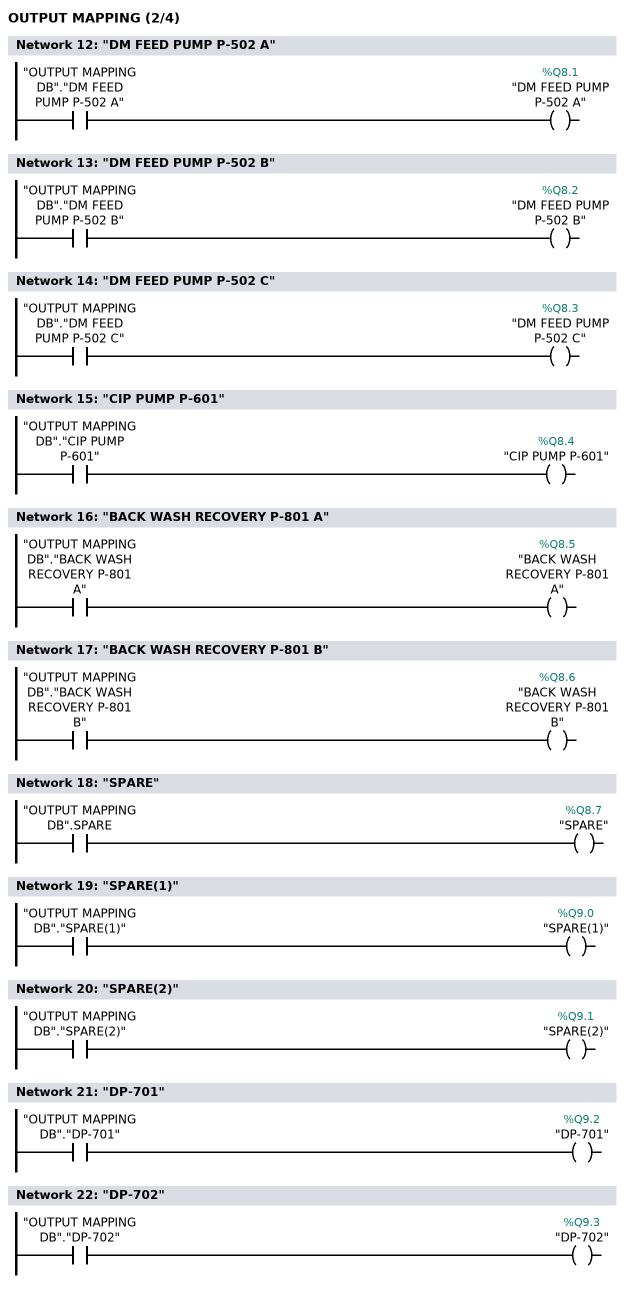
   RUNG wire#powerrail
      Contact( "OUTPUT MAPPING DB"."DM FEED PUMP P-502 A" )
      Coil( "DM FEED PUMP P-502 A" )
   END_RUNG
   // the same network as SCL:
   "DM FEED PUMP P-502 A" := "OUTPUT MAPPING DB"."DM FEED PUMP P-502 A";
END_REGION

REGION Network 13: "DM FEED PUMP P-502 B"
   RUNG wire#powerrail
      Contact( "OUTPUT MAPPING DB"."DM FEED PUMP P-502 B" )
      Coil( "DM FEED PUMP P-502 B" )
   END_RUNG
   // the same network as SCL:
   "DM FEED PUMP P-502 B" := "OUTPUT MAPPING DB"."DM FEED PUMP P-502 B";
END_REGION

REGION Network 14: "DM FEED PUMP P-502 C"
   RUNG wire#powerrail
      Contact( "OUTPUT MAPPING DB"."DM FEED PUMP P-502 C" )
      Coil( "DM FEED PUMP P-502 C" )
   END_RUNG
   // the same network as SCL:
   "DM FEED PUMP P-502 C" := "OUTPUT MAPPING DB"."DM FEED PUMP P-502 C";
END_REGION

REGION Network 15: "CIP PUMP P-601"
   RUNG wire#powerrail
      Contact( "OUTPUT MAPPING DB"."CIP PUMP P-601" )
      Coil( "CIP PUMP P-601" )
   END_RUNG
   // the same network as SCL:
   "CIP PUMP P-601" := "OUTPUT MAPPING DB"."CIP PUMP P-601";
END_REGION

REGION Network 16: "BACK WASH RECOVERY P-801 A"
   RUNG wire#powerrail
      Contact( "OUTPUT MAPPING DB"."BACK WASH RECOVERY P-801 A" )
      Coil( "BACK WASH RECOVERY P-801 A" )
   END_RUNG
   // the same network as SCL:
   "BACK WASH RECOVERY P-801 A" := "OUTPUT MAPPING DB"."BACK WASH RECOVERY P-801 A";
END_REGION

REGION Network 17: "BACK WASH RECOVERY P-801 B"
   RUNG wire#powerrail
      Contact( "OUTPUT MAPPING DB"."BACK WASH RECOVERY P-801 B" )
      Coil( "BACK WASH RECOVERY P-801 B" )
   END_RUNG
   // the same network as SCL:
   "BACK WASH RECOVERY P-801 B" := "OUTPUT MAPPING DB"."BACK WASH RECOVERY P-801 B";
END_REGION

REGION Network 18: "SPARE"
   RUNG wire#powerrail
      Contact( "OUTPUT MAPPING DB".SPARE )
      Coil( "SPARE" )
   END_RUNG
   // the same network as SCL:
   "SPARE" := "OUTPUT MAPPING DB".SPARE;
END_REGION

REGION Network 19: "SPARE(1)"
   RUNG wire#powerrail
      Contact( "OUTPUT MAPPING DB"."SPARE(1)" )
      Coil( "SPARE(1)" )
   END_RUNG
   // the same network as SCL:
   "SPARE(1)" := "OUTPUT MAPPING DB"."SPARE(1)";
END_REGION

REGION Network 20: "SPARE(2)"
   RUNG wire#powerrail
      Contact( "OUTPUT MAPPING DB"."SPARE(2)" )
      Coil( "SPARE(2)" )
   END_RUNG
   // the same network as SCL:
   "SPARE(2)" := "OUTPUT MAPPING DB"."SPARE(2)";
END_REGION

REGION Network 21: "DP-701"
   RUNG wire#powerrail
      Contact( "OUTPUT MAPPING DB"."DP-701" )
      Coil( "DP-701" )
   END_RUNG
   // the same network as SCL:
   "DP-701" := "OUTPUT MAPPING DB"."DP-701";
END_REGION

REGION Network 22: "DP-702"
   RUNG wire#powerrail
      Contact( "OUTPUT MAPPING DB"."DP-702" )
      Coil( "DP-702" )
   END_RUNG
   // the same network as SCL:
   "DP-702" := "OUTPUT MAPPING DB"."DP-702";
END_REGION

REGION Network 23: "NaOCL DOSING D-706 A"
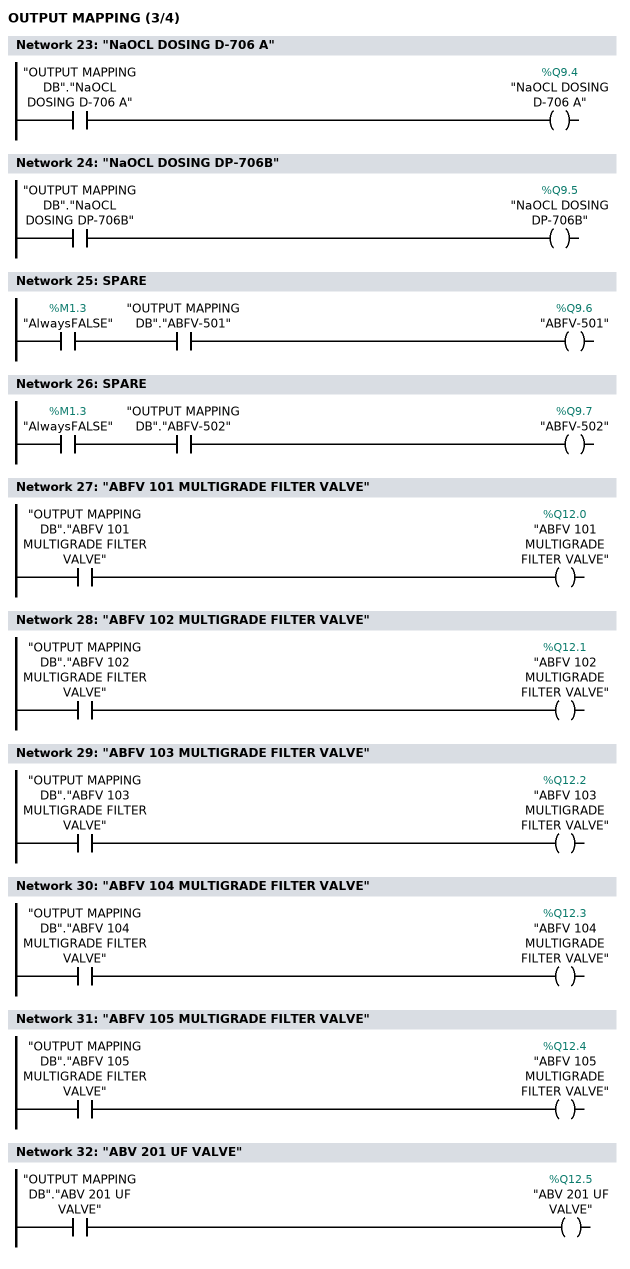
   RUNG wire#powerrail
      Contact( "OUTPUT MAPPING DB"."NaOCL DOSING D-706 A" )
      Coil( "NaOCL DOSING D-706 A" )
   END_RUNG
   // the same network as SCL:
   "NaOCL DOSING D-706 A" := "OUTPUT MAPPING DB"."NaOCL DOSING D-706 A";
END_REGION

REGION Network 24: "NaOCL DOSING DP-706B"
   RUNG wire#powerrail
      Contact( "OUTPUT MAPPING DB"."NaOCL DOSING DP-706B" )
      Coil( "NaOCL DOSING DP-706B" )
   END_RUNG
   // the same network as SCL:
   "NaOCL DOSING DP-706B" := "OUTPUT MAPPING DB"."NaOCL DOSING DP-706B";
END_REGION

REGION Network 25: SPARE
   RUNG wire#powerrail
      Contact( "AlwaysFALSE" )
      Contact( "OUTPUT MAPPING DB"."ABFV-501" )
      Coil( "ABFV-501" )
   END_RUNG
   // the same network as SCL:
   "ABFV-501" := "AlwaysFALSE" AND "OUTPUT MAPPING DB"."ABFV-501";
END_REGION

REGION Network 26: SPARE
   RUNG wire#powerrail
      Contact( "AlwaysFALSE" )
      Contact( "OUTPUT MAPPING DB"."ABFV-502" )
      Coil( "ABFV-502" )
   END_RUNG
   // the same network as SCL:
   "ABFV-502" := "AlwaysFALSE" AND "OUTPUT MAPPING DB"."ABFV-502";
END_REGION

REGION Network 27: "ABFV 101 MULTIGRADE FILTER VALVE"
   RUNG wire#powerrail
      Contact( "OUTPUT MAPPING DB"."ABFV 101 MULTIGRADE FILTER VALVE" )
      Coil( "ABFV 101 MULTIGRADE FILTER VALVE" )
   END_RUNG
   // the same network as SCL:
   "ABFV 101 MULTIGRADE FILTER VALVE" := "OUTPUT MAPPING DB"."ABFV 101 MULTIGRADE FILTER VALVE";
END_REGION

REGION Network 28: "ABFV 102 MULTIGRADE FILTER VALVE"
   RUNG wire#powerrail
      Contact( "OUTPUT MAPPING DB"."ABFV 102 MULTIGRADE FILTER VALVE" )
      Coil( "ABFV 102 MULTIGRADE FILTER VALVE" )
   END_RUNG
   // the same network as SCL:
   "ABFV 102 MULTIGRADE FILTER VALVE" := "OUTPUT MAPPING DB"."ABFV 102 MULTIGRADE FILTER VALVE";
END_REGION

REGION Network 29: "ABFV 103 MULTIGRADE FILTER VALVE"
   RUNG wire#powerrail
      Contact( "OUTPUT MAPPING DB"."ABFV 103 MULTIGRADE FILTER VALVE" )
      Coil( "ABFV 103 MULTIGRADE FILTER VALVE" )
   END_RUNG
   // the same network as SCL:
   "ABFV 103 MULTIGRADE FILTER VALVE" := "OUTPUT MAPPING DB"."ABFV 103 MULTIGRADE FILTER VALVE";
END_REGION

REGION Network 30: "ABFV 104 MULTIGRADE FILTER VALVE"
   RUNG wire#powerrail
      Contact( "OUTPUT MAPPING DB"."ABFV 104 MULTIGRADE FILTER VALVE" )
      Coil( "ABFV 104 MULTIGRADE FILTER VALVE" )
   END_RUNG
   // the same network as SCL:
   "ABFV 104 MULTIGRADE FILTER VALVE" := "OUTPUT MAPPING DB"."ABFV 104 MULTIGRADE FILTER VALVE";
END_REGION

REGION Network 31: "ABFV 105 MULTIGRADE FILTER VALVE"
   RUNG wire#powerrail
      Contact( "OUTPUT MAPPING DB"."ABFV 105 MULTIGRADE FILTER VALVE" )
      Coil( "ABFV 105 MULTIGRADE FILTER VALVE" )
   END_RUNG
   // the same network as SCL:
   "ABFV 105 MULTIGRADE FILTER VALVE" := "OUTPUT MAPPING DB"."ABFV 105 MULTIGRADE FILTER VALVE";
END_REGION

REGION Network 32: "ABV 201 UF VALVE"
   RUNG wire#powerrail
      Contact( "OUTPUT MAPPING DB"."ABV 201 UF VALVE" )
      Coil( "ABV 201 UF VALVE" )
   END_RUNG
   // the same network as SCL:
   "ABV 201 UF VALVE" := "OUTPUT MAPPING DB"."ABV 201 UF VALVE";
END_REGION

REGION Network 33: "ABFV 201 UF VALVE"
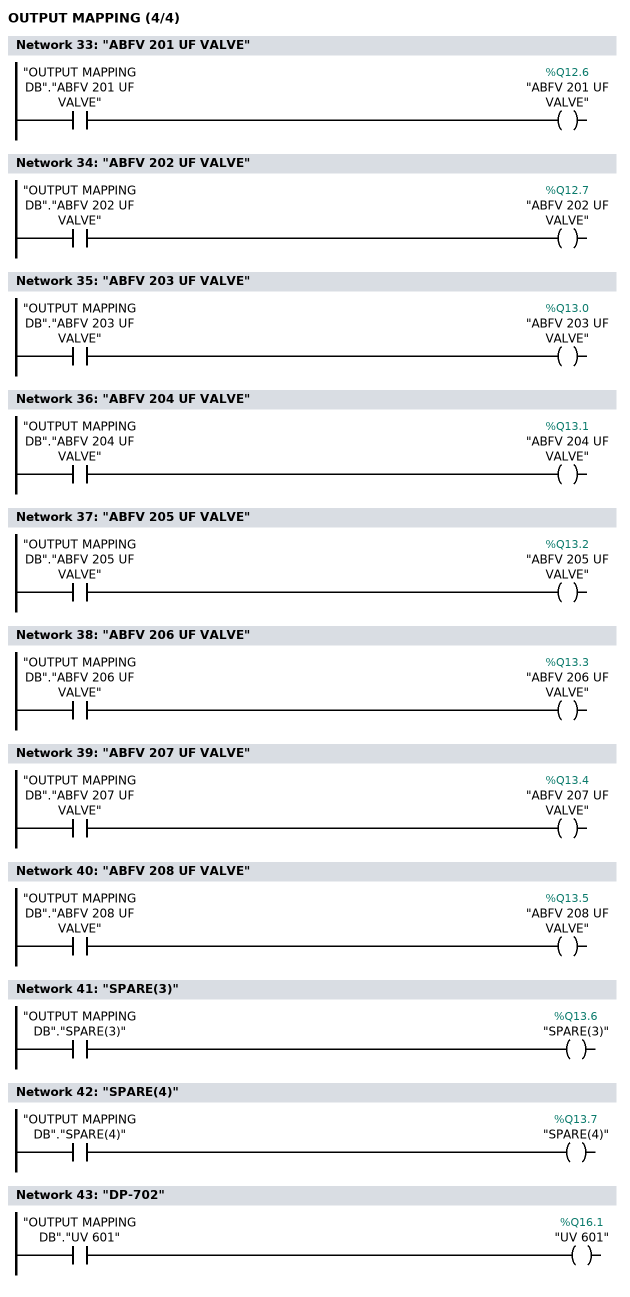
   RUNG wire#powerrail
      Contact( "OUTPUT MAPPING DB"."ABFV 201 UF VALVE" )
      Coil( "ABFV 201 UF VALVE" )
   END_RUNG
   // the same network as SCL:
   "ABFV 201 UF VALVE" := "OUTPUT MAPPING DB"."ABFV 201 UF VALVE";
END_REGION

REGION Network 34: "ABFV 202 UF VALVE"
   RUNG wire#powerrail
      Contact( "OUTPUT MAPPING DB"."ABFV 202 UF VALVE" )
      Coil( "ABFV 202 UF VALVE" )
   END_RUNG
   // the same network as SCL:
   "ABFV 202 UF VALVE" := "OUTPUT MAPPING DB"."ABFV 202 UF VALVE";
END_REGION

REGION Network 35: "ABFV 203 UF VALVE"
   RUNG wire#powerrail
      Contact( "OUTPUT MAPPING DB"."ABFV 203 UF VALVE" )
      Coil( "ABFV 203 UF VALVE" )
   END_RUNG
   // the same network as SCL:
   "ABFV 203 UF VALVE" := "OUTPUT MAPPING DB"."ABFV 203 UF VALVE";
END_REGION

REGION Network 36: "ABFV 204 UF VALVE"
   RUNG wire#powerrail
      Contact( "OUTPUT MAPPING DB"."ABFV 204 UF VALVE" )
      Coil( "ABFV 204 UF VALVE" )
   END_RUNG
   // the same network as SCL:
   "ABFV 204 UF VALVE" := "OUTPUT MAPPING DB"."ABFV 204 UF VALVE";
END_REGION

REGION Network 37: "ABFV 205 UF VALVE"
   RUNG wire#powerrail
      Contact( "OUTPUT MAPPING DB"."ABFV 205 UF VALVE" )
      Coil( "ABFV 205 UF VALVE" )
   END_RUNG
   // the same network as SCL:
   "ABFV 205 UF VALVE" := "OUTPUT MAPPING DB"."ABFV 205 UF VALVE";
END_REGION

REGION Network 38: "ABFV 206 UF VALVE"
   RUNG wire#powerrail
      Contact( "OUTPUT MAPPING DB"."ABFV 206 UF VALVE" )
      Coil( "ABFV 206 UF VALVE" )
   END_RUNG
   // the same network as SCL:
   "ABFV 206 UF VALVE" := "OUTPUT MAPPING DB"."ABFV 206 UF VALVE";
END_REGION

REGION Network 39: "ABFV 207 UF VALVE"
   RUNG wire#powerrail
      Contact( "OUTPUT MAPPING DB"."ABFV 207 UF VALVE" )
      Coil( "ABFV 207 UF VALVE" )
   END_RUNG
   // the same network as SCL:
   "ABFV 207 UF VALVE" := "OUTPUT MAPPING DB"."ABFV 207 UF VALVE";
END_REGION

REGION Network 40: "ABFV 208 UF VALVE"
   RUNG wire#powerrail
      Contact( "OUTPUT MAPPING DB"."ABFV 208 UF VALVE" )
      Coil( "ABFV 208 UF VALVE" )
   END_RUNG
   // the same network as SCL:
   "ABFV 208 UF VALVE" := "OUTPUT MAPPING DB"."ABFV 208 UF VALVE";
END_REGION

REGION Network 41: "SPARE(3)"
   RUNG wire#powerrail
      Contact( "OUTPUT MAPPING DB"."SPARE(3)" )
      Coil( "SPARE(3)" )
   END_RUNG
   // the same network as SCL:
   "SPARE(3)" := "OUTPUT MAPPING DB"."SPARE(3)";
END_REGION

REGION Network 42: "SPARE(4)"
   RUNG wire#powerrail
      Contact( "OUTPUT MAPPING DB"."SPARE(4)" )
      Coil( "SPARE(4)" )
   END_RUNG
   // the same network as SCL:
   "SPARE(4)" := "OUTPUT MAPPING DB"."SPARE(4)";
END_REGION

REGION Network 43: "DP-702"
   RUNG wire#powerrail
      Contact( "OUTPUT MAPPING DB"."UV 601" )
      Coil( "UV 601" )
   END_RUNG
   // the same network as SCL:
   "UV 601" := "OUTPUT MAPPING DB"."UV 601";
END_REGION
END_FUNCTION

FUNCTION "MODE SELECTION" : Void   // FC1, LAD
{ S7_Optimized_Access := 'TRUE' }
// stored: SetENOAutomatically false
   VAR_TEMP   // added for the SCL form of the ladder/FBD networks
      _w1 : Bool;
   END_VAR
BEGIN

REGION Network 1: STANDBY///////////////////////////////////// MGF ////////////////////////////////////////
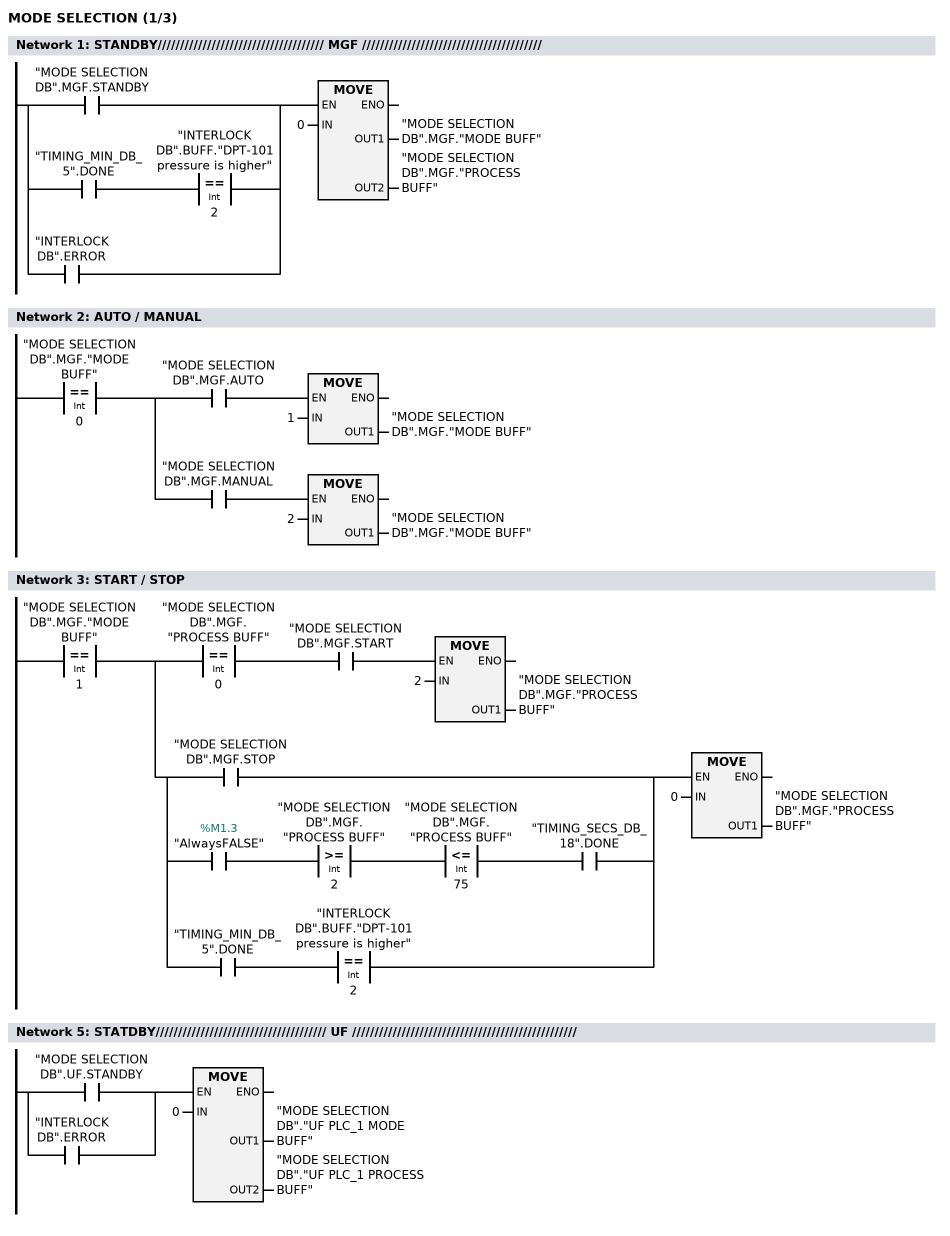
   RUNG wire#powerrail
      Contact( "MODE SELECTION DB".MGF.STANDBY )
      wire#w1
      Move(in := 0, out1 => "MODE SELECTION DB".MGF."MODE BUFF", out2 => "MODE SELECTION DB".MGF."PROCESS BUFF")
   END_RUNG
   RUNG wire#powerrail
      Contact( "TIMING_MIN_DB_5".DONE )
      { S7_Templates := "SrcType := Int" } EQ_Contact(in1 := "INTERLOCK DB".BUFF."DPT-101 pressure is higher", in2 := 2)
   END_RUNG wire#w1
   RUNG wire#powerrail
      Contact( "INTERLOCK DB".ERROR )
   END_RUNG wire#w1
   // the same network as SCL:
   IF "MODE SELECTION DB".MGF.STANDBY OR ("TIMING_MIN_DB_5".DONE AND ("INTERLOCK DB".BUFF."DPT-101 pressure is higher" = 2)) OR "INTERLOCK DB".ERROR THEN
       "MODE SELECTION DB".MGF."MODE BUFF" := 0;
       "MODE SELECTION DB".MGF."PROCESS BUFF" := 0;
   END_IF;
END_REGION

REGION Network 2: AUTO / MANUAL
   RUNG wire#powerrail
      { S7_Templates := "SrcType := Int" } EQ_Contact(in1 := "MODE SELECTION DB".MGF."MODE BUFF", in2 := 0)
      wire#w1
      Contact( "MODE SELECTION DB".MGF.AUTO )
      Move(in := 1, out1 => "MODE SELECTION DB".MGF."MODE BUFF")
   END_RUNG
   RUNG wire#w1
      Contact( "MODE SELECTION DB".MGF.MANUAL )
      Move(in := 2, out1 => "MODE SELECTION DB".MGF."MODE BUFF")
   END_RUNG
   // the same network as SCL:
   #_w1 := "MODE SELECTION DB".MGF."MODE BUFF" = 0;
   IF #_w1 AND "MODE SELECTION DB".MGF.AUTO THEN "MODE SELECTION DB".MGF."MODE BUFF" := 1; END_IF;
   IF #_w1 AND "MODE SELECTION DB".MGF.MANUAL THEN "MODE SELECTION DB".MGF."MODE BUFF" := 2; END_IF;
END_REGION

REGION Network 3: START / STOP
   RUNG wire#powerrail
      { S7_Templates := "SrcType := Int" } EQ_Contact(in1 := "MODE SELECTION DB".MGF."MODE BUFF", in2 := 1)
      wire#w1
      { S7_Templates := "SrcType := Int" } EQ_Contact(in1 := "MODE SELECTION DB".MGF."PROCESS BUFF", in2 := 0)
      Contact( "MODE SELECTION DB".MGF.START )
      Move(in := 2, out1 => "MODE SELECTION DB".MGF."PROCESS BUFF")
   END_RUNG
   RUNG wire#w1
      Contact( "MODE SELECTION DB".MGF.STOP )
      wire#w2
      Move(in := 0, out1 => "MODE SELECTION DB".MGF."PROCESS BUFF")
   END_RUNG
   RUNG wire#w1
      Contact( "AlwaysFALSE" )
      { S7_Templates := "SrcType := Int" } GE_Contact(in1 := "MODE SELECTION DB".MGF."PROCESS BUFF", in2 := 2)
      { S7_Templates := "SrcType := Int" } LE_Contact(in1 := "MODE SELECTION DB".MGF."PROCESS BUFF", in2 := 75)
      Contact( "TIMING_SECS_DB_18".DONE )
   END_RUNG wire#w2
   RUNG wire#w1
      Contact( "TIMING_MIN_DB_5".DONE )
      { S7_Templates := "SrcType := Int" } EQ_Contact(in1 := "INTERLOCK DB".BUFF."DPT-101 pressure is higher", in2 := 2)
   END_RUNG wire#w2
   // the same network as SCL:
   #_w1 := "MODE SELECTION DB".MGF."MODE BUFF" = 1;
   IF #_w1 AND ("MODE SELECTION DB".MGF."PROCESS BUFF" = 0) AND "MODE SELECTION DB".MGF.START THEN
       "MODE SELECTION DB".MGF."PROCESS BUFF" := 2;
   END_IF;
   IF #_w1 AND ("MODE SELECTION DB".MGF.STOP OR ("AlwaysFALSE" AND ("MODE SELECTION DB".MGF."PROCESS BUFF" >= 2) AND ("MODE SELECTION DB".MGF."PROCESS BUFF" <= 75) AND "TIMING_SECS_DB_18".DONE) OR ("TIMING_MIN_DB_5".DONE AND ("INTERLOCK DB".BUFF."DPT-101 pressure is higher" = 2))) THEN
       "MODE SELECTION DB".MGF."PROCESS BUFF" := 0;
   END_IF;
END_REGION

REGION Network 5: STATDBY////////////////////////////////////// UF //////////////////////////////////////////////////
   RUNG wire#powerrail
      Contact( "MODE SELECTION DB".UF.STANDBY )
      wire#w1
      Move(in := 0, out1 => "MODE SELECTION DB"."UF PLC_1 MODE BUFF", out2 => "MODE SELECTION DB"."UF PLC_1 PROCESS BUFF")
   END_RUNG
   RUNG wire#powerrail
      Contact( "INTERLOCK DB".ERROR )
   END_RUNG wire#w1
   // the same network as SCL:
   IF "MODE SELECTION DB".UF.STANDBY OR "INTERLOCK DB".ERROR THEN
       "MODE SELECTION DB"."UF PLC_1 MODE BUFF" := 0;
       "MODE SELECTION DB"."UF PLC_1 PROCESS BUFF" := 0;
   END_IF;
END_REGION

REGION Network 6: AUTO / MANUAL
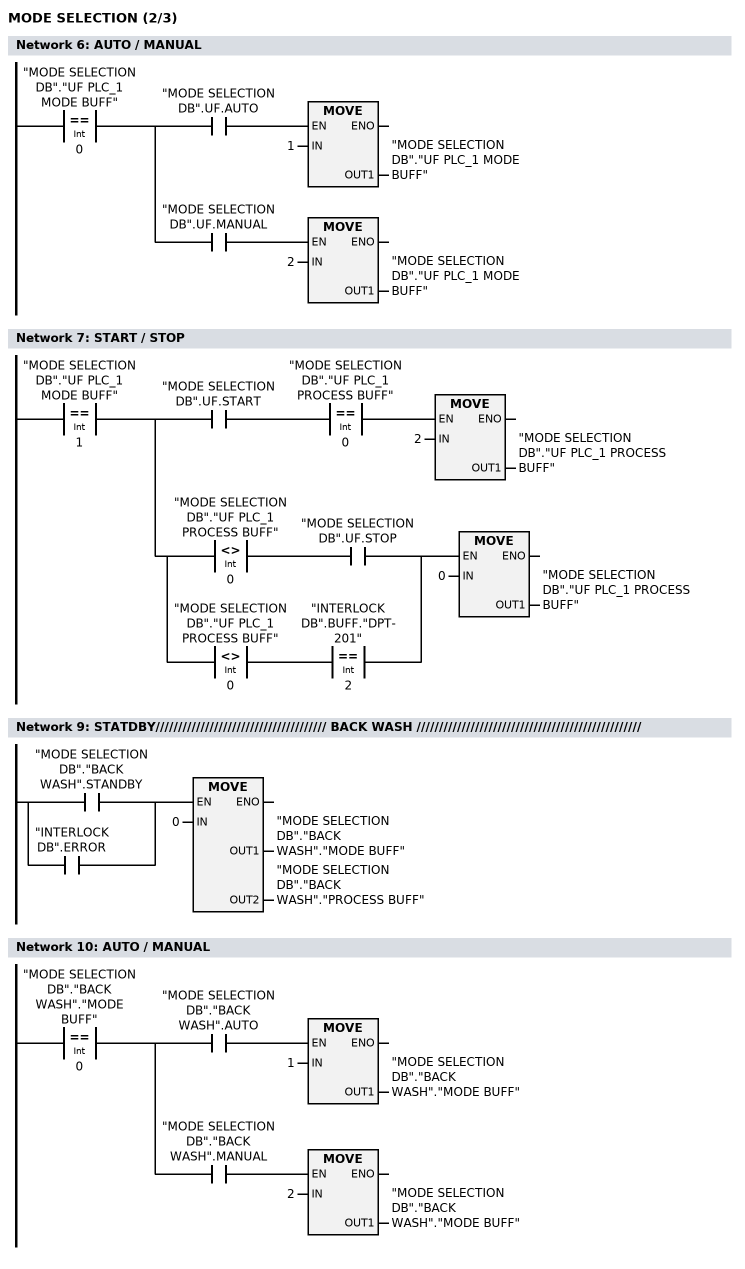
   RUNG wire#powerrail
      { S7_Templates := "SrcType := Int" } EQ_Contact(in1 := "MODE SELECTION DB"."UF PLC_1 MODE BUFF", in2 := 0)
      wire#w1
      Contact( "MODE SELECTION DB".UF.AUTO )
      Move(in := 1, out1 => "MODE SELECTION DB"."UF PLC_1 MODE BUFF")
   END_RUNG
   RUNG wire#w1
      Contact( "MODE SELECTION DB".UF.MANUAL )
      Move(in := 2, out1 => "MODE SELECTION DB"."UF PLC_1 MODE BUFF")
   END_RUNG
   // the same network as SCL:
   #_w1 := "MODE SELECTION DB"."UF PLC_1 MODE BUFF" = 0;
   IF #_w1 AND "MODE SELECTION DB".UF.AUTO THEN "MODE SELECTION DB"."UF PLC_1 MODE BUFF" := 1; END_IF;
   IF #_w1 AND "MODE SELECTION DB".UF.MANUAL THEN "MODE SELECTION DB"."UF PLC_1 MODE BUFF" := 2; END_IF;
END_REGION

REGION Network 7: START / STOP
   RUNG wire#powerrail
      { S7_Templates := "SrcType := Int" } EQ_Contact(in1 := "MODE SELECTION DB"."UF PLC_1 MODE BUFF", in2 := 1)
      wire#w1
      Contact( "MODE SELECTION DB".UF.START )
      { S7_Templates := "SrcType := Int" } EQ_Contact(in1 := "MODE SELECTION DB"."UF PLC_1 PROCESS BUFF", in2 := 0)
      Move(in := 2, out1 => "MODE SELECTION DB"."UF PLC_1 PROCESS BUFF")
   END_RUNG
   RUNG wire#w1
      { S7_Templates := "SrcType := Int" } NE_Contact(in1 := "MODE SELECTION DB"."UF PLC_1 PROCESS BUFF", in2 := 0)
      Contact( "MODE SELECTION DB".UF.STOP )
      wire#w2
      Move(in := 0, out1 => "MODE SELECTION DB"."UF PLC_1 PROCESS BUFF")
   END_RUNG
   RUNG wire#w1
      { S7_Templates := "SrcType := Int" } NE_Contact(in1 := "MODE SELECTION DB"."UF PLC_1 PROCESS BUFF", in2 := 0)
      { S7_Templates := "SrcType := Int" } EQ_Contact(in1 := "INTERLOCK DB".BUFF."DPT-201", in2 := 2)
   END_RUNG wire#w2
   // the same network as SCL:
   #_w1 := "MODE SELECTION DB"."UF PLC_1 MODE BUFF" = 1;
   IF #_w1 AND "MODE SELECTION DB".UF.START AND ("MODE SELECTION DB"."UF PLC_1 PROCESS BUFF" = 0) THEN
       "MODE SELECTION DB"."UF PLC_1 PROCESS BUFF" := 2;
   END_IF;
   IF #_w1 AND ((("MODE SELECTION DB"."UF PLC_1 PROCESS BUFF" <> 0) AND "MODE SELECTION DB".UF.STOP) OR (("MODE SELECTION DB"."UF PLC_1 PROCESS BUFF" <> 0) AND ("INTERLOCK DB".BUFF."DPT-201" = 2))) THEN
       "MODE SELECTION DB"."UF PLC_1 PROCESS BUFF" := 0;
   END_IF;
END_REGION

REGION Network 9: STATDBY////////////////////////////////////// BACK WASH //////////////////////////////////////////////////
   RUNG wire#powerrail
      Contact( "MODE SELECTION DB"."BACK WASH".STANDBY )
      wire#w1
      Move(in := 0, out1 => "MODE SELECTION DB"."BACK WASH"."MODE BUFF", out2 => "MODE SELECTION DB"."BACK WASH"."PROCESS BUFF")
   END_RUNG
   RUNG wire#powerrail
      Contact( "INTERLOCK DB".ERROR )
   END_RUNG wire#w1
   // the same network as SCL:
   IF "MODE SELECTION DB"."BACK WASH".STANDBY OR "INTERLOCK DB".ERROR THEN
       "MODE SELECTION DB"."BACK WASH"."MODE BUFF" := 0;
       "MODE SELECTION DB"."BACK WASH"."PROCESS BUFF" := 0;
   END_IF;
END_REGION

REGION Network 10: AUTO / MANUAL
   RUNG wire#powerrail
      { S7_Templates := "SrcType := Int" } EQ_Contact(in1 := "MODE SELECTION DB"."BACK WASH"."MODE BUFF", in2 := 0)
      wire#w1
      Contact( "MODE SELECTION DB"."BACK WASH".AUTO )
      Move(in := 1, out1 => "MODE SELECTION DB"."BACK WASH"."MODE BUFF")
   END_RUNG
   RUNG wire#w1
      Contact( "MODE SELECTION DB"."BACK WASH".MANUAL )
      Move(in := 2, out1 => "MODE SELECTION DB"."BACK WASH"."MODE BUFF")
   END_RUNG
   // the same network as SCL:
   #_w1 := "MODE SELECTION DB"."BACK WASH"."MODE BUFF" = 0;
   IF #_w1 AND "MODE SELECTION DB"."BACK WASH".AUTO THEN
       "MODE SELECTION DB"."BACK WASH"."MODE BUFF" := 1;
   END_IF;
   IF #_w1 AND "MODE SELECTION DB"."BACK WASH".MANUAL THEN
       "MODE SELECTION DB"."BACK WASH"."MODE BUFF" := 2;
   END_IF;
END_REGION

REGION Network 11: START / STOP
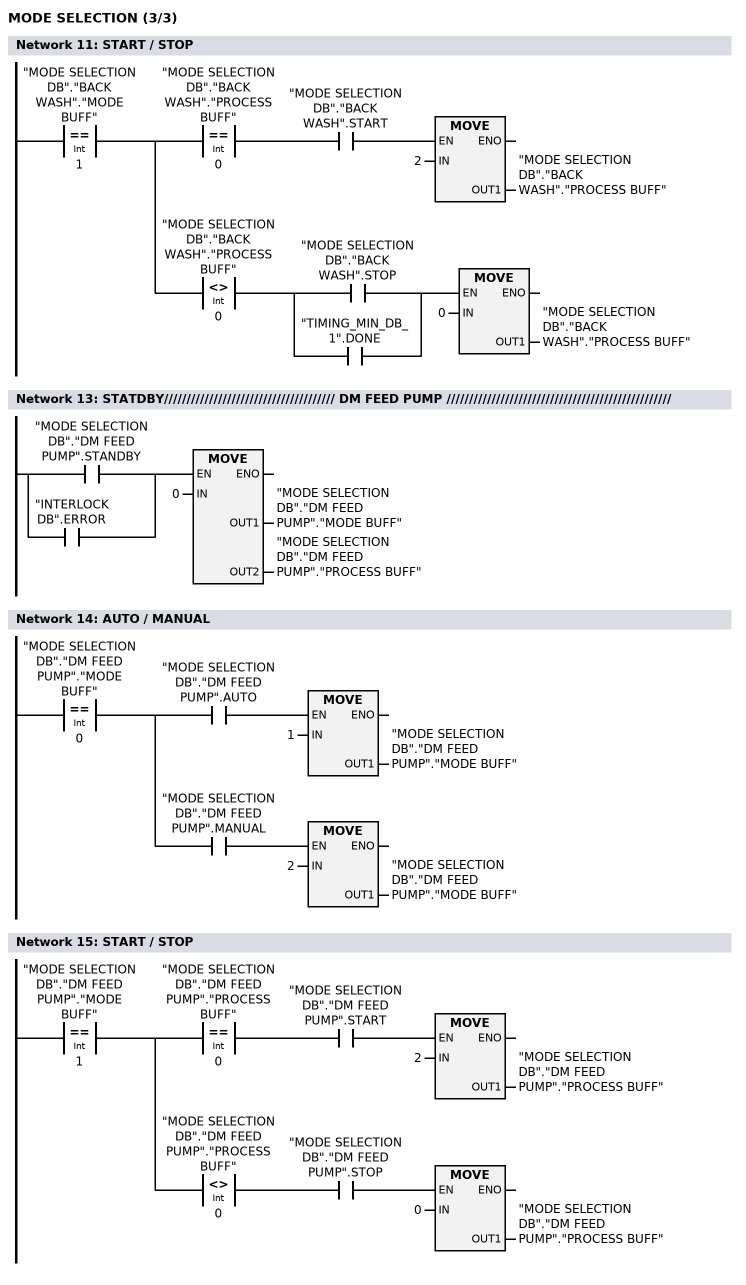
   RUNG wire#powerrail
      { S7_Templates := "SrcType := Int" } EQ_Contact(in1 := "MODE SELECTION DB"."BACK WASH"."MODE BUFF", in2 := 1)
      wire#w1
      { S7_Templates := "SrcType := Int" } EQ_Contact(in1 := "MODE SELECTION DB"."BACK WASH"."PROCESS BUFF", in2 := 0)
      Contact( "MODE SELECTION DB"."BACK WASH".START )
      Move(in := 2, out1 => "MODE SELECTION DB"."BACK WASH"."PROCESS BUFF")
   END_RUNG
   RUNG wire#w1
      { S7_Templates := "SrcType := Int" } NE_Contact(in1 := "MODE SELECTION DB"."BACK WASH"."PROCESS BUFF", in2 := 0)
      wire#w2
      Contact( "MODE SELECTION DB"."BACK WASH".STOP )
      wire#w3
      Move(in := 0, out1 => "MODE SELECTION DB"."BACK WASH"."PROCESS BUFF")
   END_RUNG
   RUNG wire#w2
      Contact( "TIMING_MIN_DB_1".DONE )
   END_RUNG wire#w3
   // the same network as SCL:
   #_w1 := "MODE SELECTION DB"."BACK WASH"."MODE BUFF" = 1;
   IF #_w1 AND ("MODE SELECTION DB"."BACK WASH"."PROCESS BUFF" = 0) AND "MODE SELECTION DB"."BACK WASH".START THEN
       "MODE SELECTION DB"."BACK WASH"."PROCESS BUFF" := 2;
   END_IF;
   IF #_w1 AND ("MODE SELECTION DB"."BACK WASH"."PROCESS BUFF" <> 0) AND ("MODE SELECTION DB"."BACK WASH".STOP OR "TIMING_MIN_DB_1".DONE) THEN
       "MODE SELECTION DB"."BACK WASH"."PROCESS BUFF" := 0;
   END_IF;
END_REGION

REGION Network 13: STATDBY////////////////////////////////////// DM FEED PUMP //////////////////////////////////////////////////
   RUNG wire#powerrail
      Contact( "MODE SELECTION DB"."DM FEED PUMP".STANDBY )
      wire#w1
      Move(in := 0, out1 => "MODE SELECTION DB"."DM FEED PUMP"."MODE BUFF", out2 => "MODE SELECTION DB"."DM FEED PUMP"."PROCESS BUFF")
   END_RUNG
   RUNG wire#powerrail
      Contact( "INTERLOCK DB".ERROR )
   END_RUNG wire#w1
   // the same network as SCL:
   IF "MODE SELECTION DB"."DM FEED PUMP".STANDBY OR "INTERLOCK DB".ERROR THEN
       "MODE SELECTION DB"."DM FEED PUMP"."MODE BUFF" := 0;
       "MODE SELECTION DB"."DM FEED PUMP"."PROCESS BUFF" := 0;
   END_IF;
END_REGION

REGION Network 14: AUTO / MANUAL
   RUNG wire#powerrail
      { S7_Templates := "SrcType := Int" } EQ_Contact(in1 := "MODE SELECTION DB"."DM FEED PUMP"."MODE BUFF", in2 := 0)
      wire#w1
      Contact( "MODE SELECTION DB"."DM FEED PUMP".AUTO )
      Move(in := 1, out1 => "MODE SELECTION DB"."DM FEED PUMP"."MODE BUFF")
   END_RUNG
   RUNG wire#w1
      Contact( "MODE SELECTION DB"."DM FEED PUMP".MANUAL )
      Move(in := 2, out1 => "MODE SELECTION DB"."DM FEED PUMP"."MODE BUFF")
   END_RUNG
   // the same network as SCL:
   #_w1 := "MODE SELECTION DB"."DM FEED PUMP"."MODE BUFF" = 0;
   IF #_w1 AND "MODE SELECTION DB"."DM FEED PUMP".AUTO THEN
       "MODE SELECTION DB"."DM FEED PUMP"."MODE BUFF" := 1;
   END_IF;
   IF #_w1 AND "MODE SELECTION DB"."DM FEED PUMP".MANUAL THEN
       "MODE SELECTION DB"."DM FEED PUMP"."MODE BUFF" := 2;
   END_IF;
END_REGION

REGION Network 15: START / STOP
   RUNG wire#powerrail
      { S7_Templates := "SrcType := Int" } EQ_Contact(in1 := "MODE SELECTION DB"."DM FEED PUMP"."MODE BUFF", in2 := 1)
      wire#w1
      { S7_Templates := "SrcType := Int" } EQ_Contact(in1 := "MODE SELECTION DB"."DM FEED PUMP"."PROCESS BUFF", in2 := 0)
      Contact( "MODE SELECTION DB"."DM FEED PUMP".START )
      Move(in := 2, out1 => "MODE SELECTION DB"."DM FEED PUMP"."PROCESS BUFF")
   END_RUNG
   RUNG wire#w1
      { S7_Templates := "SrcType := Int" } NE_Contact(in1 := "MODE SELECTION DB"."DM FEED PUMP"."PROCESS BUFF", in2 := 0)
      Contact( "MODE SELECTION DB"."DM FEED PUMP".STOP )
      Move(in := 0, out1 => "MODE SELECTION DB"."DM FEED PUMP"."PROCESS BUFF")
   END_RUNG
   // the same network as SCL:
   #_w1 := "MODE SELECTION DB"."DM FEED PUMP"."MODE BUFF" = 1;
   IF #_w1 AND ("MODE SELECTION DB"."DM FEED PUMP"."PROCESS BUFF" = 0) AND "MODE SELECTION DB"."DM FEED PUMP".START THEN
       "MODE SELECTION DB"."DM FEED PUMP"."PROCESS BUFF" := 2;
   END_IF;
   IF #_w1 AND ("MODE SELECTION DB"."DM FEED PUMP"."PROCESS BUFF" <> 0) AND "MODE SELECTION DB"."DM FEED PUMP".STOP THEN
       "MODE SELECTION DB"."DM FEED PUMP"."PROCESS BUFF" := 0;
   END_IF;
END_REGION
END_FUNCTION

FUNCTION "FLUSH VALVE" : Void
{ S7_Optimized_Access := 'TRUE' }
VERSION : 0.1

BEGIN
	
	"ABFV 101 MULTIGRADE FILTER FULSH"("SUBOUTPUT VALVE":="OUTPUT MAPPING DB"."ABFV 101 MULTIGRADE FILTER VALVE",
	                                   "OPEN FEEDBACK":="INPUT MAPPING DB"."ABFV-101 FEED BACK OPEN FEED BACK",
	                                   "CLOSE FEEDBACK":="INPUT MAPPING DB"."ABFV-101 FEED BACK CLOSE FEED BACK",
	                                   "OPEN OUTPUT VAVLE"=>"FLUSH DB"."ABFV 101 MULTIGRADE FILTER VALVE",
	                                   "CLOSE OUTPUT VAVLE"=>"FLUSH DB"."ABFV 101 MULTIGRADE FILTER VALVE_CLOSE");
	
	
	"ABFV 102 MULTIGRADE FILTER FLUSH"("SUBOUTPUT VALVE":="OUTPUT MAPPING DB"."ABFV 102 MULTIGRADE FILTER VALVE",
	                                   "OPEN FEEDBACK":="INPUT MAPPING DB"."ABFV-102 FEED BACK OPEN FEED BACK",
	                                   "CLOSE FEEDBACK":="INPUT MAPPING DB"."ABFV-102 FEED BACK CLOSE FEED BACK",
	                                   "OPEN OUTPUT VAVLE"=>"FLUSH DB"."ABFV 102 MULTIGRADE FILTER VALVE",
	                                   "CLOSE OUTPUT VAVLE"=>"FLUSH DB"."ABFV 102 MULTIGRADE FILTER VALVE_CLOSE");
	
	"ABFV 103 MULTIGRADE FILTER FLUSH"("SUBOUTPUT VALVE":="OUTPUT MAPPING DB"."ABFV 103 MULTIGRADE FILTER VALVE",
	                                   "OPEN FEEDBACK":="INPUT MAPPING DB"."ABFV-103 FEED BACK OPEN FEED BACK",
	                                   "CLOSE FEEDBACK":="INPUT MAPPING DB"."ABFV-103 FEED BACK CLOSE FEED BACK",
	                                   "OPEN OUTPUT VAVLE"=>"FLUSH DB"."ABFV 103 MULTIGRADE FILTER VALVE",
	                                   "CLOSE OUTPUT VAVLE"=>"FLUSH DB"."ABFV 103 MULTIGRADE FILTER VALVE_CLOSE");
	
	"ABFV 104 MULTIGRADE FILTER FLUSH"("SUBOUTPUT VALVE":="OUTPUT MAPPING DB"."ABFV 104 MULTIGRADE FILTER VALVE",
	                                   "OPEN FEEDBACK":="INPUT MAPPING DB"."ABFV-104 FEED BACK OPEN FEED BACK",
	                                   "CLOSE FEEDBACK":="INPUT MAPPING DB"."ABFV-104 FEED BACK CLOSE FEED BACK",
	                                   "OPEN OUTPUT VAVLE"=>"FLUSH DB"."ABFV 104 MULTIGRADE FILTER VALVE",
	                                   "CLOSE OUTPUT VAVLE"=>"FLUSH DB"."ABFV 104 MULTIGRADE FILTER VALVE_CLOSE");
	
	"ABFV 105 MULTIGRADE FILTER FLUSH"("SUBOUTPUT VALVE":="OUTPUT MAPPING DB"."ABFV 105 MULTIGRADE FILTER VALVE",
	                                   "OPEN FEEDBACK":="INPUT MAPPING DB"."ABFV 105 FEED BACK OPEN",
	                                   "CLOSE FEEDBACK":="INPUT MAPPING DB"."ABFV 105 FEED BACK CLOSE",
	                                   "OPEN OUTPUT VAVLE"=>"FLUSH DB"."ABFV 105 MULTIGRADE FILTER VALVE",
	                                   "CLOSE OUTPUT VAVLE"=>"FLUSH DB"."ABFV 105 MULTIGRADE FILTER VALVE_CLOSE");
	
	"ABV 201 FEED BACK FLUSH"("SUBOUTPUT VALVE":="OUTPUT MAPPING DB"."ABV 201 UF VALVE",
	                          "OPEN FEEDBACK":="INPUT MAPPING DB"."ABV 201 FEED BACK OPEN",
	                          "CLOSE FEEDBACK":="INPUT MAPPING DB"."ABV 201 FEED BACK CLOSE",
	                          "OPEN OUTPUT VAVLE"=>"FLUSH DB"."ABV 201 UF VALVE",
	                          "CLOSE OUTPUT VAVLE"=>"FLUSH DB"."ABV 201 UF VALVE_CLOSE");
	
	"ABFV 201 FEED BACK FLUSH"("SUBOUTPUT VALVE":="OUTPUT MAPPING DB"."ABFV 201 UF VALVE",
	                           "OPEN FEEDBACK":="INPUT MAPPING DB"."ABFV 201 FEED BACK OPEN",
	                           "CLOSE FEEDBACK":="INPUT MAPPING DB"."ABFV 201 FEED BACK CLOSE",
	                           "OPEN OUTPUT VAVLE"=>"FLUSH DB"."ABFV 201 UF VALVE",
	                           "CLOSE OUTPUT VAVLE"=>"FLUSH DB"."ABFV 201 UF VALVE_CLOSE");
	
	
	"ABFV 202 FEED BACK FLUSH"("SUBOUTPUT VALVE":="OUTPUT MAPPING DB"."ABFV 202 UF VALVE",
	                           "OPEN FEEDBACK":="INPUT MAPPING DB"."ABFV 202 FEED BACK OPEN",
	                           "CLOSE FEEDBACK":="INPUT MAPPING DB"."ABFV 202 FEED BACK CLOSE",
	                           "OPEN OUTPUT VAVLE"=>"FLUSH DB"."ABFV 202 UF VALVE",
	                           "CLOSE OUTPUT VAVLE"=>"FLUSH DB"."ABFV 202 UF VALVE_CLOSE");
	
	"ABFV 203 FEED BACK FLUSH"("SUBOUTPUT VALVE":="OUTPUT MAPPING DB"."ABFV 203 UF VALVE",
	                           "OPEN FEEDBACK":="INPUT MAPPING DB"."ABFV 203 FEED BACK OPEN",
	                           "CLOSE FEEDBACK":="INPUT MAPPING DB"."ABFV 203 FEED BACK CLOSE",
	                           "OPEN OUTPUT VAVLE"=>"FLUSH DB"."ABFV 203 UF VALVE",
	                           "CLOSE OUTPUT VAVLE"=>"FLUSH DB"."ABFV 203 UF VALVE_CLOSE");
	
	"ABFV 204 FEED BACK FLUSH"("SUBOUTPUT VALVE":="OUTPUT MAPPING DB"."ABFV 204 UF VALVE",
	                           "OPEN FEEDBACK":="INPUT MAPPING DB"."ABFV 204 FEED BACK OPEN",
	                           "CLOSE FEEDBACK":="INPUT MAPPING DB"."ABFV 204 FEED BACK CLOSE",
	                           "OPEN OUTPUT VAVLE"=>"FLUSH DB"."ABFV 204 UF VALVE",
	                           "CLOSE OUTPUT VAVLE"=>"FLUSH DB"."ABFV 204 UF VALVE_CLOSE");
	
	"ABFV 205 FEED BACK FLUSH"("SUBOUTPUT VALVE":="OUTPUT MAPPING DB"."ABFV 205 UF VALVE",
	                           "OPEN FEEDBACK":="INPUT MAPPING DB"."ABFV 205 FEED BACK OPEN",
	                           "CLOSE FEEDBACK":="INPUT MAPPING DB"."ABFV 205 FEED BACK CLOSE",
	                           "OPEN OUTPUT VAVLE"=>"FLUSH DB"."ABFV 205 UF VALVE",
	                           "CLOSE OUTPUT VAVLE"=>"FLUSH DB"."ABFV 205 UF VALVE_CLOSE");
	
	"ABFV 206 FEED BACK FLUSH"("SUBOUTPUT VALVE":="OUTPUT MAPPING DB"."ABFV 206 UF VALVE",
	                           "OPEN FEEDBACK":="INPUT MAPPING DB"."ABFV 206 FEED BACK OPEN",
	                           "CLOSE FEEDBACK":="INPUT MAPPING DB"."ABFV 206 FEED BACK CLOSE",
	                           "OPEN OUTPUT VAVLE"=>"FLUSH DB"."ABFV 206 UF VALVE",
	                           "CLOSE OUTPUT VAVLE"=>"FLUSH DB"."ABFV 206 UF VALVE_CLOSE");
	
	"ABFV 207 FEED BACK FLUSH"("SUBOUTPUT VALVE":="OUTPUT MAPPING DB"."ABFV 207 UF VALVE",
	                           "OPEN FEEDBACK":="INPUT MAPPING DB"."ABFV-207 FEED BACK OPEN",
	                           "CLOSE FEEDBACK":="INPUT MAPPING DB"."ABFV-207 FEED BACK CLOSE",
	                           "OPEN OUTPUT VAVLE"=>"FLUSH DB"."ABFV 207 UF VALVE",
	                           "CLOSE OUTPUT VAVLE"=>"FLUSH DB"."ABFV 207 UF VALVE_CLOSE");
	
	"ABFV 208 FEED BACK FLUSH"("SUBOUTPUT VALVE":="OUTPUT MAPPING DB"."ABFV 208 UF VALVE",
	                           "OPEN FEEDBACK":="INPUT MAPPING DB"."ABFV-208 FEED BACK OPEN",
	                           "CLOSE FEEDBACK":="INPUT MAPPING DB"."ABFV-208 FEED BACK CLOSE",
	                           "OPEN OUTPUT VAVLE"=>"FLUSH DB"."ABFV 208 UF VALVE",
	                           "CLOSE OUTPUT VAVLE"=>"FLUSH DB"."ABFV 208 UF VALVE_CLOSE");
	
	
	
	
	
	
END_FUNCTION

FUNCTION "INTERLOCK" : Void   // FC7, LAD
{ S7_Optimized_Access := 'TRUE' }
// stored: SetENOAutomatically false
   VAR_TEMP   // added for the SCL form of the ladder/FBD networks
      _w1 : Bool;
      _w2 : Bool;
   END_VAR
BEGIN

REGION Network 1: ERROR
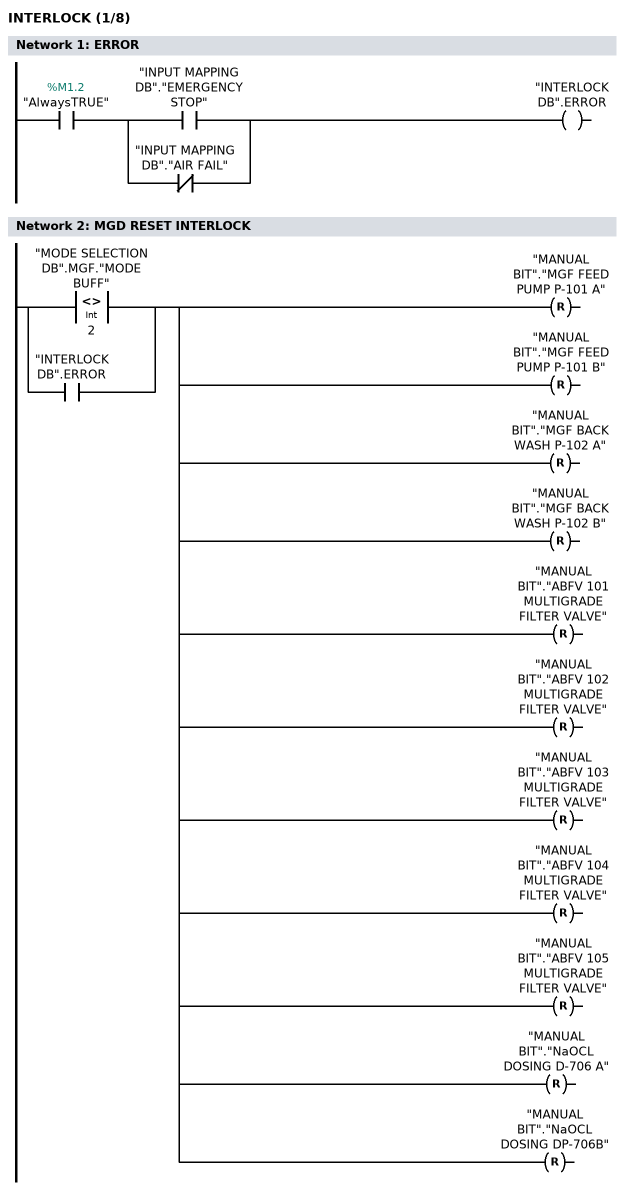
   RUNG wire#powerrail
      Contact( "AlwaysTRUE" )
      wire#w1
      Contact( "INPUT MAPPING DB"."EMERGENCY STOP" )
      wire#w2
      Coil( "INTERLOCK DB".ERROR )
   END_RUNG
   RUNG wire#w1
      I_Contact( "INPUT MAPPING DB"."AIR FAIL" )
   END_RUNG wire#w2
   // the same network as SCL:
   "INTERLOCK DB".ERROR := "AlwaysTRUE" AND ("INPUT MAPPING DB"."EMERGENCY STOP" OR NOT "INPUT MAPPING DB"."AIR FAIL");
END_REGION

REGION Network 2: MGD RESET INTERLOCK
   RUNG wire#powerrail
      { S7_Templates := "SrcType := Int" } NE_Contact(in1 := "MODE SELECTION DB".MGF."MODE BUFF", in2 := 2)
      wire#w1
      R_Coil( "MANUAL BIT"."MGF FEED PUMP P-101 A" )
   END_RUNG
   RUNG wire#powerrail
      Contact( "INTERLOCK DB".ERROR )
   END_RUNG wire#w1
   RUNG wire#w1
      R_Coil( "MANUAL BIT"."MGF FEED PUMP P-101 B" )
   END_RUNG
   RUNG wire#w1
      R_Coil( "MANUAL BIT"."MGF BACK WASH P-102 A" )
   END_RUNG
   RUNG wire#w1
      R_Coil( "MANUAL BIT"."MGF BACK WASH P-102 B" )
   END_RUNG
   RUNG wire#w1
      R_Coil( "MANUAL BIT"."ABFV 101 MULTIGRADE FILTER VALVE" )
   END_RUNG
   RUNG wire#w1
      R_Coil( "MANUAL BIT"."ABFV 102 MULTIGRADE FILTER VALVE" )
   END_RUNG
   RUNG wire#w1
      R_Coil( "MANUAL BIT"."ABFV 103 MULTIGRADE FILTER VALVE" )
   END_RUNG
   RUNG wire#w1
      R_Coil( "MANUAL BIT"."ABFV 104 MULTIGRADE FILTER VALVE" )
   END_RUNG
   RUNG wire#w1
      R_Coil( "MANUAL BIT"."ABFV 105 MULTIGRADE FILTER VALVE" )
   END_RUNG
   RUNG wire#w1
      R_Coil( "MANUAL BIT"."NaOCL DOSING D-706 A" )
   END_RUNG
   RUNG wire#w1
      R_Coil( "MANUAL BIT"."NaOCL DOSING DP-706B" )
   END_RUNG
   // the same network as SCL:
   IF ("MODE SELECTION DB".MGF."MODE BUFF" <> 2) OR "INTERLOCK DB".ERROR THEN
       "MANUAL BIT"."MGF FEED PUMP P-101 A" := FALSE;
       "MANUAL BIT"."MGF FEED PUMP P-101 B" := FALSE;
       "MANUAL BIT"."MGF BACK WASH P-102 A" := FALSE;
       "MANUAL BIT"."MGF BACK WASH P-102 B" := FALSE;
       "MANUAL BIT"."ABFV 101 MULTIGRADE FILTER VALVE" := FALSE;
       "MANUAL BIT"."ABFV 102 MULTIGRADE FILTER VALVE" := FALSE;
       "MANUAL BIT"."ABFV 103 MULTIGRADE FILTER VALVE" := FALSE;
       "MANUAL BIT"."ABFV 104 MULTIGRADE FILTER VALVE" := FALSE;
       "MANUAL BIT"."ABFV 105 MULTIGRADE FILTER VALVE" := FALSE;
       "MANUAL BIT"."NaOCL DOSING D-706 A" := FALSE;
       "MANUAL BIT"."NaOCL DOSING DP-706B" := FALSE;
   END_IF;
END_REGION

REGION Network 3: UF RESET INTERLOCK
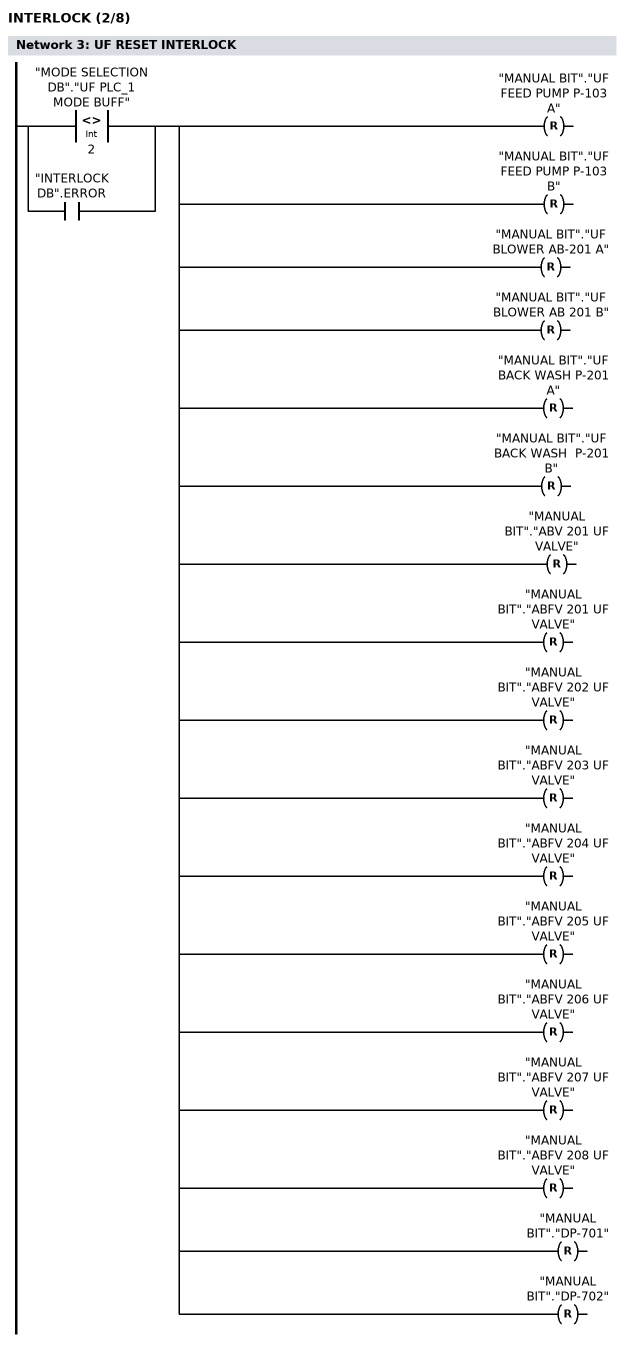
   RUNG wire#powerrail
      { S7_Templates := "SrcType := Int" } NE_Contact(in1 := "MODE SELECTION DB"."UF PLC_1 MODE BUFF", in2 := 2)
      wire#w1
      R_Coil( "MANUAL BIT"."UF FEED PUMP P-103 A" )
   END_RUNG
   RUNG wire#powerrail
      Contact( "INTERLOCK DB".ERROR )
   END_RUNG wire#w1
   RUNG wire#w1
      R_Coil( "MANUAL BIT"."UF FEED PUMP P-103 B" )
   END_RUNG
   RUNG wire#w1
      R_Coil( "MANUAL BIT"."UF BLOWER AB-201 A" )
   END_RUNG
   RUNG wire#w1
      R_Coil( "MANUAL BIT"."UF BLOWER AB 201 B" )
   END_RUNG
   RUNG wire#w1
      R_Coil( "MANUAL BIT"."UF BACK WASH P-201 A" )
   END_RUNG
   RUNG wire#w1
      R_Coil( "MANUAL BIT"."UF BACK WASH  P-201 B" )
   END_RUNG
   RUNG wire#w1
      R_Coil( "MANUAL BIT"."ABV 201 UF VALVE" )
   END_RUNG
   RUNG wire#w1
      R_Coil( "MANUAL BIT"."ABFV 201 UF VALVE" )
   END_RUNG
   RUNG wire#w1
      R_Coil( "MANUAL BIT"."ABFV 202 UF VALVE" )
   END_RUNG
   RUNG wire#w1
      R_Coil( "MANUAL BIT"."ABFV 203 UF VALVE" )
   END_RUNG
   RUNG wire#w1
      R_Coil( "MANUAL BIT"."ABFV 204 UF VALVE" )
   END_RUNG
   RUNG wire#w1
      R_Coil( "MANUAL BIT"."ABFV 205 UF VALVE" )
   END_RUNG
   RUNG wire#w1
      R_Coil( "MANUAL BIT"."ABFV 206 UF VALVE" )
   END_RUNG
   RUNG wire#w1
      R_Coil( "MANUAL BIT"."ABFV 207 UF VALVE" )
   END_RUNG
   RUNG wire#w1
      R_Coil( "MANUAL BIT"."ABFV 208 UF VALVE" )
   END_RUNG
   RUNG wire#w1
      R_Coil( "MANUAL BIT"."DP-701" )
   END_RUNG
   RUNG wire#w1
      R_Coil( "MANUAL BIT"."DP-702" )
   END_RUNG
   // the same network as SCL:
   IF ("MODE SELECTION DB"."UF PLC_1 MODE BUFF" <> 2) OR "INTERLOCK DB".ERROR THEN
       "MANUAL BIT"."UF FEED PUMP P-103 A" := FALSE;
       "MANUAL BIT"."UF FEED PUMP P-103 B" := FALSE;
       "MANUAL BIT"."UF BLOWER AB-201 A" := FALSE;
       "MANUAL BIT"."UF BLOWER AB 201 B" := FALSE;
       "MANUAL BIT"."UF BACK WASH P-201 A" := FALSE;
       "MANUAL BIT"."UF BACK WASH  P-201 B" := FALSE;
       "MANUAL BIT"."ABV 201 UF VALVE" := FALSE;
       "MANUAL BIT"."ABFV 201 UF VALVE" := FALSE;
       "MANUAL BIT"."ABFV 202 UF VALVE" := FALSE;
       "MANUAL BIT"."ABFV 203 UF VALVE" := FALSE;
       "MANUAL BIT"."ABFV 204 UF VALVE" := FALSE;
       "MANUAL BIT"."ABFV 205 UF VALVE" := FALSE;
       "MANUAL BIT"."ABFV 206 UF VALVE" := FALSE;
       "MANUAL BIT"."ABFV 207 UF VALVE" := FALSE;
       "MANUAL BIT"."ABFV 208 UF VALVE" := FALSE;
       "MANUAL BIT"."DP-701" := FALSE;
       "MANUAL BIT"."DP-702" := FALSE;
   END_IF;
END_REGION

REGION Network 4: DM RESET INTERLOCK
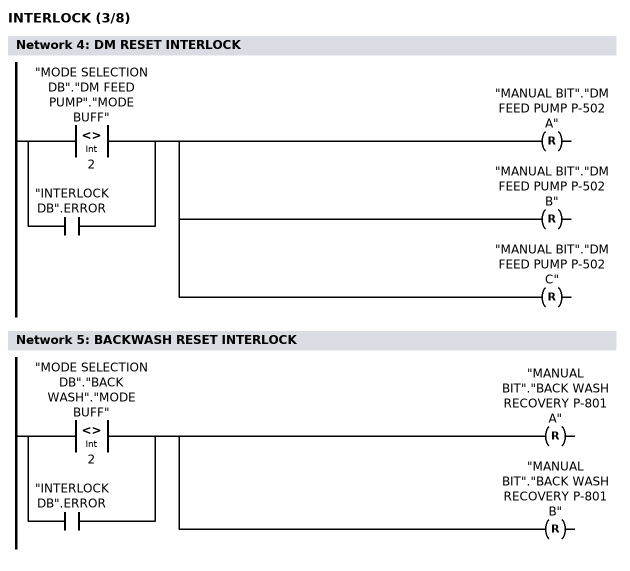
   RUNG wire#powerrail
      { S7_Templates := "SrcType := Int" } NE_Contact(in1 := "MODE SELECTION DB"."DM FEED PUMP"."MODE BUFF", in2 := 2)
      wire#w1
      R_Coil( "MANUAL BIT"."DM FEED PUMP P-502 A" )
   END_RUNG
   RUNG wire#powerrail
      Contact( "INTERLOCK DB".ERROR )
   END_RUNG wire#w1
   RUNG wire#w1
      R_Coil( "MANUAL BIT"."DM FEED PUMP P-502 B" )
   END_RUNG
   RUNG wire#w1
      R_Coil( "MANUAL BIT"."DM FEED PUMP P-502 C" )
   END_RUNG
   // the same network as SCL:
   IF ("MODE SELECTION DB"."DM FEED PUMP"."MODE BUFF" <> 2) OR "INTERLOCK DB".ERROR THEN
       "MANUAL BIT"."DM FEED PUMP P-502 A" := FALSE;
       "MANUAL BIT"."DM FEED PUMP P-502 B" := FALSE;
       "MANUAL BIT"."DM FEED PUMP P-502 C" := FALSE;
   END_IF;
END_REGION

REGION Network 5: BACKWASH RESET INTERLOCK
   RUNG wire#powerrail
      { S7_Templates := "SrcType := Int" } NE_Contact(in1 := "MODE SELECTION DB"."BACK WASH"."MODE BUFF", in2 := 2)
      wire#w1
      R_Coil( "MANUAL BIT"."BACK WASH RECOVERY P-801 A" )
   END_RUNG
   RUNG wire#powerrail
      Contact( "INTERLOCK DB".ERROR )
   END_RUNG wire#w1
   RUNG wire#w1
      R_Coil( "MANUAL BIT"."BACK WASH RECOVERY P-801 B" )
   END_RUNG
   // the same network as SCL:
   IF ("MODE SELECTION DB"."BACK WASH"."MODE BUFF" <> 2) OR "INTERLOCK DB".ERROR THEN
       "MANUAL BIT"."BACK WASH RECOVERY P-801 A" := FALSE;
       "MANUAL BIT"."BACK WASH RECOVERY P-801 B" := FALSE;
   END_IF;
END_REGION

REGION Network 6: SELECTION PUMP INTERLOCK_
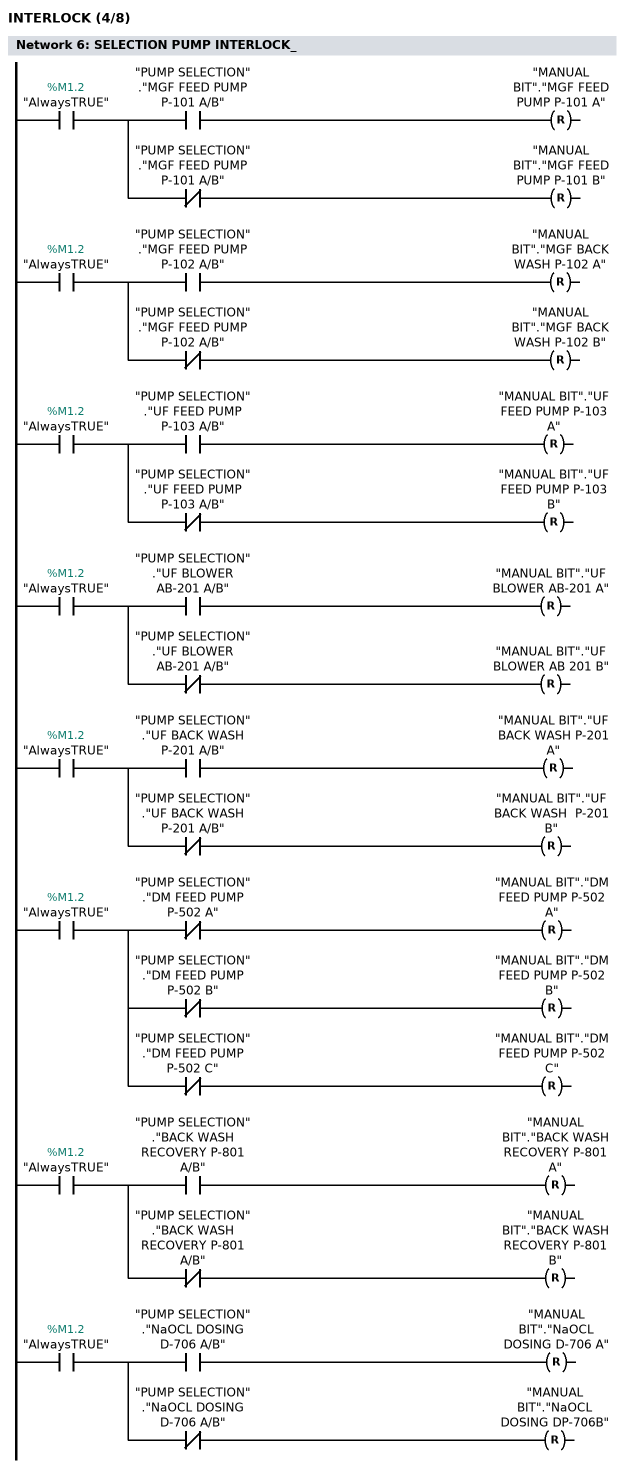
   RUNG wire#powerrail
      Contact( "AlwaysTRUE" )
      wire#w1
      Contact( "PUMP SELECTION"."MGF FEED PUMP P-101 A/B" )
      R_Coil( "MANUAL BIT"."MGF FEED PUMP P-101 A" )
   END_RUNG
   RUNG wire#w1
      I_Contact( "PUMP SELECTION"."MGF FEED PUMP P-101 A/B" )
      R_Coil( "MANUAL BIT"."MGF FEED PUMP P-101 B" )
   END_RUNG
   RUNG wire#powerrail
      Contact( "AlwaysTRUE" )
      wire#w2
      Contact( "PUMP SELECTION"."MGF FEED PUMP P-102 A/B" )
      R_Coil( "MANUAL BIT"."MGF BACK WASH P-102 A" )
   END_RUNG
   RUNG wire#w2
      I_Contact( "PUMP SELECTION"."MGF FEED PUMP P-102 A/B" )
      R_Coil( "MANUAL BIT"."MGF BACK WASH P-102 B" )
   END_RUNG
   RUNG wire#powerrail
      Contact( "AlwaysTRUE" )
      wire#w3
      Contact( "PUMP SELECTION"."UF FEED PUMP P-103 A/B" )
      R_Coil( "MANUAL BIT"."UF FEED PUMP P-103 A" )
   END_RUNG
   RUNG wire#w3
      I_Contact( "PUMP SELECTION"."UF FEED PUMP P-103 A/B" )
      R_Coil( "MANUAL BIT"."UF FEED PUMP P-103 B" )
   END_RUNG
   RUNG wire#powerrail
      Contact( "AlwaysTRUE" )
      wire#w4
      Contact( "PUMP SELECTION"."UF BLOWER AB-201 A/B" )
      R_Coil( "MANUAL BIT"."UF BLOWER AB-201 A" )
   END_RUNG
   RUNG wire#w4
      I_Contact( "PUMP SELECTION"."UF BLOWER AB-201 A/B" )
      R_Coil( "MANUAL BIT"."UF BLOWER AB 201 B" )
   END_RUNG
   RUNG wire#powerrail
      Contact( "AlwaysTRUE" )
      wire#w5
      Contact( "PUMP SELECTION"."UF BACK WASH P-201 A/B" )
      R_Coil( "MANUAL BIT"."UF BACK WASH P-201 A" )
   END_RUNG
   RUNG wire#w5
      I_Contact( "PUMP SELECTION"."UF BACK WASH P-201 A/B" )
      R_Coil( "MANUAL BIT"."UF BACK WASH  P-201 B" )
   END_RUNG
   RUNG wire#powerrail
      Contact( "AlwaysTRUE" )
      wire#w6
      I_Contact( "PUMP SELECTION"."DM FEED PUMP P-502 A" )
      R_Coil( "MANUAL BIT"."DM FEED PUMP P-502 A" )
   END_RUNG
   RUNG wire#w6
      I_Contact( "PUMP SELECTION"."DM FEED PUMP P-502 B" )
      R_Coil( "MANUAL BIT"."DM FEED PUMP P-502 B" )
   END_RUNG
   RUNG wire#w6
      I_Contact( "PUMP SELECTION"."DM FEED PUMP P-502 C" )
      R_Coil( "MANUAL BIT"."DM FEED PUMP P-502 C" )
   END_RUNG
   RUNG wire#powerrail
      Contact( "AlwaysTRUE" )
      wire#w7
      Contact( "PUMP SELECTION"."BACK WASH RECOVERY P-801 A/B" )
      R_Coil( "MANUAL BIT"."BACK WASH RECOVERY P-801 A" )
   END_RUNG
   RUNG wire#w7
      I_Contact( "PUMP SELECTION"."BACK WASH RECOVERY P-801 A/B" )
      R_Coil( "MANUAL BIT"."BACK WASH RECOVERY P-801 B" )
   END_RUNG
   RUNG wire#powerrail
      Contact( "AlwaysTRUE" )
      wire#w8
      Contact( "PUMP SELECTION"."NaOCL DOSING D-706 A/B" )
      R_Coil( "MANUAL BIT"."NaOCL DOSING D-706 A" )
   END_RUNG
   RUNG wire#w8
      I_Contact( "PUMP SELECTION"."NaOCL DOSING D-706 A/B" )
      R_Coil( "MANUAL BIT"."NaOCL DOSING DP-706B" )
   END_RUNG
   // the same network as SCL:
   IF "AlwaysTRUE" AND "PUMP SELECTION"."MGF FEED PUMP P-101 A/B" THEN
       "MANUAL BIT"."MGF FEED PUMP P-101 A" := FALSE;
   END_IF;
   IF "AlwaysTRUE" AND NOT "PUMP SELECTION"."MGF FEED PUMP P-101 A/B" THEN
       "MANUAL BIT"."MGF FEED PUMP P-101 B" := FALSE;
   END_IF;
   IF "AlwaysTRUE" AND "PUMP SELECTION"."MGF FEED PUMP P-102 A/B" THEN
       "MANUAL BIT"."MGF BACK WASH P-102 A" := FALSE;
   END_IF;
   IF "AlwaysTRUE" AND NOT "PUMP SELECTION"."MGF FEED PUMP P-102 A/B" THEN
       "MANUAL BIT"."MGF BACK WASH P-102 B" := FALSE;
   END_IF;
   IF "AlwaysTRUE" AND "PUMP SELECTION"."UF FEED PUMP P-103 A/B" THEN
       "MANUAL BIT"."UF FEED PUMP P-103 A" := FALSE;
   END_IF;
   IF "AlwaysTRUE" AND NOT "PUMP SELECTION"."UF FEED PUMP P-103 A/B" THEN
       "MANUAL BIT"."UF FEED PUMP P-103 B" := FALSE;
   END_IF;
   IF "AlwaysTRUE" AND "PUMP SELECTION"."UF BLOWER AB-201 A/B" THEN
       "MANUAL BIT"."UF BLOWER AB-201 A" := FALSE;
   END_IF;
   IF "AlwaysTRUE" AND NOT "PUMP SELECTION"."UF BLOWER AB-201 A/B" THEN
       "MANUAL BIT"."UF BLOWER AB 201 B" := FALSE;
   END_IF;
   IF "AlwaysTRUE" AND "PUMP SELECTION"."UF BACK WASH P-201 A/B" THEN
       "MANUAL BIT"."UF BACK WASH P-201 A" := FALSE;
   END_IF;
   IF "AlwaysTRUE" AND NOT "PUMP SELECTION"."UF BACK WASH P-201 A/B" THEN
       "MANUAL BIT"."UF BACK WASH  P-201 B" := FALSE;
   END_IF;
   IF "AlwaysTRUE" AND NOT "PUMP SELECTION"."DM FEED PUMP P-502 A" THEN
       "MANUAL BIT"."DM FEED PUMP P-502 A" := FALSE;
   END_IF;
   IF "AlwaysTRUE" AND NOT "PUMP SELECTION"."DM FEED PUMP P-502 B" THEN
       "MANUAL BIT"."DM FEED PUMP P-502 B" := FALSE;
   END_IF;
   IF "AlwaysTRUE" AND NOT "PUMP SELECTION"."DM FEED PUMP P-502 C" THEN
       "MANUAL BIT"."DM FEED PUMP P-502 C" := FALSE;
   END_IF;
   IF "AlwaysTRUE" AND "PUMP SELECTION"."BACK WASH RECOVERY P-801 A/B" THEN
       "MANUAL BIT"."BACK WASH RECOVERY P-801 A" := FALSE;
   END_IF;
   IF "AlwaysTRUE" AND NOT "PUMP SELECTION"."BACK WASH RECOVERY P-801 A/B" THEN
       "MANUAL BIT"."BACK WASH RECOVERY P-801 B" := FALSE;
   END_IF;
   IF "AlwaysTRUE" AND "PUMP SELECTION"."NaOCL DOSING D-706 A/B" THEN
       "MANUAL BIT"."NaOCL DOSING D-706 A" := FALSE;
   END_IF;
   IF "AlwaysTRUE" AND NOT "PUMP SELECTION"."NaOCL DOSING D-706 A/B" THEN
       "MANUAL BIT"."NaOCL DOSING DP-706B" := FALSE;
   END_IF;
END_REGION

REGION Network 9: AUTO__________________MGF PROCESS
END_REGION

REGION Network 10: PS-101.....................TAGE NHI MILA
END_REGION

REGION Network 11: PS201...........................
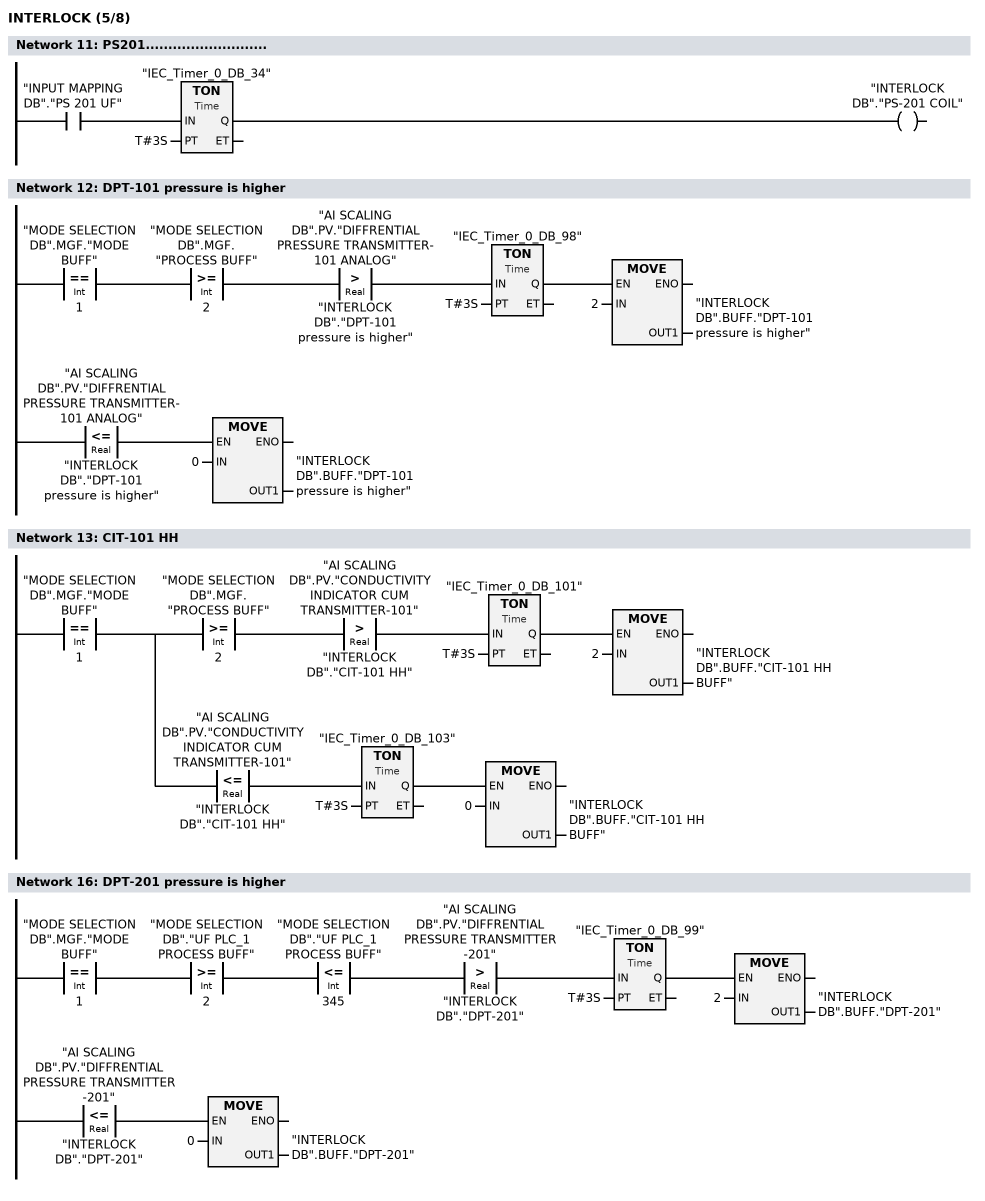
   RUNG wire#powerrail
      Contact( "INPUT MAPPING DB"."PS 201 UF" )
      { S7_Templates := "time_type := Time" } "IEC_Timer_0_DB_34".TON(pt := T#3S, et =>)
      Coil( "INTERLOCK DB"."PS-201 COIL" )
   END_RUNG
   // the same network as SCL:
   "IEC_Timer_0_DB_34".TON(IN := "INPUT MAPPING DB"."PS 201 UF", PT := T#3S);
   "INTERLOCK DB"."PS-201 COIL" := "IEC_Timer_0_DB_34".Q;
END_REGION

REGION Network 12: DPT-101 pressure is higher
   RUNG wire#powerrail
      { S7_Templates := "SrcType := Int" } EQ_Contact(in1 := "MODE SELECTION DB".MGF."MODE BUFF", in2 := 1)
      { S7_Templates := "SrcType := Int" } GE_Contact(in1 := "MODE SELECTION DB".MGF."PROCESS BUFF", in2 := 2)
      { S7_Templates := "SrcType := Real" } GT_Contact(in1 := "AI SCALING DB".PV."DIFFRENTIAL PRESSURE TRANSMITTER-101 ANALOG", in2 := "INTERLOCK DB"."DPT-101 pressure is higher")
      { S7_Templates := "time_type := Time" } "IEC_Timer_0_DB_98".TON(pt := T#3S, et =>)
      Move(in := 2, out1 => "INTERLOCK DB".BUFF."DPT-101 pressure is higher")
   END_RUNG
   RUNG wire#powerrail
      { S7_Templates := "SrcType := Real" } LE_Contact(in1 := "AI SCALING DB".PV."DIFFRENTIAL PRESSURE TRANSMITTER-101 ANALOG", in2 := "INTERLOCK DB"."DPT-101 pressure is higher")
      Move(in := 0, out1 => "INTERLOCK DB".BUFF."DPT-101 pressure is higher")
   END_RUNG
   // the same network as SCL:
   "IEC_Timer_0_DB_98".TON(IN := ("MODE SELECTION DB".MGF."MODE BUFF" = 1) AND ("MODE SELECTION DB".MGF."PROCESS BUFF" >= 2) AND ("AI SCALING DB".PV."DIFFRENTIAL PRESSURE TRANSMITTER-101 ANALOG" > "INTERLOCK DB"."DPT-101 pressure is higher"),
                           PT := T#3S);
   IF "IEC_Timer_0_DB_98".Q THEN "INTERLOCK DB".BUFF."DPT-101 pressure is higher" := 2; END_IF;
   IF "AI SCALING DB".PV."DIFFRENTIAL PRESSURE TRANSMITTER-101 ANALOG" <= "INTERLOCK DB"."DPT-101 pressure is higher" THEN
       "INTERLOCK DB".BUFF."DPT-101 pressure is higher" := 0;
   END_IF;
END_REGION

REGION Network 13: CIT-101 HH
   RUNG wire#powerrail
      { S7_Templates := "SrcType := Int" } EQ_Contact(in1 := "MODE SELECTION DB".MGF."MODE BUFF", in2 := 1)
      wire#w1
      { S7_Templates := "SrcType := Int" } GE_Contact(in1 := "MODE SELECTION DB".MGF."PROCESS BUFF", in2 := 2)
      { S7_Templates := "SrcType := Real" } GT_Contact(in1 := "AI SCALING DB".PV."CONDUCTIVITY INDICATOR CUM TRANSMITTER-101", in2 := "INTERLOCK DB"."CIT-101 HH")
      { S7_Templates := "time_type := Time" } "IEC_Timer_0_DB_101".TON(pt := T#3S, et =>)
      Move(in := 2, out1 => "INTERLOCK DB".BUFF."CIT-101 HH BUFF")
   END_RUNG
   RUNG wire#w1
      { S7_Templates := "SrcType := Real" } LE_Contact(in1 := "AI SCALING DB".PV."CONDUCTIVITY INDICATOR CUM TRANSMITTER-101", in2 := "INTERLOCK DB"."CIT-101 HH")
      { S7_Templates := "time_type := Time" } "IEC_Timer_0_DB_103".TON(pt := T#3S, et =>)
      Move(in := 0, out1 => "INTERLOCK DB".BUFF."CIT-101 HH BUFF")
   END_RUNG
   // the same network as SCL:
   #_w1 := "MODE SELECTION DB".MGF."MODE BUFF" = 1;
   "IEC_Timer_0_DB_101".TON(IN := #_w1 AND ("MODE SELECTION DB".MGF."PROCESS BUFF" >= 2) AND ("AI SCALING DB".PV."CONDUCTIVITY INDICATOR CUM TRANSMITTER-101" > "INTERLOCK DB"."CIT-101 HH"),
                           PT := T#3S);
   IF "IEC_Timer_0_DB_101".Q THEN "INTERLOCK DB".BUFF."CIT-101 HH BUFF" := 2; END_IF;
   "IEC_Timer_0_DB_103".TON(IN := #_w1 AND ("AI SCALING DB".PV."CONDUCTIVITY INDICATOR CUM TRANSMITTER-101" <= "INTERLOCK DB"."CIT-101 HH"),
                           PT := T#3S);
   IF "IEC_Timer_0_DB_103".Q THEN "INTERLOCK DB".BUFF."CIT-101 HH BUFF" := 0; END_IF;
END_REGION

REGION Network 15: AUTO__________________UF PROCESS
END_REGION

REGION Network 16: DPT-201 pressure is higher
   RUNG wire#powerrail
      { S7_Templates := "SrcType := Int" } EQ_Contact(in1 := "MODE SELECTION DB".MGF."MODE BUFF", in2 := 1)
      { S7_Templates := "SrcType := Int" } GE_Contact(in1 := "MODE SELECTION DB"."UF PLC_1 PROCESS BUFF", in2 := 2)
      { S7_Templates := "SrcType := Int" } LE_Contact(in1 := "MODE SELECTION DB"."UF PLC_1 PROCESS BUFF", in2 := 345)
      { S7_Templates := "SrcType := Real" } GT_Contact(in1 := "AI SCALING DB".PV."DIFFRENTIAL PRESSURE TRANSMITTER-201", in2 := "INTERLOCK DB"."DPT-201")
      { S7_Templates := "time_type := Time" } "IEC_Timer_0_DB_99".TON(pt := T#3S, et =>)
      Move(in := 2, out1 => "INTERLOCK DB".BUFF."DPT-201")
   END_RUNG
   RUNG wire#powerrail
      { S7_Templates := "SrcType := Real" } LE_Contact(in1 := "AI SCALING DB".PV."DIFFRENTIAL PRESSURE TRANSMITTER-201", in2 := "INTERLOCK DB"."DPT-201")
      Move(in := 0, out1 => "INTERLOCK DB".BUFF."DPT-201")
   END_RUNG
   // the same network as SCL:
   "IEC_Timer_0_DB_99".TON(IN := ("MODE SELECTION DB".MGF."MODE BUFF" = 1) AND ("MODE SELECTION DB"."UF PLC_1 PROCESS BUFF" >= 2) AND ("MODE SELECTION DB"."UF PLC_1 PROCESS BUFF" <= 345) AND ("AI SCALING DB".PV."DIFFRENTIAL PRESSURE TRANSMITTER-201" > "INTERLOCK DB"."DPT-201"),
                           PT := T#3S);
   IF "IEC_Timer_0_DB_99".Q THEN "INTERLOCK DB".BUFF."DPT-201" := 2; END_IF;
   IF "AI SCALING DB".PV."DIFFRENTIAL PRESSURE TRANSMITTER-201" <= "INTERLOCK DB"."DPT-201" THEN
       "INTERLOCK DB".BUFF."DPT-201" := 0;
   END_IF;
END_REGION

REGION Network 17: UF INTERLOCK FOR LT-102 AND LT201 SYSTER PAUSE
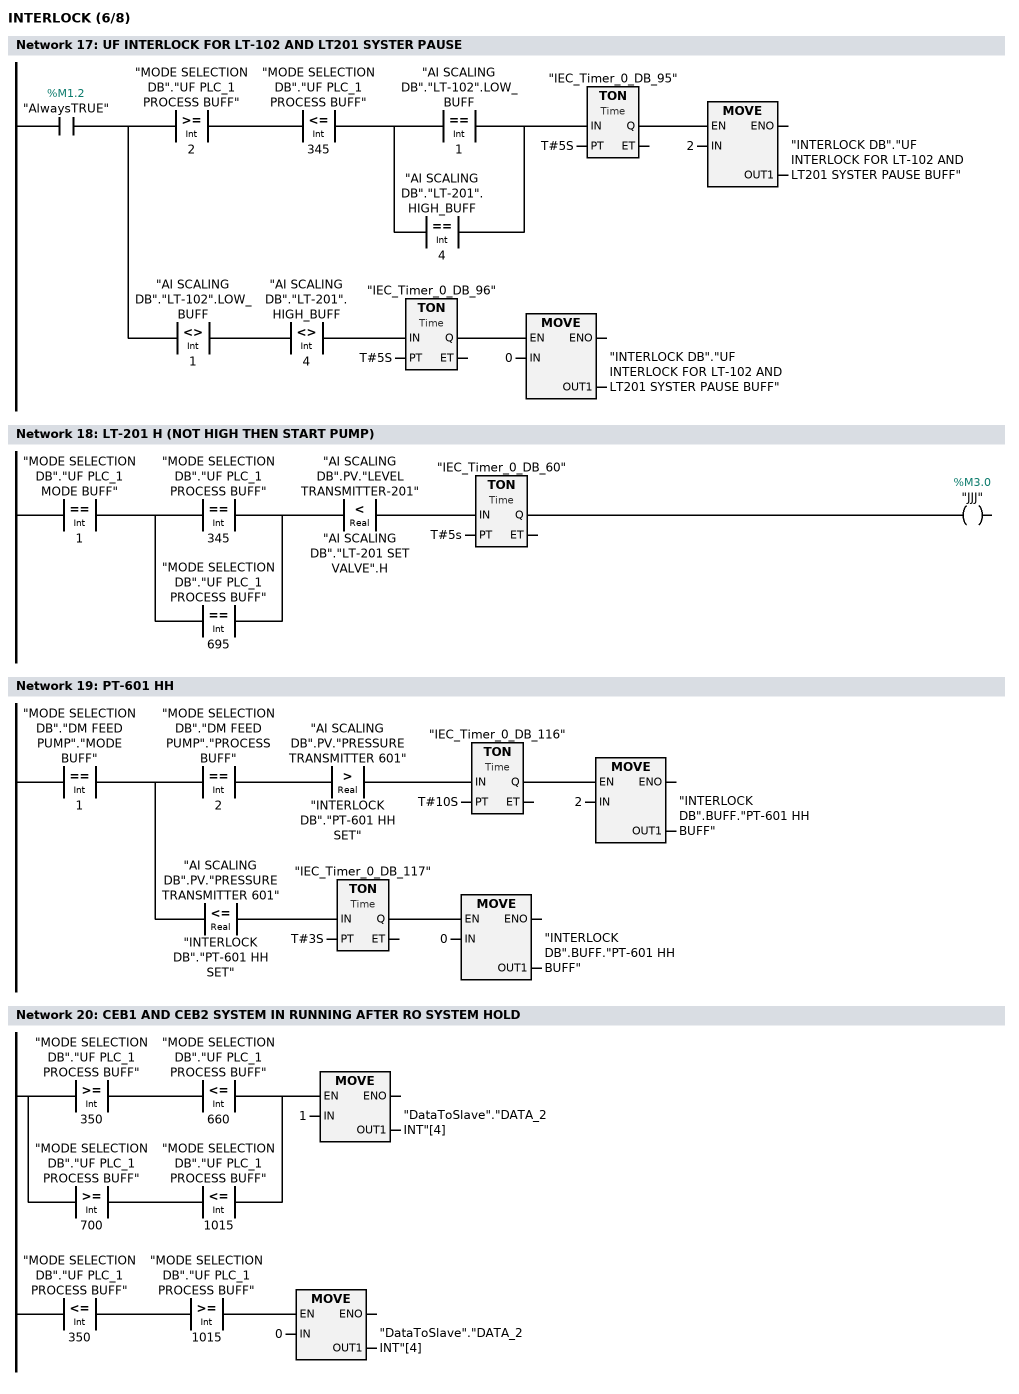
   RUNG wire#powerrail
      Contact( "AlwaysTRUE" )
      wire#w1
      { S7_Templates := "SrcType := Int" } GE_Contact(in1 := "MODE SELECTION DB"."UF PLC_1 PROCESS BUFF", in2 := 2)
      { S7_Templates := "SrcType := Int" } LE_Contact(in1 := "MODE SELECTION DB"."UF PLC_1 PROCESS BUFF", in2 := 345)
      wire#w2
      { S7_Templates := "SrcType := Int" } EQ_Contact(in1 := "AI SCALING DB"."LT-102".LOW_BUFF, in2 := 1)
      wire#w3
      { S7_Templates := "time_type := Time" } "IEC_Timer_0_DB_95".TON(pt := T#5S, et =>)
      Move(in := 2, out1 => "INTERLOCK DB"."UF INTERLOCK FOR LT-102 AND LT201 SYSTER PAUSE BUFF")
   END_RUNG
   RUNG wire#w2
      { S7_Templates := "SrcType := Int" } EQ_Contact(in1 := "AI SCALING DB"."LT-201".HIGH_BUFF, in2 := 4)
   END_RUNG wire#w3
   RUNG wire#w1
      { S7_Templates := "SrcType := Int" } NE_Contact(in1 := "AI SCALING DB"."LT-102".LOW_BUFF, in2 := 1)
      { S7_Templates := "SrcType := Int" } NE_Contact(in1 := "AI SCALING DB"."LT-201".HIGH_BUFF, in2 := 4)
      { S7_Templates := "time_type := Time" } "IEC_Timer_0_DB_96".TON(pt := T#5S, et =>)
      Move(in := 0, out1 => "INTERLOCK DB"."UF INTERLOCK FOR LT-102 AND LT201 SYSTER PAUSE BUFF")
   END_RUNG
   // the same network as SCL:
   "IEC_Timer_0_DB_95".TON(IN := "AlwaysTRUE" AND ("MODE SELECTION DB"."UF PLC_1 PROCESS BUFF" >= 2) AND ("MODE SELECTION DB"."UF PLC_1 PROCESS BUFF" <= 345) AND (("AI SCALING DB"."LT-102".LOW_BUFF = 1) OR ("AI SCALING DB"."LT-201".HIGH_BUFF = 4)),
                           PT := T#5S);
   IF "IEC_Timer_0_DB_95".Q THEN
       "INTERLOCK DB"."UF INTERLOCK FOR LT-102 AND LT201 SYSTER PAUSE BUFF" := 2;
   END_IF;
   "IEC_Timer_0_DB_96".TON(IN := "AlwaysTRUE" AND ("AI SCALING DB"."LT-102".LOW_BUFF <> 1) AND ("AI SCALING DB"."LT-201".HIGH_BUFF <> 4),
                           PT := T#5S);
   IF "IEC_Timer_0_DB_96".Q THEN
       "INTERLOCK DB"."UF INTERLOCK FOR LT-102 AND LT201 SYSTER PAUSE BUFF" := 0;
   END_IF;
END_REGION

REGION Network 18: LT-201 H (NOT HIGH THEN START PUMP)
   RUNG wire#powerrail
      { S7_Templates := "SrcType := Int" } EQ_Contact(in1 := "MODE SELECTION DB"."UF PLC_1 MODE BUFF", in2 := 1)
      wire#w1
      { S7_Templates := "SrcType := Int" } EQ_Contact(in1 := "MODE SELECTION DB"."UF PLC_1 PROCESS BUFF", in2 := 345)
      wire#w2
      { S7_Templates := "SrcType := Real" } LT_Contact(in1 := "AI SCALING DB".PV."LEVEL TRANSMITTER-201", in2 := "AI SCALING DB"."LT-201 SET VALVE".H)
      { S7_Templates := "time_type := Time" } "IEC_Timer_0_DB_60".TON(pt := T#5s, et =>)
      Coil( "JJJ" )
   END_RUNG
   RUNG wire#w1
      { S7_Templates := "SrcType := Int" } EQ_Contact(in1 := "MODE SELECTION DB"."UF PLC_1 PROCESS BUFF", in2 := 695)
   END_RUNG wire#w2
   // the same network as SCL:
   "IEC_Timer_0_DB_60".TON(IN := ("MODE SELECTION DB"."UF PLC_1 MODE BUFF" = 1) AND (("MODE SELECTION DB"."UF PLC_1 PROCESS BUFF" = 345) OR ("MODE SELECTION DB"."UF PLC_1 PROCESS BUFF" = 695)) AND ("AI SCALING DB".PV."LEVEL TRANSMITTER-201" < "AI SCALING DB"."LT-201 SET VALVE".H),
                           PT := T#5s);
   "JJJ" := "IEC_Timer_0_DB_60".Q;
END_REGION

REGION Network 19: PT-601 HH
   RUNG wire#powerrail
      { S7_Templates := "SrcType := Int" } EQ_Contact(in1 := "MODE SELECTION DB"."DM FEED PUMP"."MODE BUFF", in2 := 1)
      wire#w1
      { S7_Templates := "SrcType := Int" } EQ_Contact(in1 := "MODE SELECTION DB"."DM FEED PUMP"."PROCESS BUFF", in2 := 2)
      { S7_Templates := "SrcType := Real" } GT_Contact(in1 := "AI SCALING DB".PV."PRESSURE TRANSMITTER 601", in2 := "INTERLOCK DB"."PT-601 HH SET")
      { S7_Templates := "time_type := Time" } "IEC_Timer_0_DB_116".TON(pt := T#10S, et =>)
      Move(in := 2, out1 => "INTERLOCK DB".BUFF."PT-601 HH BUFF")
   END_RUNG
   RUNG wire#w1
      { S7_Templates := "SrcType := Real" } LE_Contact(in1 := "AI SCALING DB".PV."PRESSURE TRANSMITTER 601", in2 := "INTERLOCK DB"."PT-601 HH SET")
      { S7_Templates := "time_type := Time" } "IEC_Timer_0_DB_117".TON(pt := T#3S, et =>)
      Move(in := 0, out1 => "INTERLOCK DB".BUFF."PT-601 HH BUFF")
   END_RUNG
   // the same network as SCL:
   #_w1 := "MODE SELECTION DB"."DM FEED PUMP"."MODE BUFF" = 1;
   "IEC_Timer_0_DB_116".TON(IN := #_w1 AND ("MODE SELECTION DB"."DM FEED PUMP"."PROCESS BUFF" = 2) AND ("AI SCALING DB".PV."PRESSURE TRANSMITTER 601" > "INTERLOCK DB"."PT-601 HH SET"),
                           PT := T#10S);
   IF "IEC_Timer_0_DB_116".Q THEN "INTERLOCK DB".BUFF."PT-601 HH BUFF" := 2; END_IF;
   "IEC_Timer_0_DB_117".TON(IN := #_w1 AND ("AI SCALING DB".PV."PRESSURE TRANSMITTER 601" <= "INTERLOCK DB"."PT-601 HH SET"),
                           PT := T#3S);
   IF "IEC_Timer_0_DB_117".Q THEN "INTERLOCK DB".BUFF."PT-601 HH BUFF" := 0; END_IF;
END_REGION

REGION Network 20: CEB1 AND CEB2 SYSTEM IN RUNNING AFTER RO SYSTEM HOLD
   RUNG wire#powerrail
      { S7_Templates := "SrcType := Int" } GE_Contact(in1 := "MODE SELECTION DB"."UF PLC_1 PROCESS BUFF", in2 := 350)
      { S7_Templates := "SrcType := Int" } LE_Contact(in1 := "MODE SELECTION DB"."UF PLC_1 PROCESS BUFF", in2 := 660)
      wire#w1
      Move(in := 1, out1 => "DataToSlave"."DATA_2 INT"[4])
   END_RUNG
   RUNG wire#powerrail
      { S7_Templates := "SrcType := Int" } GE_Contact(in1 := "MODE SELECTION DB"."UF PLC_1 PROCESS BUFF", in2 := 700)
      { S7_Templates := "SrcType := Int" } LE_Contact(in1 := "MODE SELECTION DB"."UF PLC_1 PROCESS BUFF", in2 := 1015)
   END_RUNG wire#w1
   RUNG wire#powerrail
      { S7_Templates := "SrcType := Int" } LE_Contact(in1 := "MODE SELECTION DB"."UF PLC_1 PROCESS BUFF", in2 := 350)
      { S7_Templates := "SrcType := Int" } GE_Contact(in1 := "MODE SELECTION DB"."UF PLC_1 PROCESS BUFF", in2 := 1015)
      Move(in := 0, out1 => "DataToSlave"."DATA_2 INT"[4])
   END_RUNG
   // the same network as SCL:
   IF (("MODE SELECTION DB"."UF PLC_1 PROCESS BUFF" >= 350) AND ("MODE SELECTION DB"."UF PLC_1 PROCESS BUFF" <= 660)) OR (("MODE SELECTION DB"."UF PLC_1 PROCESS BUFF" >= 700) AND ("MODE SELECTION DB"."UF PLC_1 PROCESS BUFF" <= 1015)) THEN
       "DataToSlave"."DATA_2 INT"[4] := 1;
   END_IF;
   IF ("MODE SELECTION DB"."UF PLC_1 PROCESS BUFF" <= 350) AND ("MODE SELECTION DB"."UF PLC_1 PROCESS BUFF" >= 1015) THEN
       "DataToSlave"."DATA_2 INT"[4] := 0;
   END_IF;
END_REGION

REGION Network 22: AUTO__________________DM WATER TRANSFER
END_REGION

REGION Network 23: pHIT-601 LOW / HIGH
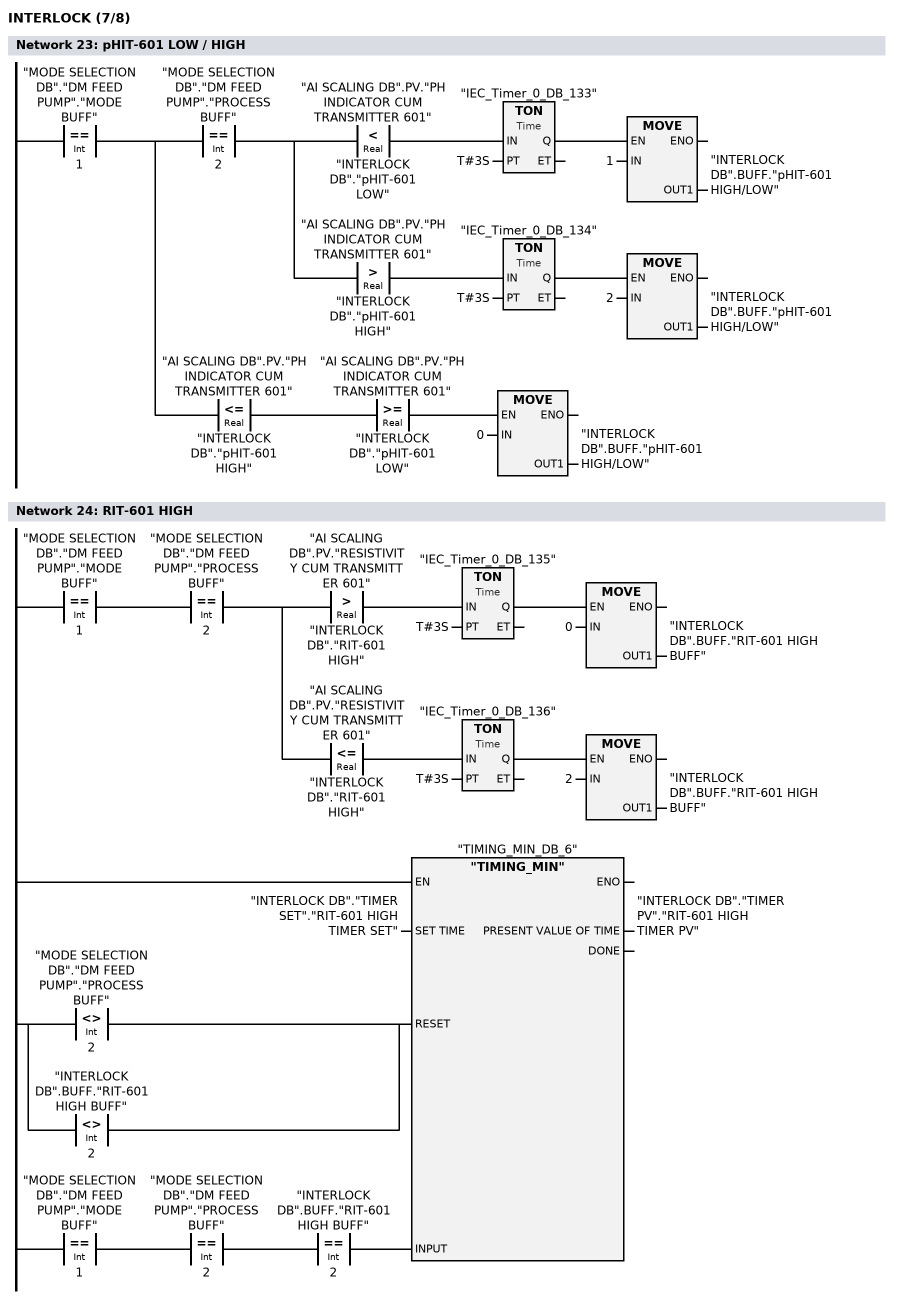
   RUNG wire#powerrail
      { S7_Templates := "SrcType := Int" } EQ_Contact(in1 := "MODE SELECTION DB"."DM FEED PUMP"."MODE BUFF", in2 := 1)
      wire#w1
      { S7_Templates := "SrcType := Int" } EQ_Contact(in1 := "MODE SELECTION DB"."DM FEED PUMP"."PROCESS BUFF", in2 := 2)
      wire#w2
      { S7_Templates := "SrcType := Real" } LT_Contact(in1 := "AI SCALING DB".PV."PH INDICATOR CUM TRANSMITTER 601", in2 := "INTERLOCK DB"."pHIT-601 LOW")
      { S7_Templates := "time_type := Time" } "IEC_Timer_0_DB_133".TON(pt := T#3S, et =>)
      Move(in := 1, out1 => "INTERLOCK DB".BUFF."pHIT-601 HIGH/LOW")
   END_RUNG
   RUNG wire#w2
      { S7_Templates := "SrcType := Real" } GT_Contact(in1 := "AI SCALING DB".PV."PH INDICATOR CUM TRANSMITTER 601", in2 := "INTERLOCK DB"."pHIT-601 HIGH")
      { S7_Templates := "time_type := Time" } "IEC_Timer_0_DB_134".TON(pt := T#3S, et =>)
      Move(in := 2, out1 => "INTERLOCK DB".BUFF."pHIT-601 HIGH/LOW")
   END_RUNG
   RUNG wire#w1
      { S7_Templates := "SrcType := Real" } LE_Contact(in1 := "AI SCALING DB".PV."PH INDICATOR CUM TRANSMITTER 601", in2 := "INTERLOCK DB"."pHIT-601 HIGH")
      { S7_Templates := "SrcType := Real" } GE_Contact(in1 := "AI SCALING DB".PV."PH INDICATOR CUM TRANSMITTER 601", in2 := "INTERLOCK DB"."pHIT-601 LOW")
      Move(in := 0, out1 => "INTERLOCK DB".BUFF."pHIT-601 HIGH/LOW")
   END_RUNG
   // the same network as SCL:
   #_w1 := "MODE SELECTION DB"."DM FEED PUMP"."MODE BUFF" = 1;
   #_w2 := #_w1 AND ("MODE SELECTION DB"."DM FEED PUMP"."PROCESS BUFF" = 2);
   "IEC_Timer_0_DB_133".TON(IN := #_w2 AND ("AI SCALING DB".PV."PH INDICATOR CUM TRANSMITTER 601" < "INTERLOCK DB"."pHIT-601 LOW"),
                           PT := T#3S);
   IF "IEC_Timer_0_DB_133".Q THEN "INTERLOCK DB".BUFF."pHIT-601 HIGH/LOW" := 1; END_IF;
   "IEC_Timer_0_DB_134".TON(IN := #_w2 AND ("AI SCALING DB".PV."PH INDICATOR CUM TRANSMITTER 601" > "INTERLOCK DB"."pHIT-601 HIGH"),
                           PT := T#3S);
   IF "IEC_Timer_0_DB_134".Q THEN "INTERLOCK DB".BUFF."pHIT-601 HIGH/LOW" := 2; END_IF;
   IF #_w1 AND ("AI SCALING DB".PV."PH INDICATOR CUM TRANSMITTER 601" <= "INTERLOCK DB"."pHIT-601 HIGH") AND ("AI SCALING DB".PV."PH INDICATOR CUM TRANSMITTER 601" >= "INTERLOCK DB"."pHIT-601 LOW") THEN
       "INTERLOCK DB".BUFF."pHIT-601 HIGH/LOW" := 0;
   END_IF;
END_REGION

REGION Network 24: RIT-601 HIGH
   RUNG wire#powerrail
      { S7_Templates := "SrcType := Int" } EQ_Contact(in1 := "MODE SELECTION DB"."DM FEED PUMP"."MODE BUFF", in2 := 1)
      { S7_Templates := "SrcType := Int" } EQ_Contact(in1 := "MODE SELECTION DB"."DM FEED PUMP"."PROCESS BUFF", in2 := 2)
      wire#w1
      { S7_Templates := "SrcType := Real" } GT_Contact(in1 := "AI SCALING DB".PV."RESISTIVITY CUM TRANSMITTER 601", in2 := "INTERLOCK DB"."RIT-601 HIGH")
      { S7_Templates := "time_type := Time" } "IEC_Timer_0_DB_135".TON(pt := T#3S, et =>)
      Move(in := 0, out1 => "INTERLOCK DB".BUFF."RIT-601 HIGH BUFF")
   END_RUNG
   RUNG wire#w1
      { S7_Templates := "SrcType := Real" } LE_Contact(in1 := "AI SCALING DB".PV."RESISTIVITY CUM TRANSMITTER 601", in2 := "INTERLOCK DB"."RIT-601 HIGH")
      { S7_Templates := "time_type := Time" } "IEC_Timer_0_DB_136".TON(pt := T#3S, et =>)
      Move(in := 2, out1 => "INTERLOCK DB".BUFF."RIT-601 HIGH BUFF")
   END_RUNG
   RUNG wire#powerrail
      "TIMING_MIN_DB_6"(RESET := wire#w2, INPUT := wire#w3, "SET TIME" := "INTERLOCK DB"."TIMER SET"."RIT-601 HIGH TIMER SET", "PRESENT VALUE OF TIME" => "INTERLOCK DB"."TIMER PV"."RIT-601 HIGH TIMER PV", DONE =>)
   END_RUNG
   RUNG wire#powerrail
      { S7_Templates := "SrcType := Int" } NE_Contact(in1 := "MODE SELECTION DB"."DM FEED PUMP"."PROCESS BUFF", in2 := 2)
   END_RUNG wire#w2
   RUNG wire#powerrail
      { S7_Templates := "SrcType := Int" } NE_Contact(in1 := "INTERLOCK DB".BUFF."RIT-601 HIGH BUFF", in2 := 2)
   END_RUNG wire#w2
   RUNG wire#powerrail
      { S7_Templates := "SrcType := Int" } EQ_Contact(in1 := "MODE SELECTION DB"."DM FEED PUMP"."MODE BUFF", in2 := 1)
      { S7_Templates := "SrcType := Int" } EQ_Contact(in1 := "MODE SELECTION DB"."DM FEED PUMP"."PROCESS BUFF", in2 := 2)
      { S7_Templates := "SrcType := Int" } EQ_Contact(in1 := "INTERLOCK DB".BUFF."RIT-601 HIGH BUFF", in2 := 2)
   END_RUNG wire#w3
   // the same network as SCL:
   #_w1 := ("MODE SELECTION DB"."DM FEED PUMP"."MODE BUFF" = 1) AND ("MODE SELECTION DB"."DM FEED PUMP"."PROCESS BUFF" = 2);
   "IEC_Timer_0_DB_135".TON(IN := #_w1 AND ("AI SCALING DB".PV."RESISTIVITY CUM TRANSMITTER 601" > "INTERLOCK DB"."RIT-601 HIGH"),
                           PT := T#3S);
   IF "IEC_Timer_0_DB_135".Q THEN "INTERLOCK DB".BUFF."RIT-601 HIGH BUFF" := 0; END_IF;
   "IEC_Timer_0_DB_136".TON(IN := #_w1 AND ("AI SCALING DB".PV."RESISTIVITY CUM TRANSMITTER 601" <= "INTERLOCK DB"."RIT-601 HIGH"),
                           PT := T#3S);
   IF "IEC_Timer_0_DB_136".Q THEN "INTERLOCK DB".BUFF."RIT-601 HIGH BUFF" := 2; END_IF;
   "TIMING_MIN_DB_6"("SET TIME" := "INTERLOCK DB"."TIMER SET"."RIT-601 HIGH TIMER SET",   // "TIMING_MIN"
                     RESET := ("MODE SELECTION DB"."DM FEED PUMP"."PROCESS BUFF" <> 2) OR ("INTERLOCK DB".BUFF."RIT-601 HIGH BUFF" <> 2),
                     INPUT := ("MODE SELECTION DB"."DM FEED PUMP"."MODE BUFF" = 1) AND ("MODE SELECTION DB"."DM FEED PUMP"."PROCESS BUFF" = 2) AND ("INTERLOCK DB".BUFF."RIT-601 HIGH BUFF" = 2),
                     "PRESENT VALUE OF TIME" => "INTERLOCK DB"."TIMER PV"."RIT-601 HIGH TIMER PV");
END_REGION

REGION Network 25: UV ONLY ALARM
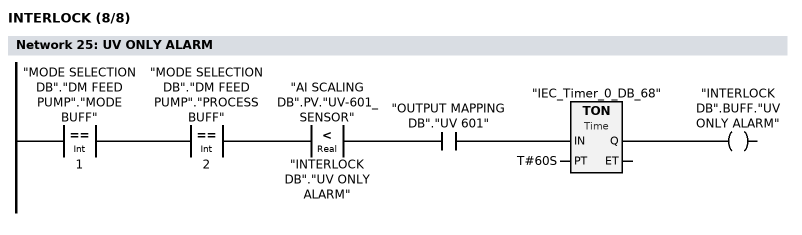
   RUNG wire#powerrail
      { S7_Templates := "SrcType := Int" } EQ_Contact(in1 := "MODE SELECTION DB"."DM FEED PUMP"."MODE BUFF", in2 := 1)
      { S7_Templates := "SrcType := Int" } EQ_Contact(in1 := "MODE SELECTION DB"."DM FEED PUMP"."PROCESS BUFF", in2 := 2)
      { S7_Templates := "SrcType := Real" } LT_Contact(in1 := "AI SCALING DB".PV."UV-601_SENSOR", in2 := "INTERLOCK DB"."UV ONLY ALARM")
      Contact( "OUTPUT MAPPING DB"."UV 601" )
      { S7_Templates := "time_type := Time" } "IEC_Timer_0_DB_68".TON(pt := T#60S, et =>)
      Coil( "INTERLOCK DB".BUFF."UV ONLY ALARM" )
   END_RUNG
   // the same network as SCL:
   "IEC_Timer_0_DB_68".TON(IN := ("MODE SELECTION DB"."DM FEED PUMP"."MODE BUFF" = 1) AND ("MODE SELECTION DB"."DM FEED PUMP"."PROCESS BUFF" = 2) AND ("AI SCALING DB".PV."UV-601_SENSOR" < "INTERLOCK DB"."UV ONLY ALARM") AND "OUTPUT MAPPING DB"."UV 601",
                           PT := T#60S);
   "INTERLOCK DB".BUFF."UV ONLY ALARM" := "IEC_Timer_0_DB_68".Q;
END_REGION
END_FUNCTION

FUNCTION_BLOCK "TIMING_MIN"   // FB4, LAD
{ S7_Optimized_Access := 'TRUE' }
// stored: MemoryReserve 100, SetENOAutomatically false
   VAR_INPUT
      "SET TIME" : Int;
      RESET : Bool;
      INPUT : Bool;
   END_VAR
   VAR_OUTPUT
      "PRESENT VALUE OF TIME" : Int;
      DONE : Bool;
   END_VAR
   VAR
      "TIMER 1" { S7_SetPoint := 'True'} : IEC_TIMER;
   END_VAR
   VAR RETAIN
      "COUNTER1 1" { S7_SetPoint := 'True'} : IEC_COUNTER;
   END_VAR
   VAR_TEMP   // added for the SCL form of the ladder/FBD networks
      _w1 : Bool;
      _w2 : Bool;
   END_VAR
BEGIN

REGION Network 1
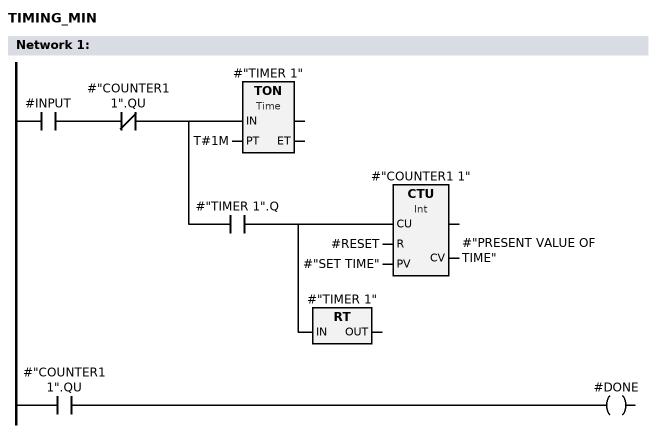
   RUNG wire#powerrail
      Contact( #INPUT )
      I_Contact( #"COUNTER1 1".QU )
      wire#w1
      { S7_Templates := "time_type := Time" } #"TIMER 1".TON(pt := T#1M, et =>)
   END_RUNG
   RUNG wire#w1
      Contact( #"TIMER 1".Q )
      wire#w2
      { S7_Templates := "value_type := Int" } #"COUNTER1 1".CTU(r := #RESET, pv := #"SET TIME", cv => #"PRESENT VALUE OF TIME")
   END_RUNG
   RUNG wire#w2
      RT_Coil( #"TIMER 1" )
   END_RUNG
   RUNG wire#powerrail
      Contact( #"COUNTER1 1".QU )
      Coil( #DONE )
   END_RUNG
   // the same network as SCL:
   #_w1 := #INPUT AND NOT #"COUNTER1 1".QU;
   #"TIMER 1".TON(IN := #_w1, PT := T#1M);
   #_w2 := #_w1 AND #"TIMER 1".Q;
   #"COUNTER1 1".CTU(CU := #_w2, R := #RESET, PV := #"SET TIME", CV => #"PRESENT VALUE OF TIME");
   IF #_w2 THEN RESET_TIMER(#"TIMER 1"); END_IF;
   #DONE := #"COUNTER1 1".QU;
END_REGION
END_FUNCTION_BLOCK

FUNCTION "DI WATER TRANSFER" : Void   // FC16, LAD
{ S7_Optimized_Access := 'TRUE' }
// stored: SetENOAutomatically false
BEGIN

REGION Network 1
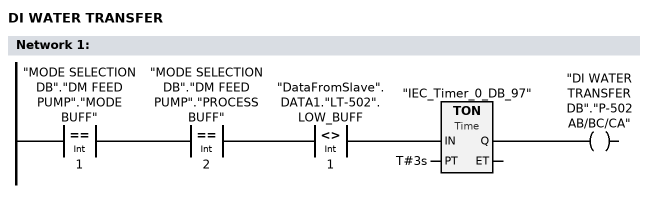
   RUNG wire#powerrail
      { S7_Templates := "SrcType := Int" } EQ_Contact(in1 := "MODE SELECTION DB"."DM FEED PUMP"."MODE BUFF", in2 := 1)
      { S7_Templates := "SrcType := Int" } EQ_Contact(in1 := "MODE SELECTION DB"."DM FEED PUMP"."PROCESS BUFF", in2 := 2)
      { S7_Templates := "SrcType := Int" } NE_Contact(in1 := "DataFromSlave".DATA1."LT-502".LOW_BUFF, in2 := 1)
      { S7_Templates := "time_type := Time" } "IEC_Timer_0_DB_97".TON(pt := T#3s, et =>)
      Coil( "DI WATER TRANSFER DB"."P-502 AB/BC/CA" )
   END_RUNG
   // the same network as SCL:
   "IEC_Timer_0_DB_97".TON(IN := ("MODE SELECTION DB"."DM FEED PUMP"."MODE BUFF" = 1) AND ("MODE SELECTION DB"."DM FEED PUMP"."PROCESS BUFF" = 2) AND ("DataFromSlave".DATA1."LT-502".LOW_BUFF <> 1),
                           PT := T#3s);
   "DI WATER TRANSFER DB"."P-502 AB/BC/CA" := "IEC_Timer_0_DB_97".Q;
END_REGION
END_FUNCTION

FUNCTION "AUTO_SUBOUTPUT" : Void   // FC11, LAD
{ S7_Optimized_Access := 'TRUE' }
// stored: SetENOAutomatically false
BEGIN

REGION Network 1: MGF FEED PUMP P-101 A
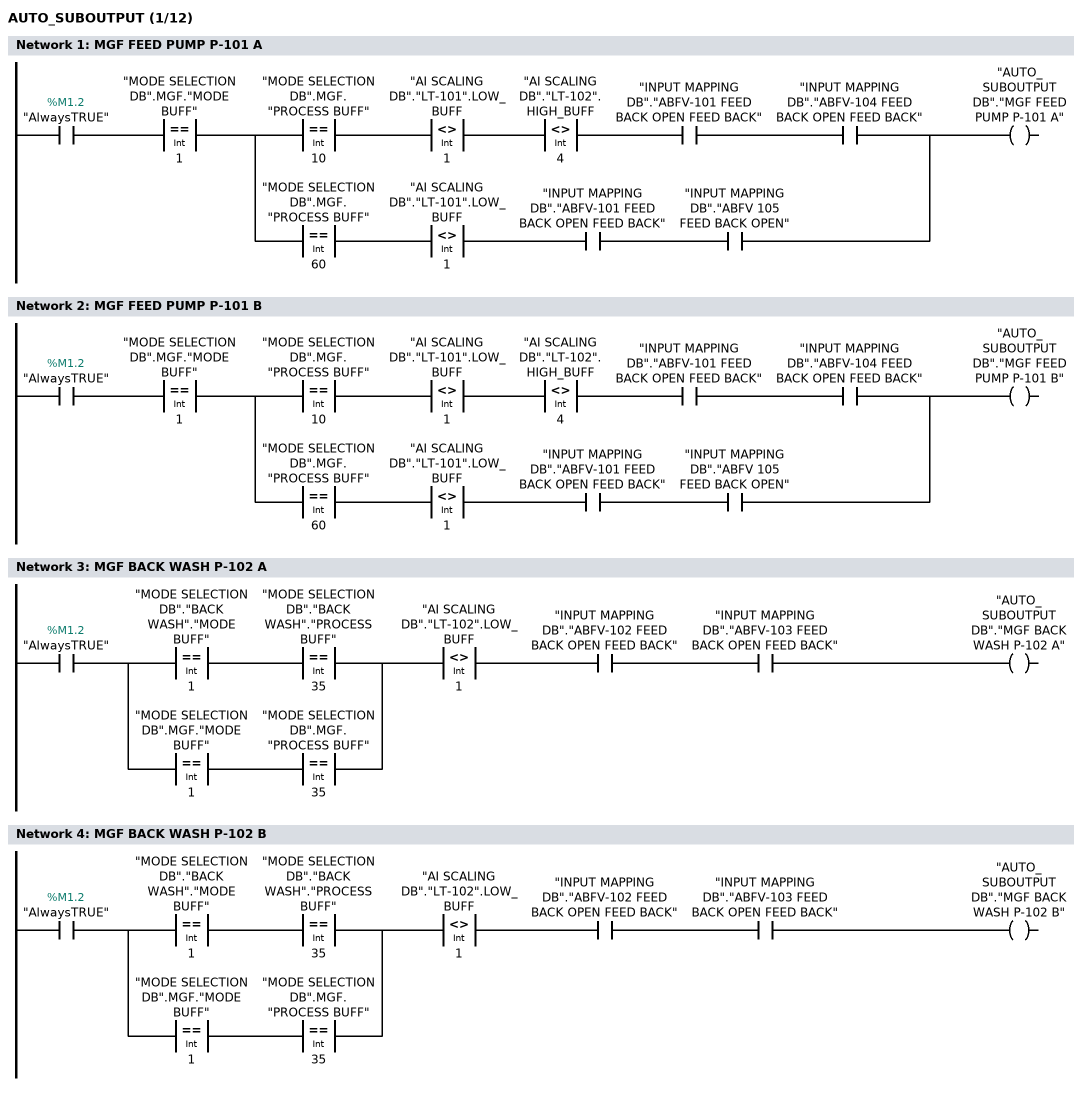
   RUNG wire#powerrail
      Contact( "AlwaysTRUE" )
      { S7_Templates := "SrcType := Int" } EQ_Contact(in1 := "MODE SELECTION DB".MGF."MODE BUFF", in2 := 1)
      wire#w1
      { S7_Templates := "SrcType := Int" } EQ_Contact(in1 := "MODE SELECTION DB".MGF."PROCESS BUFF", in2 := 10)
      { S7_Templates := "SrcType := Int" } NE_Contact(in1 := "AI SCALING DB"."LT-101".LOW_BUFF, in2 := 1)
      { S7_Templates := "SrcType := Int" } NE_Contact(in1 := "AI SCALING DB"."LT-102".HIGH_BUFF, in2 := 4)
      Contact( "INPUT MAPPING DB"."ABFV-101 FEED BACK OPEN FEED BACK" )
      Contact( "INPUT MAPPING DB"."ABFV-104 FEED BACK OPEN FEED BACK" )
      wire#w2
      Coil( "AUTO_SUBOUTPUT DB"."MGF FEED PUMP P-101 A" )
   END_RUNG
   RUNG wire#w1
      { S7_Templates := "SrcType := Int" } EQ_Contact(in1 := "MODE SELECTION DB".MGF."PROCESS BUFF", in2 := 60)
      { S7_Templates := "SrcType := Int" } NE_Contact(in1 := "AI SCALING DB"."LT-101".LOW_BUFF, in2 := 1)
      Contact( "INPUT MAPPING DB"."ABFV-101 FEED BACK OPEN FEED BACK" )
      Contact( "INPUT MAPPING DB"."ABFV 105 FEED BACK OPEN" )
   END_RUNG wire#w2
   // the same network as SCL:
   "AUTO_SUBOUTPUT DB"."MGF FEED PUMP P-101 A" := "AlwaysTRUE" AND ("MODE SELECTION DB".MGF."MODE BUFF" = 1) AND ((("MODE SELECTION DB".MGF."PROCESS BUFF" = 10) AND ("AI SCALING DB"."LT-101".LOW_BUFF <> 1) AND ("AI SCALING DB"."LT-102".HIGH_BUFF <> 4) AND "INPUT MAPPING DB"."ABFV-101 FEED BACK OPEN FEED BACK" AND "INPUT MAPPING DB"."ABFV-104 FEED BACK OPEN FEED BACK") OR (("MODE SELECTION DB".MGF."PROCESS BUFF" = 60) AND ("AI SCALING DB"."LT-101".LOW_BUFF <> 1) AND "INPUT MAPPING DB"."ABFV-101 FEED BACK OPEN FEED BACK" AND "INPUT MAPPING DB"."ABFV 105 FEED BACK OPEN"));
END_REGION

REGION Network 2: MGF FEED PUMP P-101 B
   RUNG wire#powerrail
      Contact( "AlwaysTRUE" )
      { S7_Templates := "SrcType := Int" } EQ_Contact(in1 := "MODE SELECTION DB".MGF."MODE BUFF", in2 := 1)
      wire#w1
      { S7_Templates := "SrcType := Int" } EQ_Contact(in1 := "MODE SELECTION DB".MGF."PROCESS BUFF", in2 := 10)
      { S7_Templates := "SrcType := Int" } NE_Contact(in1 := "AI SCALING DB"."LT-101".LOW_BUFF, in2 := 1)
      { S7_Templates := "SrcType := Int" } NE_Contact(in1 := "AI SCALING DB"."LT-102".HIGH_BUFF, in2 := 4)
      Contact( "INPUT MAPPING DB"."ABFV-101 FEED BACK OPEN FEED BACK" )
      Contact( "INPUT MAPPING DB"."ABFV-104 FEED BACK OPEN FEED BACK" )
      wire#w2
      Coil( "AUTO_SUBOUTPUT DB"."MGF FEED PUMP P-101 B" )
   END_RUNG
   RUNG wire#w1
      { S7_Templates := "SrcType := Int" } EQ_Contact(in1 := "MODE SELECTION DB".MGF."PROCESS BUFF", in2 := 60)
      { S7_Templates := "SrcType := Int" } NE_Contact(in1 := "AI SCALING DB"."LT-101".LOW_BUFF, in2 := 1)
      Contact( "INPUT MAPPING DB"."ABFV-101 FEED BACK OPEN FEED BACK" )
      Contact( "INPUT MAPPING DB"."ABFV 105 FEED BACK OPEN" )
   END_RUNG wire#w2
   // the same network as SCL:
   "AUTO_SUBOUTPUT DB"."MGF FEED PUMP P-101 B" := "AlwaysTRUE" AND ("MODE SELECTION DB".MGF."MODE BUFF" = 1) AND ((("MODE SELECTION DB".MGF."PROCESS BUFF" = 10) AND ("AI SCALING DB"."LT-101".LOW_BUFF <> 1) AND ("AI SCALING DB"."LT-102".HIGH_BUFF <> 4) AND "INPUT MAPPING DB"."ABFV-101 FEED BACK OPEN FEED BACK" AND "INPUT MAPPING DB"."ABFV-104 FEED BACK OPEN FEED BACK") OR (("MODE SELECTION DB".MGF."PROCESS BUFF" = 60) AND ("AI SCALING DB"."LT-101".LOW_BUFF <> 1) AND "INPUT MAPPING DB"."ABFV-101 FEED BACK OPEN FEED BACK" AND "INPUT MAPPING DB"."ABFV 105 FEED BACK OPEN"));
END_REGION

REGION Network 3: MGF BACK WASH P-102 A
   RUNG wire#powerrail
      Contact( "AlwaysTRUE" )
      wire#w1
      { S7_Templates := "SrcType := Int" } EQ_Contact(in1 := "MODE SELECTION DB"."BACK WASH"."MODE BUFF", in2 := 1)
      { S7_Templates := "SrcType := Int" } EQ_Contact(in1 := "MODE SELECTION DB"."BACK WASH"."PROCESS BUFF", in2 := 35)
      wire#w2
      { S7_Templates := "SrcType := Int" } NE_Contact(in1 := "AI SCALING DB"."LT-102".LOW_BUFF, in2 := 1)
      Contact( "INPUT MAPPING DB"."ABFV-102 FEED BACK OPEN FEED BACK" )
      Contact( "INPUT MAPPING DB"."ABFV-103 FEED BACK OPEN FEED BACK" )
      Coil( "AUTO_SUBOUTPUT DB"."MGF BACK WASH P-102 A" )
   END_RUNG
   RUNG wire#w1
      { S7_Templates := "SrcType := Int" } EQ_Contact(in1 := "MODE SELECTION DB".MGF."MODE BUFF", in2 := 1)
      { S7_Templates := "SrcType := Int" } EQ_Contact(in1 := "MODE SELECTION DB".MGF."PROCESS BUFF", in2 := 35)
   END_RUNG wire#w2
   // the same network as SCL:
   "AUTO_SUBOUTPUT DB"."MGF BACK WASH P-102 A" := "AlwaysTRUE" AND ((("MODE SELECTION DB"."BACK WASH"."MODE BUFF" = 1) AND ("MODE SELECTION DB"."BACK WASH"."PROCESS BUFF" = 35)) OR (("MODE SELECTION DB".MGF."MODE BUFF" = 1) AND ("MODE SELECTION DB".MGF."PROCESS BUFF" = 35))) AND ("AI SCALING DB"."LT-102".LOW_BUFF <> 1) AND "INPUT MAPPING DB"."ABFV-102 FEED BACK OPEN FEED BACK" AND "INPUT MAPPING DB"."ABFV-103 FEED BACK OPEN FEED BACK";
END_REGION

REGION Network 4: MGF BACK WASH P-102 B
   RUNG wire#powerrail
      Contact( "AlwaysTRUE" )
      wire#w1
      { S7_Templates := "SrcType := Int" } EQ_Contact(in1 := "MODE SELECTION DB"."BACK WASH"."MODE BUFF", in2 := 1)
      { S7_Templates := "SrcType := Int" } EQ_Contact(in1 := "MODE SELECTION DB"."BACK WASH"."PROCESS BUFF", in2 := 35)
      wire#w2
      { S7_Templates := "SrcType := Int" } NE_Contact(in1 := "AI SCALING DB"."LT-102".LOW_BUFF, in2 := 1)
      Contact( "INPUT MAPPING DB"."ABFV-102 FEED BACK OPEN FEED BACK" )
      Contact( "INPUT MAPPING DB"."ABFV-103 FEED BACK OPEN FEED BACK" )
      Coil( "AUTO_SUBOUTPUT DB"."MGF BACK WASH P-102 B" )
   END_RUNG
   RUNG wire#w1
      { S7_Templates := "SrcType := Int" } EQ_Contact(in1 := "MODE SELECTION DB".MGF."MODE BUFF", in2 := 1)
      { S7_Templates := "SrcType := Int" } EQ_Contact(in1 := "MODE SELECTION DB".MGF."PROCESS BUFF", in2 := 35)
   END_RUNG wire#w2
   // the same network as SCL:
   "AUTO_SUBOUTPUT DB"."MGF BACK WASH P-102 B" := "AlwaysTRUE" AND ((("MODE SELECTION DB"."BACK WASH"."MODE BUFF" = 1) AND ("MODE SELECTION DB"."BACK WASH"."PROCESS BUFF" = 35)) OR (("MODE SELECTION DB".MGF."MODE BUFF" = 1) AND ("MODE SELECTION DB".MGF."PROCESS BUFF" = 35))) AND ("AI SCALING DB"."LT-102".LOW_BUFF <> 1) AND "INPUT MAPPING DB"."ABFV-102 FEED BACK OPEN FEED BACK" AND "INPUT MAPPING DB"."ABFV-103 FEED BACK OPEN FEED BACK";
END_REGION

REGION Network 5: UF FEED PUMP P-103 A
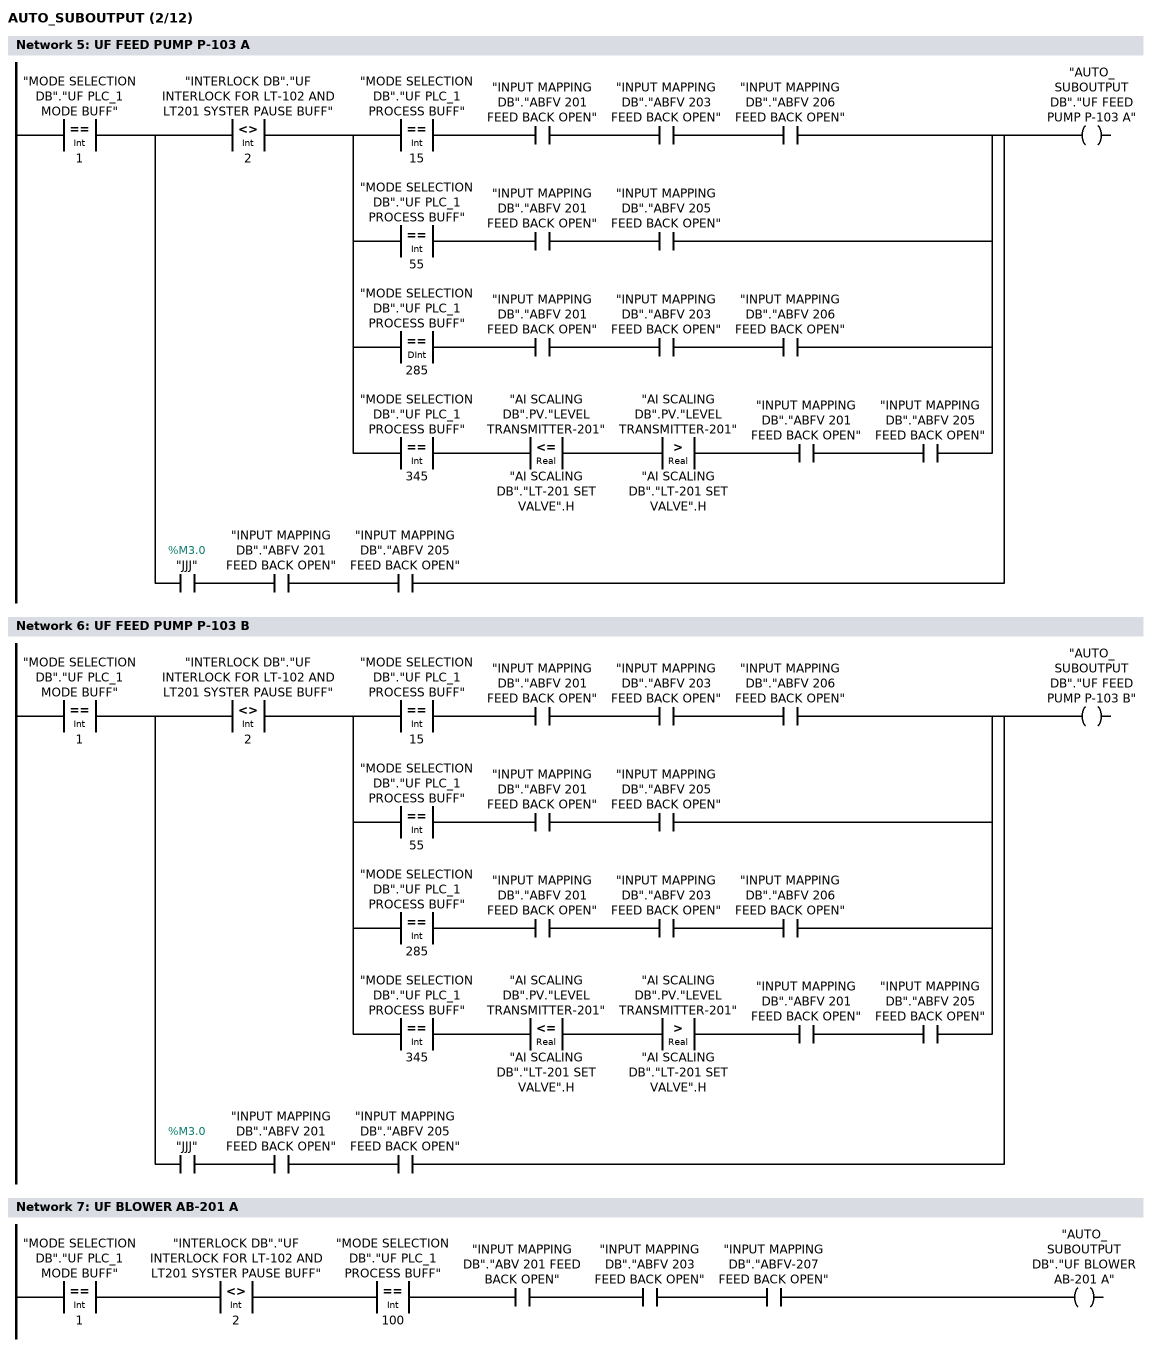
   RUNG wire#powerrail
      { S7_Templates := "SrcType := Int" } EQ_Contact(in1 := "MODE SELECTION DB"."UF PLC_1 MODE BUFF", in2 := 1)
      wire#w1
      { S7_Templates := "SrcType := Int" } NE_Contact(in1 := "INTERLOCK DB"."UF INTERLOCK FOR LT-102 AND LT201 SYSTER PAUSE BUFF", in2 := 2)
      wire#w2
      { S7_Templates := "SrcType := Int" } EQ_Contact(in1 := "MODE SELECTION DB"."UF PLC_1 PROCESS BUFF", in2 := 15)
      Contact( "INPUT MAPPING DB"."ABFV 201 FEED BACK OPEN" )
      Contact( "INPUT MAPPING DB"."ABFV 203 FEED BACK OPEN" )
      Contact( "INPUT MAPPING DB"."ABFV 206 FEED BACK OPEN" )
      wire#w3
      Coil( "AUTO_SUBOUTPUT DB"."UF FEED PUMP P-103 A" )
   END_RUNG
   RUNG wire#w2
      { S7_Templates := "SrcType := Int" } EQ_Contact(in1 := "MODE SELECTION DB"."UF PLC_1 PROCESS BUFF", in2 := 55)
      Contact( "INPUT MAPPING DB"."ABFV 201 FEED BACK OPEN" )
      Contact( "INPUT MAPPING DB"."ABFV 205 FEED BACK OPEN" )
   END_RUNG wire#w3
   RUNG wire#w2
      { S7_Templates := "SrcType := DInt" } EQ_Contact(in1 := "MODE SELECTION DB"."UF PLC_1 PROCESS BUFF", in2 := 285)
      Contact( "INPUT MAPPING DB"."ABFV 201 FEED BACK OPEN" )
      Contact( "INPUT MAPPING DB"."ABFV 203 FEED BACK OPEN" )
      Contact( "INPUT MAPPING DB"."ABFV 206 FEED BACK OPEN" )
   END_RUNG wire#w3
   RUNG wire#w2
      { S7_Templates := "SrcType := Int" } EQ_Contact(in1 := "MODE SELECTION DB"."UF PLC_1 PROCESS BUFF", in2 := 345)
      { S7_Templates := "SrcType := Real" } LE_Contact(in1 := "AI SCALING DB".PV."LEVEL TRANSMITTER-201", in2 := "AI SCALING DB"."LT-201 SET VALVE".H)
      { S7_Templates := "SrcType := Real" } GT_Contact(in1 := "AI SCALING DB".PV."LEVEL TRANSMITTER-201", in2 := "AI SCALING DB"."LT-201 SET VALVE".H)
      Contact( "INPUT MAPPING DB"."ABFV 201 FEED BACK OPEN" )
      Contact( "INPUT MAPPING DB"."ABFV 205 FEED BACK OPEN" )
   END_RUNG wire#w3
   RUNG wire#w1
      Contact( "JJJ" )
      Contact( "INPUT MAPPING DB"."ABFV 201 FEED BACK OPEN" )
      Contact( "INPUT MAPPING DB"."ABFV 205 FEED BACK OPEN" )
   END_RUNG wire#w3
   // the same network as SCL:
   "AUTO_SUBOUTPUT DB"."UF FEED PUMP P-103 A" := ("MODE SELECTION DB"."UF PLC_1 MODE BUFF" = 1) AND ((("INTERLOCK DB"."UF INTERLOCK FOR LT-102 AND LT201 SYSTER PAUSE BUFF" <> 2) AND ((("MODE SELECTION DB"."UF PLC_1 PROCESS BUFF" = 15) AND "INPUT MAPPING DB"."ABFV 201 FEED BACK OPEN" AND "INPUT MAPPING DB"."ABFV 203 FEED BACK OPEN" AND "INPUT MAPPING DB"."ABFV 206 FEED BACK OPEN") OR (("MODE SELECTION DB"."UF PLC_1 PROCESS BUFF" = 55) AND "INPUT MAPPING DB"."ABFV 201 FEED BACK OPEN" AND "INPUT MAPPING DB"."ABFV 205 FEED BACK OPEN") OR (("MODE SELECTION DB"."UF PLC_1 PROCESS BUFF" = 285) AND "INPUT MAPPING DB"."ABFV 201 FEED BACK OPEN" AND "INPUT MAPPING DB"."ABFV 203 FEED BACK OPEN" AND "INPUT MAPPING DB"."ABFV 206 FEED BACK OPEN") OR (("MODE SELECTION DB"."UF PLC_1 PROCESS BUFF" = 345) AND ("AI SCALING DB".PV."LEVEL TRANSMITTER-201" <= "AI SCALING DB"."LT-201 SET VALVE".H) AND ("AI SCALING DB".PV."LEVEL TRANSMITTER-201" > "AI SCALING DB"."LT-201 SET VALVE".H) AND "INPUT MAPPING DB"."ABFV 201 FEED BACK OPEN" AND "INPUT MAPPING DB"."ABFV 205 FEED BACK OPEN"))) OR ("JJJ" AND "INPUT MAPPING DB"."ABFV 201 FEED BACK OPEN" AND "INPUT MAPPING DB"."ABFV 205 FEED BACK OPEN"));
END_REGION

REGION Network 6: UF FEED PUMP P-103 B
   RUNG wire#powerrail
      { S7_Templates := "SrcType := Int" } EQ_Contact(in1 := "MODE SELECTION DB"."UF PLC_1 MODE BUFF", in2 := 1)
      wire#w1
      { S7_Templates := "SrcType := Int" } NE_Contact(in1 := "INTERLOCK DB"."UF INTERLOCK FOR LT-102 AND LT201 SYSTER PAUSE BUFF", in2 := 2)
      wire#w2
      { S7_Templates := "SrcType := Int" } EQ_Contact(in1 := "MODE SELECTION DB"."UF PLC_1 PROCESS BUFF", in2 := 15)
      Contact( "INPUT MAPPING DB"."ABFV 201 FEED BACK OPEN" )
      Contact( "INPUT MAPPING DB"."ABFV 203 FEED BACK OPEN" )
      Contact( "INPUT MAPPING DB"."ABFV 206 FEED BACK OPEN" )
      wire#w3
      Coil( "AUTO_SUBOUTPUT DB"."UF FEED PUMP P-103 B" )
   END_RUNG
   RUNG wire#w2
      { S7_Templates := "SrcType := Int" } EQ_Contact(in1 := "MODE SELECTION DB"."UF PLC_1 PROCESS BUFF", in2 := 55)
      Contact( "INPUT MAPPING DB"."ABFV 201 FEED BACK OPEN" )
      Contact( "INPUT MAPPING DB"."ABFV 205 FEED BACK OPEN" )
   END_RUNG wire#w3
   RUNG wire#w2
      { S7_Templates := "SrcType := Int" } EQ_Contact(in1 := "MODE SELECTION DB"."UF PLC_1 PROCESS BUFF", in2 := 285)
      Contact( "INPUT MAPPING DB"."ABFV 201 FEED BACK OPEN" )
      Contact( "INPUT MAPPING DB"."ABFV 203 FEED BACK OPEN" )
      Contact( "INPUT MAPPING DB"."ABFV 206 FEED BACK OPEN" )
   END_RUNG wire#w3
   RUNG wire#w2
      { S7_Templates := "SrcType := Int" } EQ_Contact(in1 := "MODE SELECTION DB"."UF PLC_1 PROCESS BUFF", in2 := 345)
      { S7_Templates := "SrcType := Real" } LE_Contact(in1 := "AI SCALING DB".PV."LEVEL TRANSMITTER-201", in2 := "AI SCALING DB"."LT-201 SET VALVE".H)
      { S7_Templates := "SrcType := Real" } GT_Contact(in1 := "AI SCALING DB".PV."LEVEL TRANSMITTER-201", in2 := "AI SCALING DB"."LT-201 SET VALVE".H)
      Contact( "INPUT MAPPING DB"."ABFV 201 FEED BACK OPEN" )
      Contact( "INPUT MAPPING DB"."ABFV 205 FEED BACK OPEN" )
   END_RUNG wire#w3
   RUNG wire#w1
      Contact( "JJJ" )
      Contact( "INPUT MAPPING DB"."ABFV 201 FEED BACK OPEN" )
      Contact( "INPUT MAPPING DB"."ABFV 205 FEED BACK OPEN" )
   END_RUNG wire#w3
   // the same network as SCL:
   "AUTO_SUBOUTPUT DB"."UF FEED PUMP P-103 B" := ("MODE SELECTION DB"."UF PLC_1 MODE BUFF" = 1) AND ((("INTERLOCK DB"."UF INTERLOCK FOR LT-102 AND LT201 SYSTER PAUSE BUFF" <> 2) AND ((("MODE SELECTION DB"."UF PLC_1 PROCESS BUFF" = 15) AND "INPUT MAPPING DB"."ABFV 201 FEED BACK OPEN" AND "INPUT MAPPING DB"."ABFV 203 FEED BACK OPEN" AND "INPUT MAPPING DB"."ABFV 206 FEED BACK OPEN") OR (("MODE SELECTION DB"."UF PLC_1 PROCESS BUFF" = 55) AND "INPUT MAPPING DB"."ABFV 201 FEED BACK OPEN" AND "INPUT MAPPING DB"."ABFV 205 FEED BACK OPEN") OR (("MODE SELECTION DB"."UF PLC_1 PROCESS BUFF" = 285) AND "INPUT MAPPING DB"."ABFV 201 FEED BACK OPEN" AND "INPUT MAPPING DB"."ABFV 203 FEED BACK OPEN" AND "INPUT MAPPING DB"."ABFV 206 FEED BACK OPEN") OR (("MODE SELECTION DB"."UF PLC_1 PROCESS BUFF" = 345) AND ("AI SCALING DB".PV."LEVEL TRANSMITTER-201" <= "AI SCALING DB"."LT-201 SET VALVE".H) AND ("AI SCALING DB".PV."LEVEL TRANSMITTER-201" > "AI SCALING DB"."LT-201 SET VALVE".H) AND "INPUT MAPPING DB"."ABFV 201 FEED BACK OPEN" AND "INPUT MAPPING DB"."ABFV 205 FEED BACK OPEN"))) OR ("JJJ" AND "INPUT MAPPING DB"."ABFV 201 FEED BACK OPEN" AND "INPUT MAPPING DB"."ABFV 205 FEED BACK OPEN"));
END_REGION

REGION Network 7: UF BLOWER AB-201 A
   RUNG wire#powerrail
      { S7_Templates := "SrcType := Int" } EQ_Contact(in1 := "MODE SELECTION DB"."UF PLC_1 MODE BUFF", in2 := 1)
      { S7_Templates := "SrcType := Int" } NE_Contact(in1 := "INTERLOCK DB"."UF INTERLOCK FOR LT-102 AND LT201 SYSTER PAUSE BUFF", in2 := 2)
      { S7_Templates := "SrcType := Int" } EQ_Contact(in1 := "MODE SELECTION DB"."UF PLC_1 PROCESS BUFF", in2 := 100)
      Contact( "INPUT MAPPING DB"."ABV 201 FEED BACK OPEN" )
      Contact( "INPUT MAPPING DB"."ABFV 203 FEED BACK OPEN" )
      Contact( "INPUT MAPPING DB"."ABFV-207 FEED BACK OPEN" )
      Coil( "AUTO_SUBOUTPUT DB"."UF BLOWER AB-201 A" )
   END_RUNG
   // the same network as SCL:
   "AUTO_SUBOUTPUT DB"."UF BLOWER AB-201 A" := ("MODE SELECTION DB"."UF PLC_1 MODE BUFF" = 1) AND ("INTERLOCK DB"."UF INTERLOCK FOR LT-102 AND LT201 SYSTER PAUSE BUFF" <> 2) AND ("MODE SELECTION DB"."UF PLC_1 PROCESS BUFF" = 100) AND "INPUT MAPPING DB"."ABV 201 FEED BACK OPEN" AND "INPUT MAPPING DB"."ABFV 203 FEED BACK OPEN" AND "INPUT MAPPING DB"."ABFV-207 FEED BACK OPEN";
END_REGION

REGION Network 8: UF BLOWER AB 201 B
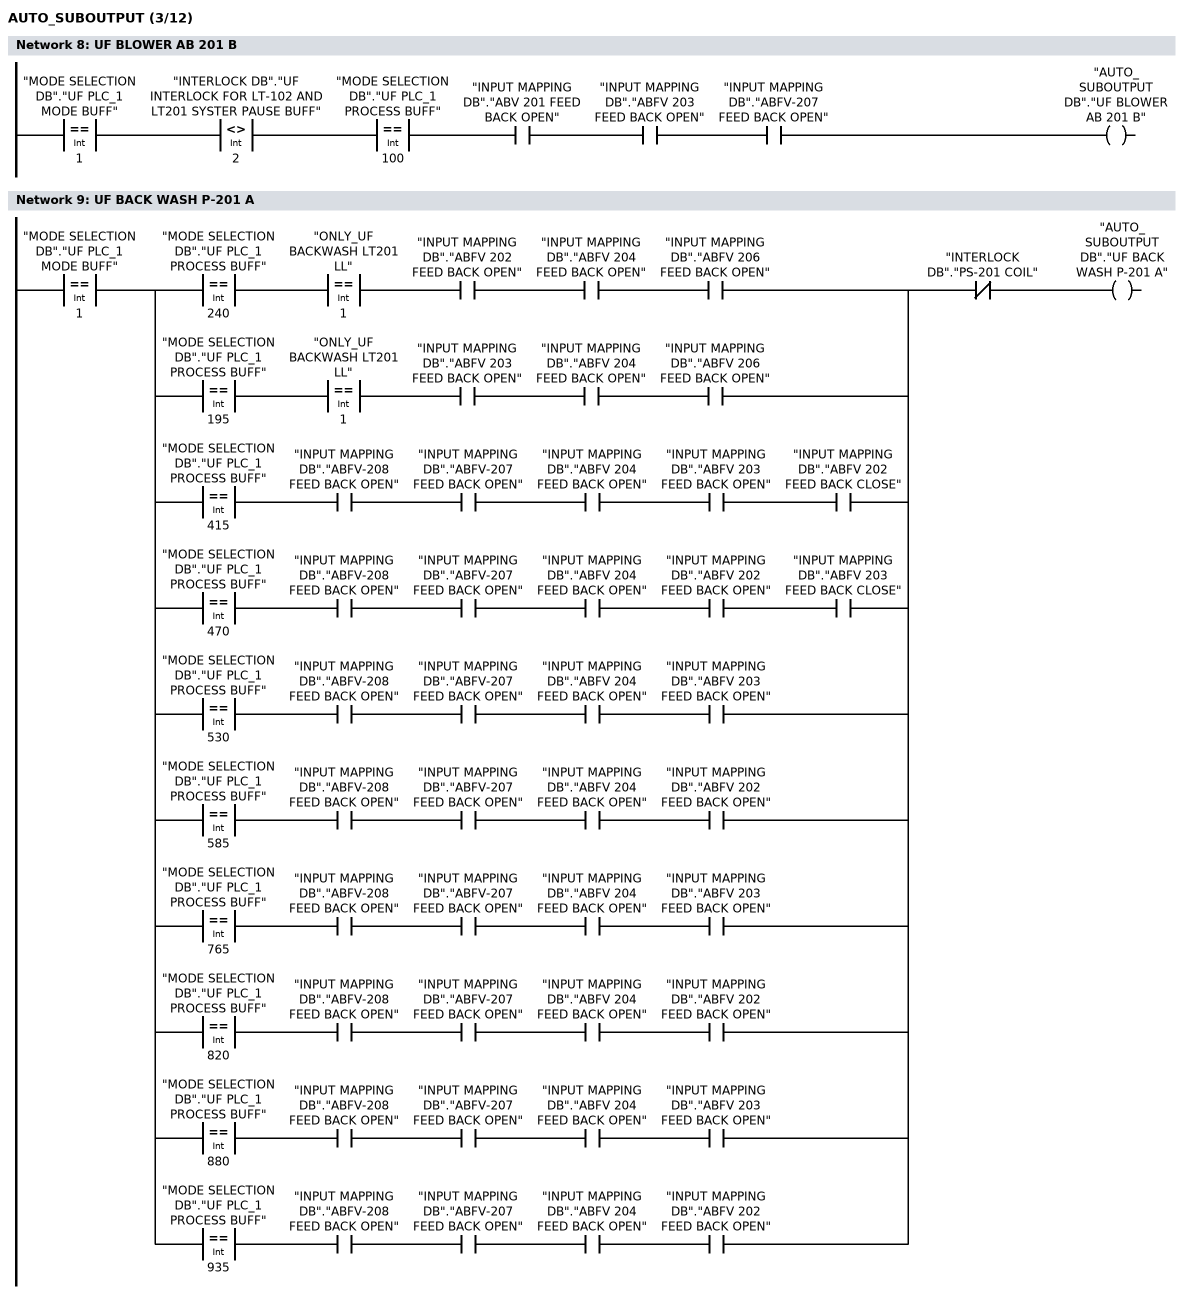
   RUNG wire#powerrail
      { S7_Templates := "SrcType := Int" } EQ_Contact(in1 := "MODE SELECTION DB"."UF PLC_1 MODE BUFF", in2 := 1)
      { S7_Templates := "SrcType := Int" } NE_Contact(in1 := "INTERLOCK DB"."UF INTERLOCK FOR LT-102 AND LT201 SYSTER PAUSE BUFF", in2 := 2)
      { S7_Templates := "SrcType := Int" } EQ_Contact(in1 := "MODE SELECTION DB"."UF PLC_1 PROCESS BUFF", in2 := 100)
      Contact( "INPUT MAPPING DB"."ABV 201 FEED BACK OPEN" )
      Contact( "INPUT MAPPING DB"."ABFV 203 FEED BACK OPEN" )
      Contact( "INPUT MAPPING DB"."ABFV-207 FEED BACK OPEN" )
      Coil( "AUTO_SUBOUTPUT DB"."UF BLOWER AB 201 B" )
   END_RUNG
   // the same network as SCL:
   "AUTO_SUBOUTPUT DB"."UF BLOWER AB 201 B" := ("MODE SELECTION DB"."UF PLC_1 MODE BUFF" = 1) AND ("INTERLOCK DB"."UF INTERLOCK FOR LT-102 AND LT201 SYSTER PAUSE BUFF" <> 2) AND ("MODE SELECTION DB"."UF PLC_1 PROCESS BUFF" = 100) AND "INPUT MAPPING DB"."ABV 201 FEED BACK OPEN" AND "INPUT MAPPING DB"."ABFV 203 FEED BACK OPEN" AND "INPUT MAPPING DB"."ABFV-207 FEED BACK OPEN";
END_REGION

REGION Network 9: UF BACK WASH P-201 A
   RUNG wire#powerrail
      { S7_Templates := "SrcType := Int" } EQ_Contact(in1 := "MODE SELECTION DB"."UF PLC_1 MODE BUFF", in2 := 1)
      wire#w1
      { S7_Templates := "SrcType := Int" } EQ_Contact(in1 := "MODE SELECTION DB"."UF PLC_1 PROCESS BUFF", in2 := 240)
      { S7_Templates := "SrcType := Int" } EQ_Contact(in1 := "ONLY_UF BACKWASH LT201 LL", in2 := 1)
      Contact( "INPUT MAPPING DB"."ABFV 202 FEED BACK OPEN" )
      Contact( "INPUT MAPPING DB"."ABFV 204 FEED BACK OPEN" )
      Contact( "INPUT MAPPING DB"."ABFV 206 FEED BACK OPEN" )
      wire#w2
      I_Contact( "INTERLOCK DB"."PS-201 COIL" )
      Coil( "AUTO_SUBOUTPUT DB"."UF BACK WASH P-201 A" )
   END_RUNG
   RUNG wire#w1
      { S7_Templates := "SrcType := Int" } EQ_Contact(in1 := "MODE SELECTION DB"."UF PLC_1 PROCESS BUFF", in2 := 195)
      { S7_Templates := "SrcType := Int" } EQ_Contact(in1 := "ONLY_UF BACKWASH LT201 LL", in2 := 1)
      Contact( "INPUT MAPPING DB"."ABFV 203 FEED BACK OPEN" )
      Contact( "INPUT MAPPING DB"."ABFV 204 FEED BACK OPEN" )
      Contact( "INPUT MAPPING DB"."ABFV 206 FEED BACK OPEN" )
   END_RUNG wire#w2
   RUNG wire#w1
      { S7_Templates := "SrcType := Int" } EQ_Contact(in1 := "MODE SELECTION DB"."UF PLC_1 PROCESS BUFF", in2 := 415)
      Contact( "INPUT MAPPING DB"."ABFV-208 FEED BACK OPEN" )
      Contact( "INPUT MAPPING DB"."ABFV-207 FEED BACK OPEN" )
      Contact( "INPUT MAPPING DB"."ABFV 204 FEED BACK OPEN" )
      Contact( "INPUT MAPPING DB"."ABFV 203 FEED BACK OPEN" )
      Contact( "INPUT MAPPING DB"."ABFV 202 FEED BACK CLOSE" )
   END_RUNG wire#w2
   RUNG wire#w1
      { S7_Templates := "SrcType := Int" } EQ_Contact(in1 := "MODE SELECTION DB"."UF PLC_1 PROCESS BUFF", in2 := 470)
      Contact( "INPUT MAPPING DB"."ABFV-208 FEED BACK OPEN" )
      Contact( "INPUT MAPPING DB"."ABFV-207 FEED BACK OPEN" )
      Contact( "INPUT MAPPING DB"."ABFV 204 FEED BACK OPEN" )
      Contact( "INPUT MAPPING DB"."ABFV 202 FEED BACK OPEN" )
      Contact( "INPUT MAPPING DB"."ABFV 203 FEED BACK CLOSE" )
   END_RUNG wire#w2
   RUNG wire#w1
      { S7_Templates := "SrcType := Int" } EQ_Contact(in1 := "MODE SELECTION DB"."UF PLC_1 PROCESS BUFF", in2 := 530)
      Contact( "INPUT MAPPING DB"."ABFV-208 FEED BACK OPEN" )
      Contact( "INPUT MAPPING DB"."ABFV-207 FEED BACK OPEN" )
      Contact( "INPUT MAPPING DB"."ABFV 204 FEED BACK OPEN" )
      Contact( "INPUT MAPPING DB"."ABFV 203 FEED BACK OPEN" )
   END_RUNG wire#w2
   RUNG wire#w1
      { S7_Templates := "SrcType := Int" } EQ_Contact(in1 := "MODE SELECTION DB"."UF PLC_1 PROCESS BUFF", in2 := 585)
      Contact( "INPUT MAPPING DB"."ABFV-208 FEED BACK OPEN" )
      Contact( "INPUT MAPPING DB"."ABFV-207 FEED BACK OPEN" )
      Contact( "INPUT MAPPING DB"."ABFV 204 FEED BACK OPEN" )
      Contact( "INPUT MAPPING DB"."ABFV 202 FEED BACK OPEN" )
   END_RUNG wire#w2
   RUNG wire#w1
      { S7_Templates := "SrcType := Int" } EQ_Contact(in1 := "MODE SELECTION DB"."UF PLC_1 PROCESS BUFF", in2 := 765)
      Contact( "INPUT MAPPING DB"."ABFV-208 FEED BACK OPEN" )
      Contact( "INPUT MAPPING DB"."ABFV-207 FEED BACK OPEN" )
      Contact( "INPUT MAPPING DB"."ABFV 204 FEED BACK OPEN" )
      Contact( "INPUT MAPPING DB"."ABFV 203 FEED BACK OPEN" )
   END_RUNG wire#w2
   RUNG wire#w1
      { S7_Templates := "SrcType := Int" } EQ_Contact(in1 := "MODE SELECTION DB"."UF PLC_1 PROCESS BUFF", in2 := 820)
      Contact( "INPUT MAPPING DB"."ABFV-208 FEED BACK OPEN" )
      Contact( "INPUT MAPPING DB"."ABFV-207 FEED BACK OPEN" )
      Contact( "INPUT MAPPING DB"."ABFV 204 FEED BACK OPEN" )
      Contact( "INPUT MAPPING DB"."ABFV 202 FEED BACK OPEN" )
   END_RUNG wire#w2
   RUNG wire#w1
      { S7_Templates := "SrcType := Int" } EQ_Contact(in1 := "MODE SELECTION DB"."UF PLC_1 PROCESS BUFF", in2 := 880)
      Contact( "INPUT MAPPING DB"."ABFV-208 FEED BACK OPEN" )
      Contact( "INPUT MAPPING DB"."ABFV-207 FEED BACK OPEN" )
      Contact( "INPUT MAPPING DB"."ABFV 204 FEED BACK OPEN" )
      Contact( "INPUT MAPPING DB"."ABFV 203 FEED BACK OPEN" )
   END_RUNG wire#w2
   RUNG wire#w1
      { S7_Templates := "SrcType := Int" } EQ_Contact(in1 := "MODE SELECTION DB"."UF PLC_1 PROCESS BUFF", in2 := 935)
      Contact( "INPUT MAPPING DB"."ABFV-208 FEED BACK OPEN" )
      Contact( "INPUT MAPPING DB"."ABFV-207 FEED BACK OPEN" )
      Contact( "INPUT MAPPING DB"."ABFV 204 FEED BACK OPEN" )
      Contact( "INPUT MAPPING DB"."ABFV 202 FEED BACK OPEN" )
   END_RUNG wire#w2
   // the same network as SCL:
   "AUTO_SUBOUTPUT DB"."UF BACK WASH P-201 A" := ("MODE SELECTION DB"."UF PLC_1 MODE BUFF" = 1) AND ((("MODE SELECTION DB"."UF PLC_1 PROCESS BUFF" = 240) AND ("ONLY_UF BACKWASH LT201 LL" = 1) AND "INPUT MAPPING DB"."ABFV 202 FEED BACK OPEN" AND "INPUT MAPPING DB"."ABFV 204 FEED BACK OPEN" AND "INPUT MAPPING DB"."ABFV 206 FEED BACK OPEN") OR (("MODE SELECTION DB"."UF PLC_1 PROCESS BUFF" = 195) AND ("ONLY_UF BACKWASH LT201 LL" = 1) AND "INPUT MAPPING DB"."ABFV 203 FEED BACK OPEN" AND "INPUT MAPPING DB"."ABFV 204 FEED BACK OPEN" AND "INPUT MAPPING DB"."ABFV 206 FEED BACK OPEN") OR (("MODE SELECTION DB"."UF PLC_1 PROCESS BUFF" = 415) AND "INPUT MAPPING DB"."ABFV-208 FEED BACK OPEN" AND "INPUT MAPPING DB"."ABFV-207 FEED BACK OPEN" AND "INPUT MAPPING DB"."ABFV 204 FEED BACK OPEN" AND "INPUT MAPPING DB"."ABFV 203 FEED BACK OPEN" AND "INPUT MAPPING DB"."ABFV 202 FEED BACK CLOSE") OR (("MODE SELECTION DB"."UF PLC_1 PROCESS BUFF" = 470) AND "INPUT MAPPING DB"."ABFV-208 FEED BACK OPEN" AND "INPUT MAPPING DB"."ABFV-207 FEED BACK OPEN" AND "INPUT MAPPING DB"."ABFV 204 FEED BACK OPEN" AND "INPUT MAPPING DB"."ABFV 202 FEED BACK OPEN" AND "INPUT MAPPING DB"."ABFV 203 FEED BACK CLOSE") OR (("MODE SELECTION DB"."UF PLC_1 PROCESS BUFF" = 530) AND "INPUT MAPPING DB"."ABFV-208 FEED BACK OPEN" AND "INPUT MAPPING DB"."ABFV-207 FEED BACK OPEN" AND "INPUT MAPPING DB"."ABFV 204 FEED BACK OPEN" AND "INPUT MAPPING DB"."ABFV 203 FEED BACK OPEN") OR (("MODE SELECTION DB"."UF PLC_1 PROCESS BUFF" = 585) AND "INPUT MAPPING DB"."ABFV-208 FEED BACK OPEN" AND "INPUT MAPPING DB"."ABFV-207 FEED BACK OPEN" AND "INPUT MAPPING DB"."ABFV 204 FEED BACK OPEN" AND "INPUT MAPPING DB"."ABFV 202 FEED BACK OPEN") OR (("MODE SELECTION DB"."UF PLC_1 PROCESS BUFF" = 765) AND "INPUT MAPPING DB"."ABFV-208 FEED BACK OPEN" AND "INPUT MAPPING DB"."ABFV-207 FEED BACK OPEN" AND "INPUT MAPPING DB"."ABFV 204 FEED BACK OPEN" AND "INPUT MAPPING DB"."ABFV 203 FEED BACK OPEN") OR (("MODE SELECTION DB"."UF PLC_1 PROCESS BUFF" = 820) AND "INPUT MAPPING DB"."ABFV-208 FEED BACK OPEN" AND "INPUT MAPPING DB"."ABFV-207 FEED BACK OPEN" AND "INPUT MAPPING DB"."ABFV 204 FEED BACK OPEN" AND "INPUT MAPPING DB"."ABFV 202 FEED BACK OPEN") OR (("MODE SELECTION DB"."UF PLC_1 PROCESS BUFF" = 880) AND "INPUT MAPPING DB"."ABFV-208 FEED BACK OPEN" AND "INPUT MAPPING DB"."ABFV-207 FEED BACK OPEN" AND "INPUT MAPPING DB"."ABFV 204 FEED BACK OPEN" AND "INPUT MAPPING DB"."ABFV 203 FEED BACK OPEN") OR (("MODE SELECTION DB"."UF PLC_1 PROCESS BUFF" = 935) AND "INPUT MAPPING DB"."ABFV-208 FEED BACK OPEN" AND "INPUT MAPPING DB"."ABFV-207 FEED BACK OPEN" AND "INPUT MAPPING DB"."ABFV 204 FEED BACK OPEN" AND "INPUT MAPPING DB"."ABFV 202 FEED BACK OPEN")) AND NOT "INTERLOCK DB"."PS-201 COIL";
END_REGION

REGION Network 10: UF BACK WASH P-201 B
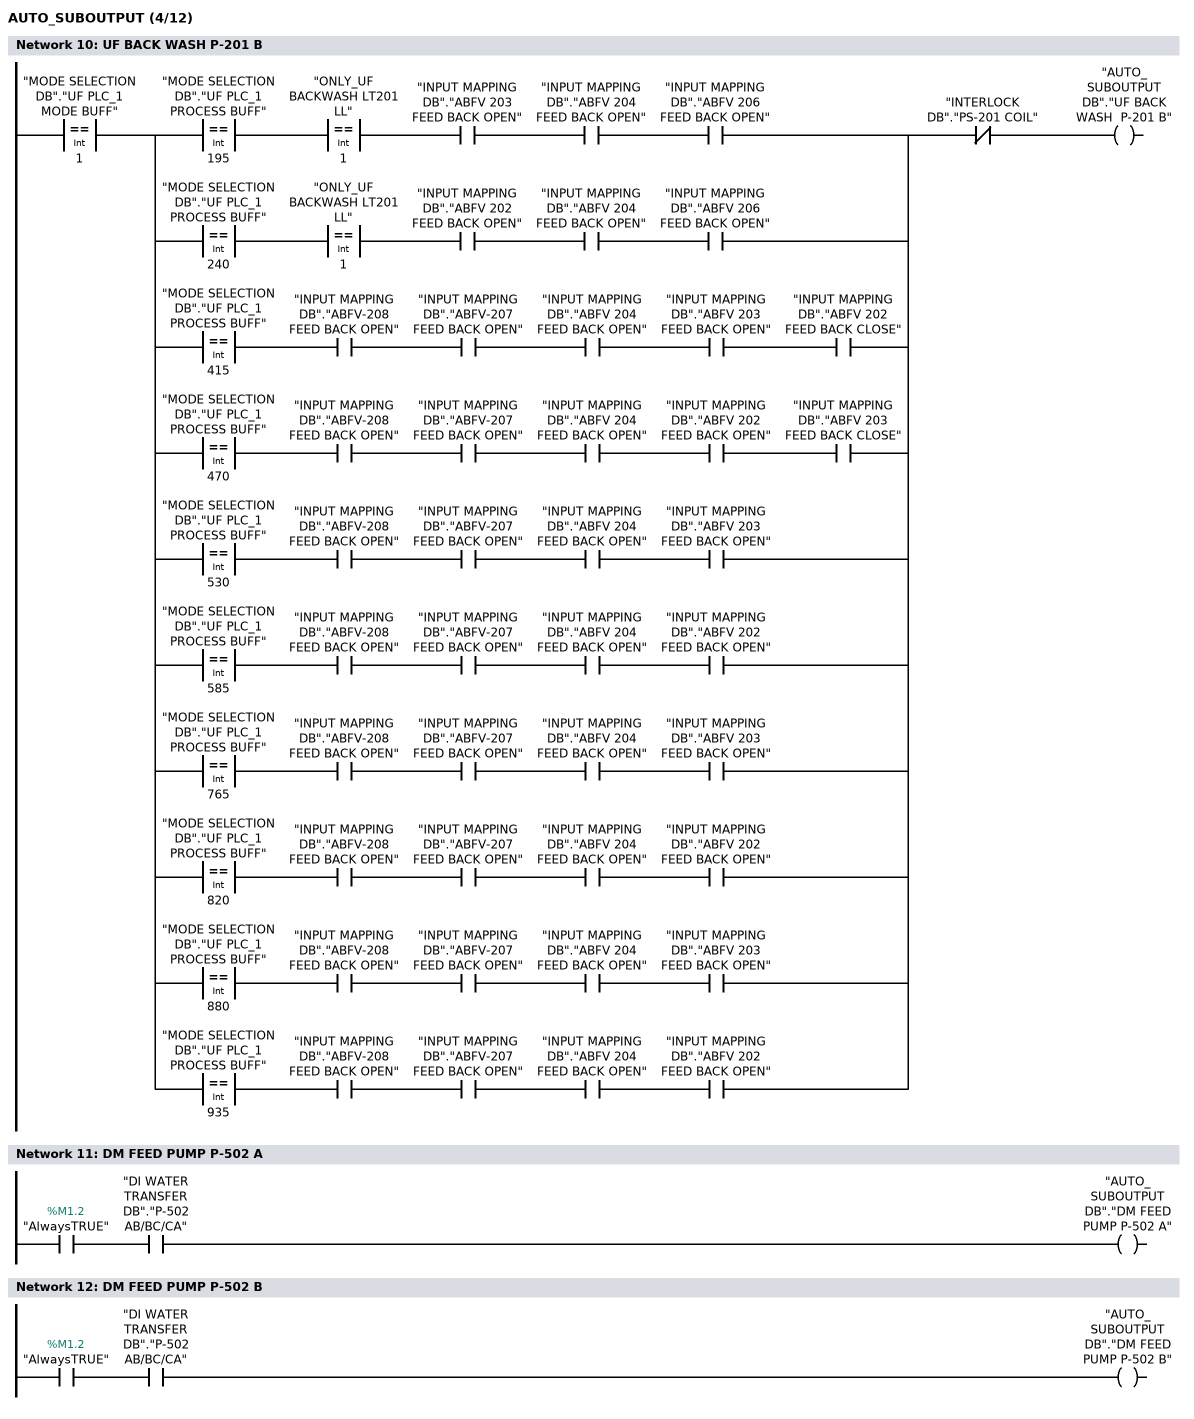
   RUNG wire#powerrail
      { S7_Templates := "SrcType := Int" } EQ_Contact(in1 := "MODE SELECTION DB"."UF PLC_1 MODE BUFF", in2 := 1)
      wire#w1
      { S7_Templates := "SrcType := Int" } EQ_Contact(in1 := "MODE SELECTION DB"."UF PLC_1 PROCESS BUFF", in2 := 195)
      { S7_Templates := "SrcType := Int" } EQ_Contact(in1 := "ONLY_UF BACKWASH LT201 LL", in2 := 1)
      Contact( "INPUT MAPPING DB"."ABFV 203 FEED BACK OPEN" )
      Contact( "INPUT MAPPING DB"."ABFV 204 FEED BACK OPEN" )
      Contact( "INPUT MAPPING DB"."ABFV 206 FEED BACK OPEN" )
      wire#w2
      I_Contact( "INTERLOCK DB"."PS-201 COIL" )
      Coil( "AUTO_SUBOUTPUT DB"."UF BACK WASH  P-201 B" )
   END_RUNG
   RUNG wire#w1
      { S7_Templates := "SrcType := Int" } EQ_Contact(in1 := "MODE SELECTION DB"."UF PLC_1 PROCESS BUFF", in2 := 240)
      { S7_Templates := "SrcType := Int" } EQ_Contact(in1 := "ONLY_UF BACKWASH LT201 LL", in2 := 1)
      Contact( "INPUT MAPPING DB"."ABFV 202 FEED BACK OPEN" )
      Contact( "INPUT MAPPING DB"."ABFV 204 FEED BACK OPEN" )
      Contact( "INPUT MAPPING DB"."ABFV 206 FEED BACK OPEN" )
   END_RUNG wire#w2
   RUNG wire#w1
      { S7_Templates := "SrcType := Int" } EQ_Contact(in1 := "MODE SELECTION DB"."UF PLC_1 PROCESS BUFF", in2 := 415)
      Contact( "INPUT MAPPING DB"."ABFV-208 FEED BACK OPEN" )
      Contact( "INPUT MAPPING DB"."ABFV-207 FEED BACK OPEN" )
      Contact( "INPUT MAPPING DB"."ABFV 204 FEED BACK OPEN" )
      Contact( "INPUT MAPPING DB"."ABFV 203 FEED BACK OPEN" )
      Contact( "INPUT MAPPING DB"."ABFV 202 FEED BACK CLOSE" )
   END_RUNG wire#w2
   RUNG wire#w1
      { S7_Templates := "SrcType := Int" } EQ_Contact(in1 := "MODE SELECTION DB"."UF PLC_1 PROCESS BUFF", in2 := 470)
      Contact( "INPUT MAPPING DB"."ABFV-208 FEED BACK OPEN" )
      Contact( "INPUT MAPPING DB"."ABFV-207 FEED BACK OPEN" )
      Contact( "INPUT MAPPING DB"."ABFV 204 FEED BACK OPEN" )
      Contact( "INPUT MAPPING DB"."ABFV 202 FEED BACK OPEN" )
      Contact( "INPUT MAPPING DB"."ABFV 203 FEED BACK CLOSE" )
   END_RUNG wire#w2
   RUNG wire#w1
      { S7_Templates := "SrcType := Int" } EQ_Contact(in1 := "MODE SELECTION DB"."UF PLC_1 PROCESS BUFF", in2 := 530)
      Contact( "INPUT MAPPING DB"."ABFV-208 FEED BACK OPEN" )
      Contact( "INPUT MAPPING DB"."ABFV-207 FEED BACK OPEN" )
      Contact( "INPUT MAPPING DB"."ABFV 204 FEED BACK OPEN" )
      Contact( "INPUT MAPPING DB"."ABFV 203 FEED BACK OPEN" )
   END_RUNG wire#w2
   RUNG wire#w1
      { S7_Templates := "SrcType := Int" } EQ_Contact(in1 := "MODE SELECTION DB"."UF PLC_1 PROCESS BUFF", in2 := 585)
      Contact( "INPUT MAPPING DB"."ABFV-208 FEED BACK OPEN" )
      Contact( "INPUT MAPPING DB"."ABFV-207 FEED BACK OPEN" )
      Contact( "INPUT MAPPING DB"."ABFV 204 FEED BACK OPEN" )
      Contact( "INPUT MAPPING DB"."ABFV 202 FEED BACK OPEN" )
   END_RUNG wire#w2
   RUNG wire#w1
      { S7_Templates := "SrcType := Int" } EQ_Contact(in1 := "MODE SELECTION DB"."UF PLC_1 PROCESS BUFF", in2 := 765)
      Contact( "INPUT MAPPING DB"."ABFV-208 FEED BACK OPEN" )
      Contact( "INPUT MAPPING DB"."ABFV-207 FEED BACK OPEN" )
      Contact( "INPUT MAPPING DB"."ABFV 204 FEED BACK OPEN" )
      Contact( "INPUT MAPPING DB"."ABFV 203 FEED BACK OPEN" )
   END_RUNG wire#w2
   RUNG wire#w1
      { S7_Templates := "SrcType := Int" } EQ_Contact(in1 := "MODE SELECTION DB"."UF PLC_1 PROCESS BUFF", in2 := 820)
      Contact( "INPUT MAPPING DB"."ABFV-208 FEED BACK OPEN" )
      Contact( "INPUT MAPPING DB"."ABFV-207 FEED BACK OPEN" )
      Contact( "INPUT MAPPING DB"."ABFV 204 FEED BACK OPEN" )
      Contact( "INPUT MAPPING DB"."ABFV 202 FEED BACK OPEN" )
   END_RUNG wire#w2
   RUNG wire#w1
      { S7_Templates := "SrcType := Int" } EQ_Contact(in1 := "MODE SELECTION DB"."UF PLC_1 PROCESS BUFF", in2 := 880)
      Contact( "INPUT MAPPING DB"."ABFV-208 FEED BACK OPEN" )
      Contact( "INPUT MAPPING DB"."ABFV-207 FEED BACK OPEN" )
      Contact( "INPUT MAPPING DB"."ABFV 204 FEED BACK OPEN" )
      Contact( "INPUT MAPPING DB"."ABFV 203 FEED BACK OPEN" )
   END_RUNG wire#w2
   RUNG wire#w1
      { S7_Templates := "SrcType := Int" } EQ_Contact(in1 := "MODE SELECTION DB"."UF PLC_1 PROCESS BUFF", in2 := 935)
      Contact( "INPUT MAPPING DB"."ABFV-208 FEED BACK OPEN" )
      Contact( "INPUT MAPPING DB"."ABFV-207 FEED BACK OPEN" )
      Contact( "INPUT MAPPING DB"."ABFV 204 FEED BACK OPEN" )
      Contact( "INPUT MAPPING DB"."ABFV 202 FEED BACK OPEN" )
   END_RUNG wire#w2
   // the same network as SCL:
   "AUTO_SUBOUTPUT DB"."UF BACK WASH  P-201 B" := ("MODE SELECTION DB"."UF PLC_1 MODE BUFF" = 1) AND ((("MODE SELECTION DB"."UF PLC_1 PROCESS BUFF" = 195) AND ("ONLY_UF BACKWASH LT201 LL" = 1) AND "INPUT MAPPING DB"."ABFV 203 FEED BACK OPEN" AND "INPUT MAPPING DB"."ABFV 204 FEED BACK OPEN" AND "INPUT MAPPING DB"."ABFV 206 FEED BACK OPEN") OR (("MODE SELECTION DB"."UF PLC_1 PROCESS BUFF" = 240) AND ("ONLY_UF BACKWASH LT201 LL" = 1) AND "INPUT MAPPING DB"."ABFV 202 FEED BACK OPEN" AND "INPUT MAPPING DB"."ABFV 204 FEED BACK OPEN" AND "INPUT MAPPING DB"."ABFV 206 FEED BACK OPEN") OR (("MODE SELECTION DB"."UF PLC_1 PROCESS BUFF" = 415) AND "INPUT MAPPING DB"."ABFV-208 FEED BACK OPEN" AND "INPUT MAPPING DB"."ABFV-207 FEED BACK OPEN" AND "INPUT MAPPING DB"."ABFV 204 FEED BACK OPEN" AND "INPUT MAPPING DB"."ABFV 203 FEED BACK OPEN" AND "INPUT MAPPING DB"."ABFV 202 FEED BACK CLOSE") OR (("MODE SELECTION DB"."UF PLC_1 PROCESS BUFF" = 470) AND "INPUT MAPPING DB"."ABFV-208 FEED BACK OPEN" AND "INPUT MAPPING DB"."ABFV-207 FEED BACK OPEN" AND "INPUT MAPPING DB"."ABFV 204 FEED BACK OPEN" AND "INPUT MAPPING DB"."ABFV 202 FEED BACK OPEN" AND "INPUT MAPPING DB"."ABFV 203 FEED BACK CLOSE") OR (("MODE SELECTION DB"."UF PLC_1 PROCESS BUFF" = 530) AND "INPUT MAPPING DB"."ABFV-208 FEED BACK OPEN" AND "INPUT MAPPING DB"."ABFV-207 FEED BACK OPEN" AND "INPUT MAPPING DB"."ABFV 204 FEED BACK OPEN" AND "INPUT MAPPING DB"."ABFV 203 FEED BACK OPEN") OR (("MODE SELECTION DB"."UF PLC_1 PROCESS BUFF" = 585) AND "INPUT MAPPING DB"."ABFV-208 FEED BACK OPEN" AND "INPUT MAPPING DB"."ABFV-207 FEED BACK OPEN" AND "INPUT MAPPING DB"."ABFV 204 FEED BACK OPEN" AND "INPUT MAPPING DB"."ABFV 202 FEED BACK OPEN") OR (("MODE SELECTION DB"."UF PLC_1 PROCESS BUFF" = 765) AND "INPUT MAPPING DB"."ABFV-208 FEED BACK OPEN" AND "INPUT MAPPING DB"."ABFV-207 FEED BACK OPEN" AND "INPUT MAPPING DB"."ABFV 204 FEED BACK OPEN" AND "INPUT MAPPING DB"."ABFV 203 FEED BACK OPEN") OR (("MODE SELECTION DB"."UF PLC_1 PROCESS BUFF" = 820) AND "INPUT MAPPING DB"."ABFV-208 FEED BACK OPEN" AND "INPUT MAPPING DB"."ABFV-207 FEED BACK OPEN" AND "INPUT MAPPING DB"."ABFV 204 FEED BACK OPEN" AND "INPUT MAPPING DB"."ABFV 202 FEED BACK OPEN") OR (("MODE SELECTION DB"."UF PLC_1 PROCESS BUFF" = 880) AND "INPUT MAPPING DB"."ABFV-208 FEED BACK OPEN" AND "INPUT MAPPING DB"."ABFV-207 FEED BACK OPEN" AND "INPUT MAPPING DB"."ABFV 204 FEED BACK OPEN" AND "INPUT MAPPING DB"."ABFV 203 FEED BACK OPEN") OR (("MODE SELECTION DB"."UF PLC_1 PROCESS BUFF" = 935) AND "INPUT MAPPING DB"."ABFV-208 FEED BACK OPEN" AND "INPUT MAPPING DB"."ABFV-207 FEED BACK OPEN" AND "INPUT MAPPING DB"."ABFV 204 FEED BACK OPEN" AND "INPUT MAPPING DB"."ABFV 202 FEED BACK OPEN")) AND NOT "INTERLOCK DB"."PS-201 COIL";
END_REGION

REGION Network 11: DM FEED PUMP P-502 A
   RUNG wire#powerrail
      Contact( "AlwaysTRUE" )
      Contact( "DI WATER TRANSFER DB"."P-502 AB/BC/CA" )
      Coil( "AUTO_SUBOUTPUT DB"."DM FEED PUMP P-502 A" )
   END_RUNG
   // the same network as SCL:
   "AUTO_SUBOUTPUT DB"."DM FEED PUMP P-502 A" := "AlwaysTRUE" AND "DI WATER TRANSFER DB"."P-502 AB/BC/CA";
END_REGION

REGION Network 12: DM FEED PUMP P-502 B
   RUNG wire#powerrail
      Contact( "AlwaysTRUE" )
      Contact( "DI WATER TRANSFER DB"."P-502 AB/BC/CA" )
      Coil( "AUTO_SUBOUTPUT DB"."DM FEED PUMP P-502 B" )
   END_RUNG
   // the same network as SCL:
   "AUTO_SUBOUTPUT DB"."DM FEED PUMP P-502 B" := "AlwaysTRUE" AND "DI WATER TRANSFER DB"."P-502 AB/BC/CA";
END_REGION

REGION Network 13: DM FEED PUMP P-502 C
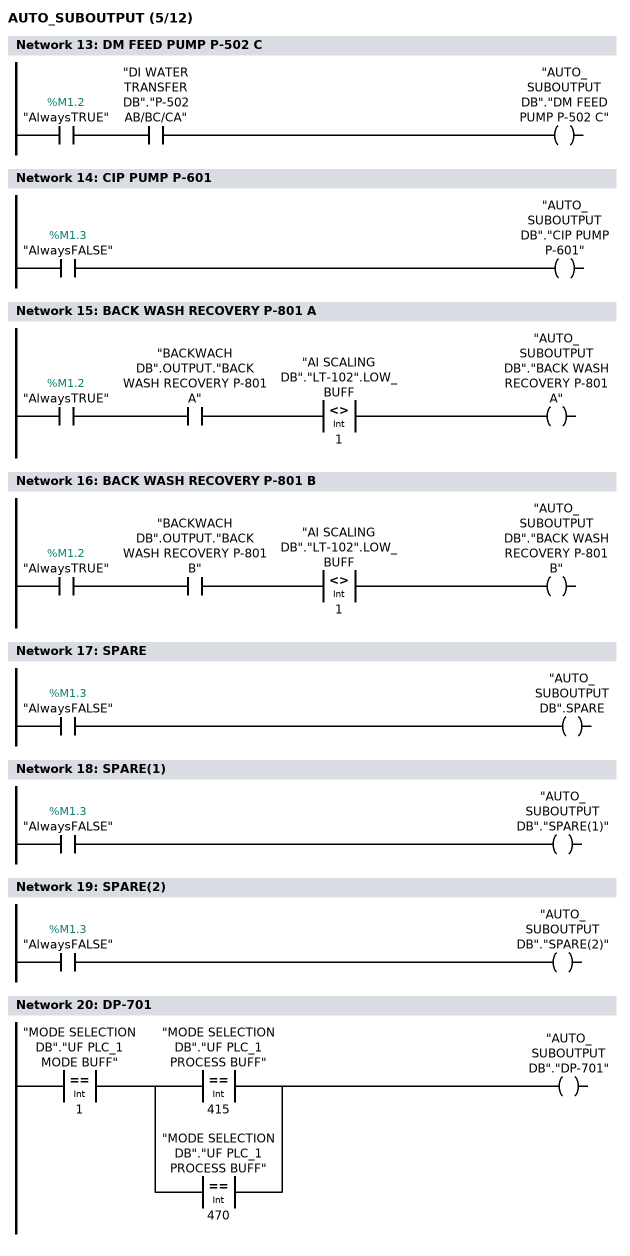
   RUNG wire#powerrail
      Contact( "AlwaysTRUE" )
      Contact( "DI WATER TRANSFER DB"."P-502 AB/BC/CA" )
      Coil( "AUTO_SUBOUTPUT DB"."DM FEED PUMP P-502 C" )
   END_RUNG
   // the same network as SCL:
   "AUTO_SUBOUTPUT DB"."DM FEED PUMP P-502 C" := "AlwaysTRUE" AND "DI WATER TRANSFER DB"."P-502 AB/BC/CA";
END_REGION

REGION Network 14: CIP PUMP P-601
   RUNG wire#powerrail
      Contact( "AlwaysFALSE" )
      Coil( "AUTO_SUBOUTPUT DB"."CIP PUMP P-601" )
   END_RUNG
   // the same network as SCL:
   "AUTO_SUBOUTPUT DB"."CIP PUMP P-601" := "AlwaysFALSE";
END_REGION

REGION Network 15: BACK WASH RECOVERY P-801 A
   RUNG wire#powerrail
      Contact( "AlwaysTRUE" )
      Contact( "BACKWACH DB".OUTPUT."BACK WASH RECOVERY P-801 A" )
      { S7_Templates := "SrcType := Int" } NE_Contact(in1 := "AI SCALING DB"."LT-102".LOW_BUFF, in2 := 1)
      Coil( "AUTO_SUBOUTPUT DB"."BACK WASH RECOVERY P-801 A" )
   END_RUNG
   // the same network as SCL:
   "AUTO_SUBOUTPUT DB"."BACK WASH RECOVERY P-801 A" := "AlwaysTRUE" AND "BACKWACH DB".OUTPUT."BACK WASH RECOVERY P-801 A" AND ("AI SCALING DB"."LT-102".LOW_BUFF <> 1);
END_REGION

REGION Network 16: BACK WASH RECOVERY P-801 B
   RUNG wire#powerrail
      Contact( "AlwaysTRUE" )
      Contact( "BACKWACH DB".OUTPUT."BACK WASH RECOVERY P-801 B" )
      { S7_Templates := "SrcType := Int" } NE_Contact(in1 := "AI SCALING DB"."LT-102".LOW_BUFF, in2 := 1)
      Coil( "AUTO_SUBOUTPUT DB"."BACK WASH RECOVERY P-801 B" )
   END_RUNG
   // the same network as SCL:
   "AUTO_SUBOUTPUT DB"."BACK WASH RECOVERY P-801 B" := "AlwaysTRUE" AND "BACKWACH DB".OUTPUT."BACK WASH RECOVERY P-801 B" AND ("AI SCALING DB"."LT-102".LOW_BUFF <> 1);
END_REGION

REGION Network 17: SPARE
   RUNG wire#powerrail
      Contact( "AlwaysFALSE" )
      Coil( "AUTO_SUBOUTPUT DB".SPARE )
   END_RUNG
   // the same network as SCL:
   "AUTO_SUBOUTPUT DB".SPARE := "AlwaysFALSE";
END_REGION

REGION Network 18: SPARE(1)
   RUNG wire#powerrail
      Contact( "AlwaysFALSE" )
      Coil( "AUTO_SUBOUTPUT DB"."SPARE(1)" )
   END_RUNG
   // the same network as SCL:
   "AUTO_SUBOUTPUT DB"."SPARE(1)" := "AlwaysFALSE";
END_REGION

REGION Network 19: SPARE(2)
   RUNG wire#powerrail
      Contact( "AlwaysFALSE" )
      Coil( "AUTO_SUBOUTPUT DB"."SPARE(2)" )
   END_RUNG
   // the same network as SCL:
   "AUTO_SUBOUTPUT DB"."SPARE(2)" := "AlwaysFALSE";
END_REGION

REGION Network 20: DP-701
   RUNG wire#powerrail
      { S7_Templates := "SrcType := Int" } EQ_Contact(in1 := "MODE SELECTION DB"."UF PLC_1 MODE BUFF", in2 := 1)
      wire#w1
      { S7_Templates := "SrcType := Int" } EQ_Contact(in1 := "MODE SELECTION DB"."UF PLC_1 PROCESS BUFF", in2 := 415)
      wire#w2
      Coil( "AUTO_SUBOUTPUT DB"."DP-701" )
   END_RUNG
   RUNG wire#w1
      { S7_Templates := "SrcType := Int" } EQ_Contact(in1 := "MODE SELECTION DB"."UF PLC_1 PROCESS BUFF", in2 := 470)
   END_RUNG wire#w2
   // the same network as SCL:
   "AUTO_SUBOUTPUT DB"."DP-701" := ("MODE SELECTION DB"."UF PLC_1 MODE BUFF" = 1) AND (("MODE SELECTION DB"."UF PLC_1 PROCESS BUFF" = 415) OR ("MODE SELECTION DB"."UF PLC_1 PROCESS BUFF" = 470));
END_REGION

REGION Network 21: DP-702
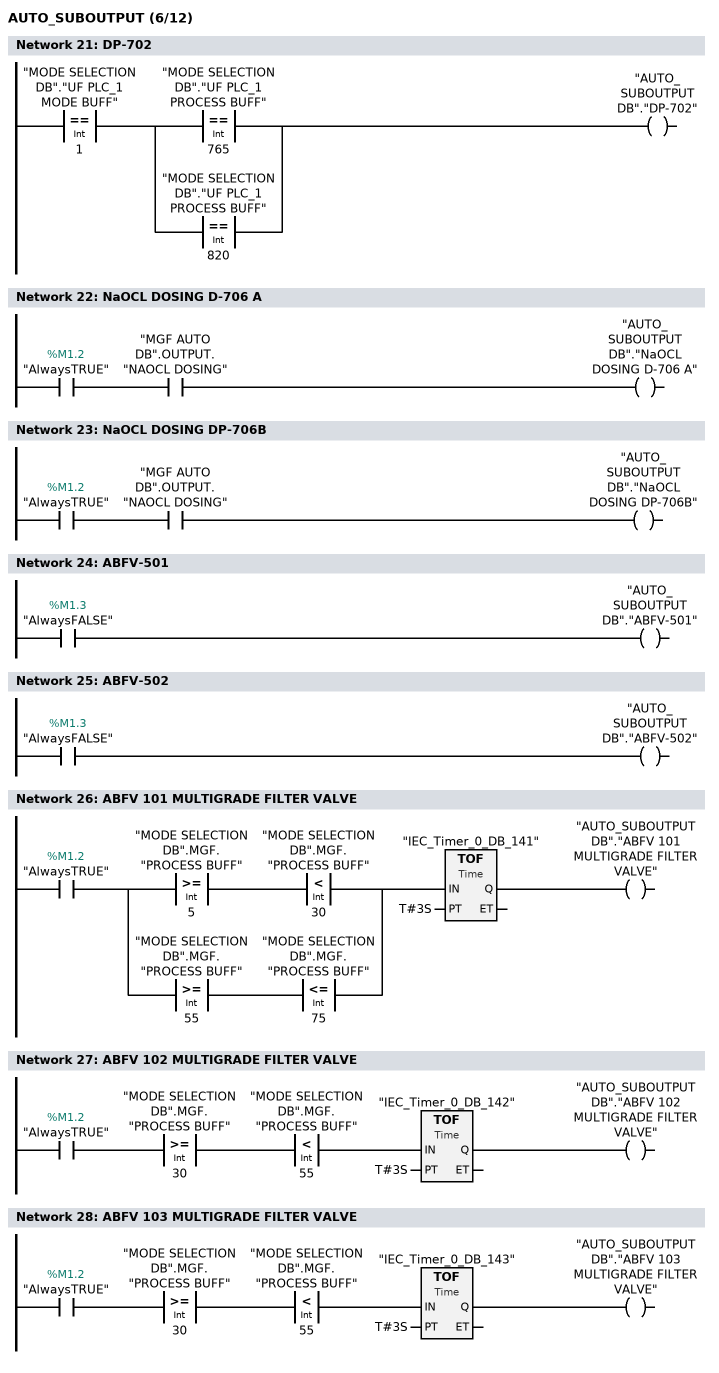
   RUNG wire#powerrail
      { S7_Templates := "SrcType := Int" } EQ_Contact(in1 := "MODE SELECTION DB"."UF PLC_1 MODE BUFF", in2 := 1)
      wire#w1
      { S7_Templates := "SrcType := Int" } EQ_Contact(in1 := "MODE SELECTION DB"."UF PLC_1 PROCESS BUFF", in2 := 765)
      wire#w2
      Coil( "AUTO_SUBOUTPUT DB"."DP-702" )
   END_RUNG
   RUNG wire#w1
      { S7_Templates := "SrcType := Int" } EQ_Contact(in1 := "MODE SELECTION DB"."UF PLC_1 PROCESS BUFF", in2 := 820)
   END_RUNG wire#w2
   // the same network as SCL:
   "AUTO_SUBOUTPUT DB"."DP-702" := ("MODE SELECTION DB"."UF PLC_1 MODE BUFF" = 1) AND (("MODE SELECTION DB"."UF PLC_1 PROCESS BUFF" = 765) OR ("MODE SELECTION DB"."UF PLC_1 PROCESS BUFF" = 820));
END_REGION

REGION Network 22: NaOCL DOSING D-706 A
   RUNG wire#powerrail
      Contact( "AlwaysTRUE" )
      Contact( "MGF AUTO DB".OUTPUT."NAOCL DOSING" )
      Coil( "AUTO_SUBOUTPUT DB"."NaOCL DOSING D-706 A" )
   END_RUNG
   // the same network as SCL:
   "AUTO_SUBOUTPUT DB"."NaOCL DOSING D-706 A" := "AlwaysTRUE" AND "MGF AUTO DB".OUTPUT."NAOCL DOSING";
END_REGION

REGION Network 23: NaOCL DOSING DP-706B
   RUNG wire#powerrail
      Contact( "AlwaysTRUE" )
      Contact( "MGF AUTO DB".OUTPUT."NAOCL DOSING" )
      Coil( "AUTO_SUBOUTPUT DB"."NaOCL DOSING DP-706B" )
   END_RUNG
   // the same network as SCL:
   "AUTO_SUBOUTPUT DB"."NaOCL DOSING DP-706B" := "AlwaysTRUE" AND "MGF AUTO DB".OUTPUT."NAOCL DOSING";
END_REGION

REGION Network 24: ABFV-501
   RUNG wire#powerrail
      Contact( "AlwaysFALSE" )
      Coil( "AUTO_SUBOUTPUT DB"."ABFV-501" )
   END_RUNG
   // the same network as SCL:
   "AUTO_SUBOUTPUT DB"."ABFV-501" := "AlwaysFALSE";
END_REGION

REGION Network 25: ABFV-502
   RUNG wire#powerrail
      Contact( "AlwaysFALSE" )
      Coil( "AUTO_SUBOUTPUT DB"."ABFV-502" )
   END_RUNG
   // the same network as SCL:
   "AUTO_SUBOUTPUT DB"."ABFV-502" := "AlwaysFALSE";
END_REGION

REGION Network 26: ABFV 101 MULTIGRADE FILTER VALVE
   RUNG wire#powerrail
      Contact( "AlwaysTRUE" )
      wire#w1
      { S7_Templates := "SrcType := Int" } GE_Contact(in1 := "MODE SELECTION DB".MGF."PROCESS BUFF", in2 := 5)
      { S7_Templates := "SrcType := Int" } LT_Contact(in1 := "MODE SELECTION DB".MGF."PROCESS BUFF", in2 := 30)
      wire#w2
      { S7_Templates := "time_type := Time" } "IEC_Timer_0_DB_141".TOF(pt := T#3S, et =>)
      Coil( "AUTO_SUBOUTPUT DB"."ABFV 101 MULTIGRADE FILTER VALVE" )
   END_RUNG
   RUNG wire#w1
      { S7_Templates := "SrcType := Int" } GE_Contact(in1 := "MODE SELECTION DB".MGF."PROCESS BUFF", in2 := 55)
      { S7_Templates := "SrcType := Int" } LE_Contact(in1 := "MODE SELECTION DB".MGF."PROCESS BUFF", in2 := 75)
   END_RUNG wire#w2
   // the same network as SCL:
   "IEC_Timer_0_DB_141".TOF(IN := "AlwaysTRUE" AND ((("MODE SELECTION DB".MGF."PROCESS BUFF" >= 5) AND ("MODE SELECTION DB".MGF."PROCESS BUFF" < 30)) OR (("MODE SELECTION DB".MGF."PROCESS BUFF" >= 55) AND ("MODE SELECTION DB".MGF."PROCESS BUFF" <= 75))),
                           PT := T#3S);
   "AUTO_SUBOUTPUT DB"."ABFV 101 MULTIGRADE FILTER VALVE" := "IEC_Timer_0_DB_141".Q;
END_REGION

REGION Network 27: ABFV 102 MULTIGRADE FILTER VALVE
   RUNG wire#powerrail
      Contact( "AlwaysTRUE" )
      { S7_Templates := "SrcType := Int" } GE_Contact(in1 := "MODE SELECTION DB".MGF."PROCESS BUFF", in2 := 30)
      { S7_Templates := "SrcType := Int" } LT_Contact(in1 := "MODE SELECTION DB".MGF."PROCESS BUFF", in2 := 55)
      { S7_Templates := "time_type := Time" } "IEC_Timer_0_DB_142".TOF(pt := T#3S, et =>)
      Coil( "AUTO_SUBOUTPUT DB"."ABFV 102 MULTIGRADE FILTER VALVE" )
   END_RUNG
   // the same network as SCL:
   "IEC_Timer_0_DB_142".TOF(IN := "AlwaysTRUE" AND ("MODE SELECTION DB".MGF."PROCESS BUFF" >= 30) AND ("MODE SELECTION DB".MGF."PROCESS BUFF" < 55),
                           PT := T#3S);
   "AUTO_SUBOUTPUT DB"."ABFV 102 MULTIGRADE FILTER VALVE" := "IEC_Timer_0_DB_142".Q;
END_REGION

